(* LS Electric XG5000 project: 1군지사 유류제어(V1.0.3) *)
(* PLC LSPLC *)
(* module base 0 slot 0: FEnet:XGL-EFMT(B) (Fast Ethernet 통신 모듈, 전기 Master) *)
(* module base 1 slot 0: 입력 모듈:XGI-D28A/B (DC 24V 입력, 64점 (전류소스 싱크공용/ 전류소스 입력)) *)
(* module base 1 slot 1: 입력 모듈:XGI-D28A/B (DC 24V 입력, 64점 (전류소스 싱크공용/ 전류소스 입력)) *)
(* module base 1 slot 2: 출력 모듈:XGQ-TR8A/B (트랜지스터 출력, 64점 (0.1A용, 싱크출력/소스출력)) *)
(* module base 1 slot 3: 출력 모듈:XGQ-TR4A/B (트랜지스터 출력, 32점 (0.1A용, 싱크출력/소스출력)) *)
(* module base 1 slot 4: 출력 모듈:XGQ-TR8A/B (트랜지스터 출력, 64점 (0.1A용, 싱크출력/소스출력)) *)
(* module base 1 slot 5: 입력 모듈:XGI-D24A/B (DC 24V 입력, 32점 (전류소스 싱크공용/ 전류소스 입력)) *)
(* module base 1 slot 6: 출력 모듈:XGQ-TR8A/B (트랜지스터 출력, 64점 (0.1A용, 싱크출력/소스출력)) *)
(* module base 1 slot 7: 출력 모듈:XGQ-TR4A/B (트랜지스터 출력, 32점 (0.1A용, 싱크출력/소스출력)) *)
(* module base 1 slot 8: 아날로그입력 모듈:XGF-AD4S (A/D 절연형 4채널) *)
(* module base 1 slot 9: 아날로그출력 모듈:XGF-DC4S (D/A 절연형 4채널(전류형)) *)
(* module base 1 slot 10: 아날로그출력 모듈:XGF-DC4S (D/A 절연형 4채널(전류형)) *)
(* module base 1 slot 11: 입력 모듈:XGI-D24A/B (DC 24V 입력, 32점 (전류소스 싱크공용/ 전류소스 입력)) *)
(* module base 2 slot 0: 입력 모듈:XGI-D24A/B (DC 24V 입력, 32점 (전류소스 싱크공용/ 전류소스 입력)) *)
(* module base 2 slot 1: 입력 모듈:XGI-D24A/B (DC 24V 입력, 32점 (전류소스 싱크공용/ 전류소스 입력)) *)
(* module base 2 slot 2: 입력 모듈:XGI-D24A/B (DC 24V 입력, 32점 (전류소스 싱크공용/ 전류소스 입력)) *)
(* module base 2 slot 3: 출력 모듈:XGQ-TR4A/B (트랜지스터 출력, 32점 (0.1A용, 싱크출력/소스출력)) *)
(* module base 2 slot 4: 출력 모듈:XGQ-TR4A/B (트랜지스터 출력, 32점 (0.1A용, 싱크출력/소스출력)) *)
(* module base 2 slot 5: 출력 모듈:XGQ-TR4A/B (트랜지스터 출력, 32점 (0.1A용, 싱크출력/소스출력)) *)
(* module base 2 slot 6: 아날로그입력 모듈:XGF-AD4S (A/D 절연형 4채널) *)
(* module base 2 slot 7: 아날로그출력 모듈:XGF-DC4S (D/A 절연형 4채널(전류형)) *)
(* module base 2 slot 9: 입력 모듈:XGI-D24A/B (DC 24V 입력, 32점 (전류소스 싱크공용/ 전류소스 입력)) *)
(* module base 3 slot 0: 입력 모듈:XGI-D24A/B (DC 24V 입력, 32점 (전류소스 싱크공용/ 전류소스 입력)) *)
(* module base 3 slot 1: 입력 모듈:XGI-D24A/B (DC 24V 입력, 32점 (전류소스 싱크공용/ 전류소스 입력)) *)
(* module base 3 slot 2: 입력 모듈:XGI-D24A/B (DC 24V 입력, 32점 (전류소스 싱크공용/ 전류소스 입력)) *)
(* module base 3 slot 3: 출력 모듈:XGQ-TR4A/B (트랜지스터 출력, 32점 (0.1A용, 싱크출력/소스출력)) *)
(* module base 3 slot 4: 출력 모듈:XGQ-TR4A/B (트랜지스터 출력, 32점 (0.1A용, 싱크출력/소스출력)) *)
(* module base 3 slot 5: 출력 모듈:XGQ-TR4A/B (트랜지스터 출력, 32점 (0.1A용, 싱크출력/소스출력)) *)
(* module base 3 slot 6: 출력 모듈:XGQ-TR4A/B (트랜지스터 출력, 32점 (0.1A용, 싱크출력/소스출력)) *)
(* module base 3 slot 7: 아날로그입력 모듈:XGF-AD4S (A/D 절연형 4채널) *)
(* module base 3 slot 8: 아날로그출력 모듈:XGF-DC4S (D/A 절연형 4채널(전류형)) *)
(* module base 4 slot 0: Cnet:XGL-CH2A/B (Cnet 통신 모듈(RS-232C, RS-422/485)) *)
VAR_GLOBAL
    RP01_2차 : TON;
    RP01_3차 : TON;
    _0108_CH0_ACT AT %UX1.8.16 : BOOL; (* 절연형 아날로그입력 모듈: 채널0 운전중 *)
    _0108_CH0_DATA AT %UW1.8.2 : INT; (* 절연형 아날로그입력 모듈: 채널0 변환값 *)
    _0108_CH0_IDD AT %UX1.8.160 : BOOL; (* 절연형 아날로그입력 모듈: 채널0 입력단선검출 *)
    _0108_CH1_ACT AT %UX1.8.17 : BOOL; (* 절연형 아날로그입력 모듈: 채널1 운전중 *)
    _0108_CH1_DATA AT %UW1.8.3 : INT; (* 절연형 아날로그입력 모듈: 채널1 변환값 *)
    _0108_CH1_IDD AT %UX1.8.161 : BOOL; (* 절연형 아날로그입력 모듈: 채널1 입력단선검출 *)
    _0108_CH2_ACT AT %UX1.8.18 : BOOL; (* 절연형 아날로그입력 모듈: 채널2 운전중 *)
    _0108_CH2_DATA AT %UW1.8.4 : INT; (* 절연형 아날로그입력 모듈: 채널2 변환값 *)
    _0108_CH2_IDD AT %UX1.8.162 : BOOL; (* 절연형 아날로그입력 모듈: 채널2 입력단선검출 *)
    _0108_CH3_ACT AT %UX1.8.19 : BOOL; (* 절연형 아날로그입력 모듈: 채널3 운전중 *)
    _0108_CH3_DATA AT %UW1.8.5 : INT; (* 절연형 아날로그입력 모듈: 채널3 변환값 *)
    _0108_CH3_IDD AT %UX1.8.163 : BOOL; (* 절연형 아날로그입력 모듈: 채널3 입력단선검출 *)
    _0109_CH0_ACT AT %UX1.9.16 : BOOL; (* 절연형 아날로그출력 모듈: 채널0 운전중 *)
    _0109_CH0_DATA AT %UW1.9.3 : INT; (* 절연형 아날로그출력 모듈: 채널0 입력값 *)
    _0109_CH0_ERR AT %UX1.9.0 : BOOL; (* 절연형 아날로그출력 모듈: 채널0 에러 *)
    _0109_CH0_OUTEN AT %UX1.9.32 : BOOL; (* 절연형 아날로그출력 모듈: 채널0 출력상태설정 *)
    _0109_CH1_ACT AT %UX1.9.17 : BOOL; (* 절연형 아날로그출력 모듈: 채널1 운전중 *)
    _0109_CH1_DATA AT %UW1.9.4 : INT; (* 절연형 아날로그출력 모듈: 채널1 입력값 *)
    _0109_CH1_ERR AT %UX1.9.1 : BOOL; (* 절연형 아날로그출력 모듈: 채널1 에러 *)
    _0109_CH2_ACT AT %UX1.9.18 : BOOL; (* 절연형 아날로그출력 모듈: 채널2 운전중 *)
    _0109_CH2_DATA AT %UW1.9.5 : INT; (* 절연형 아날로그출력 모듈: 채널2 입력값 *)
    _0109_CH2_ERR AT %UX1.9.2 : BOOL; (* 절연형 아날로그출력 모듈: 채널2 에러 *)
    _0109_CH3_ACT AT %UX1.9.19 : BOOL; (* 절연형 아날로그출력 모듈: 채널3 운전중 *)
    _0109_CH3_DATA AT %UW1.9.6 : INT; (* 절연형 아날로그출력 모듈: 채널3 입력값 *)
    _0109_CH3_ERR AT %UX1.9.3 : BOOL; (* 절연형 아날로그출력 모듈: 채널3 에러 *)
    _0109_OUTEN AT %UW1.9.2 : WORD; (* 절연형 아날로그출력 모듈: 출력상태 설정 *)
    _0110_CH0_ACT AT %UX1.10.16 : BOOL; (* 절연형 아날로그출력 모듈: 채널0 운전중 *)
    _0110_CH0_DATA AT %UW1.10.3 : INT; (* 절연형 아날로그출력 모듈: 채널0 입력값 *)
    _0110_CH0_ERR AT %UX1.10.0 : BOOL; (* 절연형 아날로그출력 모듈: 채널0 에러 *)
    _0110_OUTEN AT %UW1.10.2 : WORD; (* 절연형 아날로그출력 모듈: 출력상태 설정 *)
    _0206_CH0_ACT AT %UX2.6.16 : BOOL; (* 절연형 아날로그입력 모듈: 채널0 운전중 *)
    _0206_CH0_DATA AT %UW2.6.2 : INT; (* 절연형 아날로그입력 모듈: 채널0 변환값 *)
    _0206_CH0_IDD AT %UX2.6.160 : BOOL; (* 절연형 아날로그입력 모듈: 채널0 입력단선검출 *)
    _0206_CH1_ACT AT %UX2.6.17 : BOOL; (* 절연형 아날로그입력 모듈: 채널1 운전중 *)
    _0206_CH1_DATA AT %UW2.6.3 : INT; (* 절연형 아날로그입력 모듈: 채널1 변환값 *)
    _0206_CH1_IDD AT %UX2.6.161 : BOOL; (* 절연형 아날로그입력 모듈: 채널1 입력단선검출 *)
    _0206_CH2_ACT AT %UX2.6.18 : BOOL; (* 절연형 아날로그입력 모듈: 채널2 운전중 *)
    _0206_CH2_DATA AT %UW2.6.4 : INT; (* 절연형 아날로그입력 모듈: 채널2 변환값 *)
    _0206_CH2_IDD AT %UX2.6.162 : BOOL; (* 절연형 아날로그입력 모듈: 채널2 입력단선검출 *)
    _0206_CH3_ACT AT %UX2.6.19 : BOOL; (* 절연형 아날로그입력 모듈: 채널3 운전중 *)
    _0206_CH3_DATA AT %UW2.6.5 : INT; (* 절연형 아날로그입력 모듈: 채널3 변환값 *)
    _0206_CH3_IDD AT %UX2.6.163 : BOOL; (* 절연형 아날로그입력 모듈: 채널3 입력단선검출 *)
    _0207_CH0_ACT AT %UX2.7.16 : BOOL; (* 절연형 아날로그출력 모듈: 채널0 운전중 *)
    _0207_CH0_DATA AT %UW2.7.3 : INT; (* 절연형 아날로그출력 모듈: 채널0 입력값 *)
    _0207_CH0_ERR AT %UX2.7.0 : BOOL; (* 절연형 아날로그출력 모듈: 채널0 에러 *)
    _0207_CH1_ACT AT %UX2.7.17 : BOOL; (* 절연형 아날로그출력 모듈: 채널1 운전중 *)
    _0207_CH1_DATA AT %UW2.7.4 : INT; (* 절연형 아날로그출력 모듈: 채널1 입력값 *)
    _0207_CH2_ACT AT %UX2.7.18 : BOOL; (* 절연형 아날로그출력 모듈: 채널2 운전중 *)
    _0207_CH2_DATA AT %UW2.7.5 : INT; (* 절연형 아날로그출력 모듈: 채널2 입력값 *)
    _0207_CH2_ERR AT %UX2.7.2 : BOOL; (* 절연형 아날로그출력 모듈: 채널2 에러 *)
    _0207_CH3_DATA AT %UW2.7.6 : INT; (* 절연형 아날로그출력 모듈: 채널3 입력값 *)
    _0207_OUTEN AT %UW2.7.2 : WORD; (* 절연형 아날로그출력 모듈: 출력상태 설정 *)
    _0307_CH0_ACT AT %UX3.7.16 : BOOL; (* 절연형 아날로그입력 모듈: 채널0 운전중 *)
    _0307_CH0_DATA AT %UW3.7.2 : INT; (* 절연형 아날로그입력 모듈: 채널0 변환값 *)
    _0307_CH0_IDD AT %UX3.7.160 : BOOL; (* 절연형 아날로그입력 모듈: 채널0 입력단선검출 *)
    _0307_CH1_ACT AT %UX3.7.17 : BOOL; (* 절연형 아날로그입력 모듈: 채널1 운전중 *)
    _0307_CH1_DATA AT %UW3.7.3 : INT; (* 절연형 아날로그입력 모듈: 채널1 변환값 *)
    _0307_CH1_IDD AT %UX3.7.161 : BOOL; (* 절연형 아날로그입력 모듈: 채널1 입력단선검출 *)
    _0307_CH2_ACT AT %UX3.7.18 : BOOL; (* 절연형 아날로그입력 모듈: 채널2 운전중 *)
    _0307_CH2_DATA AT %UW3.7.4 : INT; (* 절연형 아날로그입력 모듈: 채널2 변환값 *)
    _0307_CH2_IDD AT %UX3.7.162 : BOOL; (* 절연형 아날로그입력 모듈: 채널2 입력단선검출 *)
    _0307_CH3_DATA AT %UW3.7.5 : INT; (* 절연형 아날로그입력 모듈: 채널3 변환값 *)
    _0307_CH3_IDD AT %UX3.7.163 : BOOL; (* 절연형 아날로그입력 모듈: 채널3 입력단선검출 *)
    _0308_CH0_ACT AT %UX3.8.16 : BOOL; (* 절연형 아날로그출력 모듈: 채널0 운전중 *)
    _0308_CH0_DATA AT %UW3.8.3 : INT; (* 절연형 아날로그출력 모듈: 채널0 입력값 *)
    _0308_CH1_ACT AT %UX3.8.17 : BOOL; (* 절연형 아날로그출력 모듈: 채널1 운전중 *)
    _0308_CH1_DATA AT %UW3.8.4 : INT; (* 절연형 아날로그출력 모듈: 채널1 입력값 *)
    _0308_CH2_ACT AT %UX3.8.18 : BOOL; (* 절연형 아날로그출력 모듈: 채널2 운전중 *)
    _0308_CH2_DATA AT %UW3.8.5 : INT; (* 절연형 아날로그출력 모듈: 채널2 입력값 *)
    _0308_CH2_ERR AT %UX3.8.2 : BOOL; (* 절연형 아날로그출력 모듈: 채널2 에러 *)
    _0308_CH3_ACT AT %UX3.8.19 : BOOL; (* 절연형 아날로그출력 모듈: 채널3 운전중 *)
    _0308_CH3_DATA AT %UW3.8.6 : INT; (* 절연형 아날로그출력 모듈: 채널3 입력값 *)
    _0308_CH3_ERR AT %UX3.8.3 : BOOL; (* 절연형 아날로그출력 모듈: 채널3 에러 *)
    _0308_OUTEN AT %UW3.8.2 : WORD; (* 절연형 아날로그출력 모듈: 출력상태 설정 *)
END_VAR
VAR_GLOBAL CONSTANT
    _F0308_CH0_DEC_RATE : UINT := 30; (* 절연형 아날로그출력 모듈: 채널0 변화율 감소값 *)
    _F0308_CH0_STAT : UINT := 03; (* 절연형 아날로그출력 모듈: 채널0 이상 상태 출력 설정값 *)
    _F0308_LIMIT_EN : UINT := 19; (* 절연형 아날로그출력 모듈: 출력제한 채널 설정 *)
END_VAR

(* Comments on direct variables
%QX1.2.0	UPS ON LAMP
%QX1.2.1	UPS TROUBLE LAMP
%QX1.2.2	MCC ON LAMP
%QX1.2.3	AUTO LAMP
%QX1.2.4	MANUAL LAMP
%QX1.2.5	HORN STOP LAMP
%QX1.2.6	RESET LAMP
%QX1.2.7	LAMP TEST LAMP
%QX1.2.8	SYSTEM PRESSURE MIN
LAMP
%QX1.2.9	PUMP RESTART 6TIME/H
LAMP
%QX1.2.10	EV-1 LAMP
%QX1.2.11	EV-2 LAMP
%QX1.2.12	BPCV LAMP
%QX1.2.13	SPARE LAMP
%QX1.2.14	SPARE LAMP
%QX1.2.15	CONTROL PANEL EM S/W
LAMP
%QX1.2.16	DF-1A TANK EM S/W
LAMP
%QX1.2.17	DF-1B TANK EM S/W
LAMP
%QX1.2.18	DRAIN TANK EM S/W
LAMP
%QX1.2.19	FILTER ROOM EM S/W
LAMP
%QX1.2.20	대량 주유대 1 EM S/W
LAMP
%QX1.2.21	대량 주유대 2 EM S/W
LAMP
%QX1.2.22	대량 주유대 3 EM S/W
LAMP
%QX1.2.23	대량 주유대 4 EM S/W
LAMP
%QX1.2.24	포장 주유대 EM S/W
LAMP
%QX1.2.25	PIT-1 TROUBLE LAMP
%QX1.2.26	PIT-2 TROUBLE LAMP
%QX1.2.27	FIT-1 TROUBLE LAMP
%QX1.2.28	FIT-2 TROUBLE LAMP
%QX1.2.29	PLC 1 RUN LAMP
%QX1.2.30	PLC 1 STANDBY LAMP
%QX1.2.31	PLC 1 TROUBLE LAMP
%QX1.2.32	PLC 2 RUN LAMP

%QX1.2.33	PLC 2 STANDBY LAMP

%QX1.2.34	PLC 2 TROUBLE LAMP

%QX1.2.35	DF-1 DRAIN PUMP 1 TROUBLE LAMP

%QX1.2.36	DF-1 DRAIN PUMP 1 LOCAL LAMP

%QX1.2.37	DP-01 STOP LAMP

%QX1.2.38	DF-1 DRAIN PUMP RUN LAMP

%QX1.2.39	DTK-1 HLVD LAMP
%QX1.2.40	DTK-1 LEVEL HH LAMP

%QX1.2.41	DTK-1 LEVEL H LAMP

%QX1.2.42	DTK-1 LEVEL L LAMP

%QX1.2.43	DTK-1 LEVEL LL LAMP

%QX1.2.44	DTK-1 LEVEL TROUBLE LAMP

%QX1.2.45	SPARE LAMP

%QX1.2.46	SPARE LAMP
%QX1.2.47	SPARE LAMP
%QX1.3.0	경광등
%QX1.3.1	RP11 LEVEL TROUBLE RELAY
%QX1.3.3	RP-1 START RELAY
%QX1.3.4	RP01LEVEL HH RELAY
%QX1.3.5	RP01 INVERTER RESET RELAY
%QX1.3.7	RP-2 START RELAY
%QX1.3.8	RP02 LEVEL HH RELAY
%QX1.3.9	RP02 INVERTER RESET
RELAY
%QX1.3.11	RP03 START RELAY
%QX1.3.12	DF-1B RP3 LEVEL HH RELAY
%QX1.3.13	RP03 INVERTER RESET RELAY
%QX1.3.14	RP1, RP2 LEVEL TROUBLE RELAY
%QX1.3.16	RP04 START RELAY
%QX1.3.17	RP9 LEVEL TROUBLE RELAY
%QX1.3.18	RP10 LEVEL TROUBLE RELAY
%QX1.3.20	RP-9 START RELAY
%QX1.3.21	RP9 LEVEL LL RELAY

%QX1.3.22	RP3, RP4 LEVEL TROUBLE RELAY
%QX1.3.24	RP-10 START RELAY
%QX1.3.25	RP10 LEVEL HH RELAY
%QX1.3.26	RP10 INVERTER RESET RELAY
%QX1.3.28	RP11 START RELAY
%QX1.3.29	RP11 LEVEL HH RELAY
%QX1.3.30	RP11 INVERTER RESET RELAY
%QX1.4.0	RP12 START RELAY
%QX1.4.1	RP12 LEVEL TROUBLE RELAY
%QX1.4.2	RP12 INVERTER RESET RELAY
%QX1.4.4	SP-1 START RELAY

%QX1.4.5	DF-1A SUMP PUMP DMPI RESET RELAY

%QX1.4.7	SP-2 START RELAY
%QX1.4.8	DF-1B SUMP PUMP DMPI RESET RELAY

%QX1.4.10	DF-1B FAN START RELAY
%QX1.4.11	DF-1A FAN START RELAY
%QX1.4.13	DF-1 DRAIN PUMP START RELAY

%QX1.4.14	DP1 LEVEL TROUBLE RELAY
%QX1.4.16	EV-1 SOLVALVE RELAY
%QX1.4.17	EV-2 SOLVALVE RELAY
%QX1.4.18	EV-3 SOLVALVE RELAY
%QX1.4.19	EV-4 SOLVALVE RELAY
%QX1.4.20	EV-5 SOLVALVE RELAY
%QX1.4.21	EV-6 SOLVALVE RELAY
%QX1.4.22	DF-1/BPCV SOLVALVE RELAY
%QX1.4.23	DF-M/BPCV SOLVALVE RELAY
%QX1.4.24	MOGAS/BPCV SOLVALVE RELAY
%QX1.4.25	DF-1B HLV SOLVALVE RELAY

%QX1.4.26	DF-1A HLV SOLVALVE RELAY
%QX1.4.32	SP1 LEVEL TROUBLE RELAY
%QX1.4.33	SP2 LEVEL TROUBLE RELAY
%QX1.4.34	DMPI RESET
%QX1.4.35	DMPI RESET
%QX1.4.36	RP04 DMPI RESET RELAY
%QX1.4.48	RP-1 TIME WATCH RELAY
%QX1.4.49	RP-2 TIME WATCH RELAY
%QX1.4.50	RP-3 TIME WATCH RELAY

%QX1.4.51	RP-4 TIME WATCH RELAY

%QX1.4.52	RP9 TIME WATCH RELAY

%QX1.4.53	RP-10 TIME WATCH RELAY

%QX1.4.54	RP-11 TIME WATCH RELAY

%QX1.4.55	RP-12 TIME WATCH RELAY

%QX1.6.0	DF-1B FAN RUN LAMP
%QX1.6.1	DF-1B HLV LAMP

%QX1.6.2	RP-1 TROUBLE LAMP
%QX1.6.3	RP-1 LOCAL LAMP
%QX1.6.4	RP-1 STOP LAMP
%QX1.6.5	RP-1 RUN LAMP
%QX1.6.6	SUMP-1 TROUBLE LAMP
%QX1.6.7	SUMP-1 LOCAL LAMP
%QX1.6.8	SUMP-1 STOP LAMP
%QX1.6.9	SUMP-1 RUN LAMP
%QX1.6.10	RP-2 TROUBLE LAMP

%QX1.6.11	RP-2 LOCAL LAMP

%QX1.6.12	RP-2 STOP LAMP

%QX1.6.13	RP-2 RUN LAMP

%QX1.6.14	DF-1B LEVEL HH LAMP

%QX1.6.15	DF-1B LEVEL H LAMP

%QX1.6.16	DF-1B LEVEL L LAMP

%QX1.6.17	DF-1B LEVEL LL LAMP

%QX1.6.18	DF-1A LEVEL TROUBLE LAMP

%QX1.6.19	DF-1B 소화피트-1 누수 LAMP

%QX1.6.20	DF-1B 소화피트-1 누유 LAMP

%QX1.6.21	DF-1B 소화피트-2 누수 LAMP

%QX1.6.22	DF-1B 소화피트-2 누유 LAMP

%QX1.6.23	DF-1B 소화피트-3 누수 LAMP

%QX1.6.24	DF-1B 소화피트-3 누유 LAMP

%QX1.6.25	DF-1B 소화피트-4 누수 LAMP

%QX1.6.26	DF-1B 소화피트-4 누유 LAMP

%QX1.6.27	PUMP 선택 RP-1 1ST SET LAMP

%QX1.6.28	PUMP 선택 RP-2 1ST SET LAMP
%QX1.6.29	PUMP 선택 RP-3 1ST SET LAMP
%QX1.6.30	PUMP 선택 RP-4 1ST SET LAMP
%QX1.6.31	PUMP 선택 RP-1 2ST SET LAMP
%QX1.6.32	PUMP 선택 RP-2 2ST SET LAMP
%QX1.6.33	PUMP 선택 RP-3 2ST SET LAMP
%QX1.6.34	PUMP 선택 RP-4 2ST SET LAMP
%QX1.6.35	DF-1A FAN RUN LAMP
%QX1.6.36	DF-1A HLV LAMP

%QX1.6.37	RP-3 TROUBLE LAMP

%QX1.6.38	RP-3 LOCAL LAMP

%QX1.6.39	RP-3 STOP LAMP

%QX1.6.40	RP-3 RUN LAMP

%QX1.6.41	SUMP-2 TROUBLE LAMP

%QX1.6.42	SUMP-2 LOCAL LAMP

%QX1.6.43	SUMP-2 STOP LAMP

%QX1.6.44	SUMP-2 RUN LAMP

%QX1.6.45	RP-4 TROUBLE LAMP

%QX1.6.46	RP-4 LOCAL LAMP

%QX1.6.47	RP-4 STOP LAMP

%QX1.6.48	RP-4 RUN LAMP

%QX1.6.49	DF-1A LEVEL HH LAMP

%QX1.6.50	DF-1A LEVEL H LAMP

%QX1.6.51	DF-1A LEVEL L LAMP

%QX1.6.52	DF-1A LEVEL LL LAMP

%QX1.6.53	DF-1B LEVEL TROUBLE LAMP

%QX1.6.54	DF-1A 소화피트-1 누수 LAMP

%QX1.6.55	DF-1A 소화피트-1 누유 LAMP

%QX1.6.56	DF-1A 소화피트-2 누수 LAMP

%QX1.6.57	DF-1A 소화피트-2 누유 LAMP

%QX1.6.58	DF-1A 소화피트-3 누수 LAMP

%QX1.6.59	DF-1A 소화피트-3 누유 LAMP

%QX1.6.60	DF-1A 소화피트-4 누수 LAM

%QX1.6.61	DF-1A 소화피트-4 누유 LAMP

%QX1.6.62	RP-9 TROUBLE LAMP
%QX1.6.63	RP-9 LOCAL LAMP

%QX1.7.0	RP-9 STOP LAMP

%QX1.7.1	RP-9 RUN LAMP
 
%QX1.7.2	RP-10 TROUBLE LAMP
%QX1.7.3	RP-10 LOCAL LAMP
%QX1.7.4	RP-10 STOP LAMP
%QX1.7.5	RP-10 RUN LAMP
%QX1.7.6	RP-11 TROUBLE LAMP

%QX1.7.7	RP-11 LOCAL LAMP

%QX1.7.8	RP-11 STOP LAMP

%QX1.7.9	RP-11 RUN LAMP

%QX1.7.10	RP-12 TROUBLE LAMP
%QX1.7.11	RP-12 LOCAL LAMP
%QX1.7.12	RP-12 STOP LAMP
%QX1.7.13	RP-12 RUN LAMP
%QX2.3.0	RP-7 START RELAY [TO MCC]
%QX2.3.1	DF-M PUMP RP7 DMPI RESET RELAY

%QX2.3.2	DF-M PUMP RP7 INVERTER RESET
 RELAY
%QX2.3.4	RP-8 START RELAY
%QX2.3.5	DF-M PUMP RP8 DMPI RESET RELAY

%QX2.3.6	DF-M PUMP RP8 INVERTER RESET RELAY

%QX2.3.8	DF-M PUMP RP13 START RELAY

%QX2.3.9	RP13 LEVEL TROUBLE RELAY
%QX2.3.10	DF-M PUMP RP13 INVERTER RESET RELAY

%QX2.3.12	PUMP RP14 START RELAY

%QX2.3.13	RP14 LEVEL TROUBLE RELAY
%QX2.3.14	PUMP RP14 INVERTER RESET RELAY

%QX2.3.16	SP-4 START RELAY

%QX2.3.17	DF-M SUMP PUMP DMPI RESET RELAY

%QX2.3.19	DF-M FAN START RELAY
%QX2.3.21	RP7. RP8 LEVEL TROUBLE RELAY
%QX2.3.22	SP4 LEVEL TROUBLE RELAY
%QX2.3.24	RP-7 TIME WATCH RELAY

%QX2.3.25	RP-8 TIME WATCH RELAY
%QX2.3.26	RP-13 TIME WATCH RELAY
%QX2.3.27	RP-14 TIME WATCH RELAY
%QX2.4.0	DF-M EV-3 LAMP

%QX2.4.1	DF-M EV-4 LAMP

%QX2.4.3	DF-M BPCV LAMP

%QX2.4.6	FILTER ROOM EM-STOP LAMP

%QX2.4.7	DF-M TANK EM-STOP LAMP

%QX2.4.8	DF-M 대량 주유대 EM-STOP LAMP

%QX2.4.9	DF-M 포장주유대 EM-STOP DRUM LAMP

%QX2.4.12	RP-7 SET LAMP

%QX2.4.13	RP-8 SET LAMP

%QX2.4.14	DF-M PIT-3 TROUBLE LAMP

%QX2.4.15	DF-M PIT-4 TROUBLE LAMP

%QX2.4.16	DF-M FIT-3 TROUBLE LAMP

%QX2.4.17	DF-M FIT-4 TROUBLE LAMP

%QX2.4.18	RP-13 TROUBLE LAMP

%QX2.4.19	RP-13 LOCAL LAMP

%QX2.4.20	RP-13 STOP LAMP

%QX2.4.21	RP-13 RUN LAMP

%QX2.4.22	RP-14 TROUBLE LAMP

%QX2.4.23	RP-14 LOCAL LAMP

%QX2.4.24	RP-14 STOP LAMP

%QX2.4.25	RP-14 RUN LAMP

%QX2.4.26	DF-M FAN LAMP

%QX2.4.27	RP-7 TROUBLE LAMP [PANEL]
%QX2.4.28	RP-7 LOCAL LAMP [PANEL]
%QX2.4.29	RP-7 STOP LAMP [PANEL]
%QX2.4.30	RP-7 RUN LAMP [PANEL]
%QX2.4.31	SP-4 TROUBLE LAMP

%QX2.5.0	SUMP-4 LOCAL LAMP

%QX2.5.1	SUMP-4 STOP LAMP

%QX2.5.2	SUMP-4 RUN LAMP

%QX2.5.3	RP-8 TROUBLE LAMP

%QX2.5.4	RP-8 LOCAL LAMP

%QX2.5.5	RP-8 STOP LAMP

%QX2.5.6	RP-8 RUN LAMP

%QX2.5.7	DF-M LEVEL HH LAMP

%QX2.5.8	DF-M LEVEL H LAMP

%QX2.5.9	DF-M LEVEL L LAMP

%QX2.5.10	DF-M LEVEL LL LAMP
%QX2.5.11	DF-M LEVEL TROUBLE LAMP

%QX2.5.12	DF-M 소화피트-1 누수 LAMP

%QX2.5.13	DF-M 소화피트-1 누유 LAMP

%QX2.5.14	DF-M 소화피트-2 누수 LAMP

%QX2.5.15	DF-M 소화피트-2 누유 LAMP

%QX2.5.16	DF-M 소화피트-3 누수 LAMP

%QX2.5.17	DF-M 소화피트-3 누유 LAMP

%QX2.5.18	DF-M 소화피트-4 누수 LAMP

%QX2.5.19	DF-M 소화피트-4 누유 LAMP

%QX3.2.21	RP5, RP6 LEVEL TROUBLE RELAY
%QX3.3.0	PUMP RP5 START RELAY
%QX3.3.1	RP15 LEVEL TROUBLE RELAY

%QX3.3.2	RP16 LEVEL TROUBLE RELAY
%QX3.3.4	PUMP RP6 START RELAY
%QX3.3.5	PUMP RP6 DMPI RESET RELAY

%QX3.3.6	PUMP RP6 INVERTER RESET RELAY

%QX3.3.8	PUMP RP15 START RELAY
%QX3.3.9	PUMP RP15 DMPI RESET RELAY
%QX3.3.10	PUMP RP15 INVERTER RESET RELAY
%QX3.3.12	PUMP RP16 START RELAY

%QX3.3.13	PUMP RP16 DMPI RESET RELAY
%QX3.3.14	PUMP RP16 INVERTER RESET RELAY

%QX3.3.16	SP-3 START RELAY
%QX3.3.17	DP2 LEVEL TROUBLE RELAY
%QX3.3.19	FAN START RELAY

%QX3.3.21	RP5, RP6 LEVEL TROUBLE RELAY
%QX3.3.22	SP3 LEVEL TROUBLE RELAY
%QX3.3.24	RP-5 TIME WATCH RELAY

%QX3.3.25	RP-6 TIME WATCH RELAY
%QX3.3.26	RP-15 TIME WATCH RELAY
%QX3.3.27	RP-16 TIME WATCH RELAY
%QX3.3.28	DRAIN TANK TIME WATCH RELAY
%QX3.4.0	DRAIN PUMP START RELAY

%QX3.4.1	DRAIN PUMP DMPI RESET RELAY

%QX3.4.3	BUZZER 1 RELAY

%QX3.4.4	BUZZER 2 RELAY
%QX3.4.5	BUZZER 3 RELAY
%QX3.4.6	BUZZER 4 RELAY
%QX3.4.7	BUZZER 5 RELAY
%QX3.5.0	MOGAS EV-5 LAMP

%QX3.5.1	MOGAS EV-6 LAMP
%QX3.5.3	MOGAS BPCV LAMP
%QX3.5.6	MOGAS FILTER ROOM EM S/W LAMP
%QX3.5.7	MOGAS TANK EM S/W LAMP
%QX3.5.8	MOGAS 대량 주유대 EM S/W LAMP
%QX3.5.9	MOGAS 포장주유대 EM STOP LAMP
%QX3.5.10	MOGAS DRAIN TANK-2 EM S/W LAMP
%QX3.5.12	MOGAS RP-5 SET LAMP
%QX3.5.13	MOGAS RP-6 SET LAMP
%QX3.5.14	MOGAS PIT-5 TROUBLE LAMP
%QX3.5.15	MOGAS PIT-6 TROUBLE LAMP
%QX3.5.16	MOGAS FIT-5 TROUBLE LAMP
%QX3.5.17	MOGAS FIT-6 TROUBLE LAMP
%QX3.5.18	RP-15 TROUBLE LAMP
%QX3.5.19	RP-15 LOCAL LAMP
%QX3.5.20	RP-15 STOP LAMP
%QX3.5.21	RP-15 RUN LAMP
%QX3.5.22	RP-16 TROUBLE LAMP
%QX3.5.23	RP-16 LOCAL LAMP
%QX3.5.24	RP-16 STOP LAMP
%QX3.5.25	RP-16 RUN LAMP
%QX3.5.26	MOGAS FAN LAMP
%QX3.5.27	RP-5 TROUBLE LAMP
%QX3.5.28	RP-5 LOCAL LAMP
%QX3.5.29	RP-5 STOP LAMP
%QX3.5.30	RP-5 RUN LAMP
%QX3.5.31	SP-3 TROUBLE LAMP
%QX3.6.0	SUMP-3 LOCAL LAMP

%QX3.6.1	SUMP-3 STOP LAMP

%QX3.6.2	SUMP-3 RUN LAMP

%QX3.6.3	RP-6 TROUBLE LAMP
%QX3.6.4	RP-6 LOCAL LAMP
%QX3.6.5	RP-6 STOP LAMP
%QX3.6.6	RP-6 RUN LAMP
%QX3.6.7	MOGAS LEVEL HH LAMP
%QX3.6.8	MOGAS LEVEL H LAMP
%QX3.6.9	MOGAS LEVEL L LAMP
%QX3.6.10	MOGAS LEVEL LL LAMP
%QX3.6.11	MOGAS LEVEL TROUBLE LAMP
%QX3.6.12	MOGAS 소화피트-1 누수 LAMP
%QX3.6.13	MOGAS 소화피트-1 누유 LAMP
%QX3.6.14	MOGAS 소화피트-2 누수 LAMP
%QX3.6.15	MOGAS 소화피트-2 누유 LAMP
%QX3.6.16	MOGAS 소화피트-3 누수 LAMP
%QX3.6.17	MOGAS 소화피트-3 누유 LAMP
%QX3.6.18	MOGAS 소화피트-4 누수 LAMP
%QX3.6.19	MOGAS 소화피트-4 누유 LAMP
%QX3.6.20	DP-02 TROUBLE LAMP

%QX3.6.21	DP-02 LOCAL LAMP
%QX3.6.22	DP-02 STOP LAMP
%QX3.6.23	DP-02 RUN LAMP
%QX3.6.24	DTK-2 HLVD LAMP
%QX3.6.25	DTK-2 LEVEL HH LAMP
%QX3.6.26	DTK-2 LEVEL H LAMP
%QX3.6.27	DTK-2 LEVEL L LAMP
%QX3.6.28	DTK-2 LEVEL LL LAMP
%QX3.6.29	DTK-2 LEVEL TROUBLE LAMP
%IX1.0.0	UPS ON
%IX1.0.1	UPS TROUBLE 
%IX1.0.3	MCCB POWER ON CHECK
%IX1.0.4	MCCB 2 POWER ON CHECK
%IX1.0.8	RP-1 REMOTE 선택 (MCC)
%IX1.0.9	RP-1 RUN (MCC)
%IX1.0.10	RP-1 DMPI(INV) ALARM (MCC)
%IX1.0.11	RP-1 FLOW S/W (MCC)
%IX1.0.12	RP-1 MCCB ON (MCC)
%IX1.0.13	RP-1 PUMP 과열 (MCC)
%IX1.0.16	RP-2 REMOTE 선택 (MCC)
%IX1.0.17	RP-2 RUN (MCC)
%IX1.0.18	RP-2 DMPI(INV) ALARM (MCC)
%IX1.0.19	FLOW S/W (MCC)
%IX1.0.20	RP-2 MCCB ON (MCC)
%IX1.0.21	RP-2 PUMP 과열 (MCC)
%IX1.0.24	RP-3 REMOTE 선택 (MCC)
%IX1.0.25	RP-3 RUN (MCC)
%IX1.0.26	RP-3 DMPI(INV) ALARM (MCC)
%IX1.0.27	FLOW S/W (MCC)
%IX1.0.28	RP-3 MCCB ON (MCC)
%IX1.0.29	RP-3 PUMP 과열 (MCC)
%IX1.0.32	RP -4 REMOTE 선택 (MCC)
%IX1.0.33	RP-4 RUN (MCC)
%IX1.0.34	RP-4 DMPI(INV) ALARM (MCC)
%IX1.0.35	FLOW S/W (MCC)
%IX1.0.36	RP-4 MCCB ON (MCC)
%IX1.0.37	RP-4 PUMP 과열 (MCC)
%IX1.0.40	RP-9 REMOTE 선택 (MCC)
%IX1.0.41	RP-9 RUN (MCC)
%IX1.0.42	RP-9 DMPI ALARM (MCC)
%IX1.0.43	RP-9 FLOW S/W (MCC)
%IX1.0.44	RP-9 MCCB ON (MCC)
%IX1.0.45	RP-9 PUMP 과열 (MCC)
%IX1.0.48	RP-10 REMOTE 선택 (MCC)
%IX1.0.49	RP-10 PUMP RUN (MCC)
%IX1.0.50	RP-10 DMPI ALARM (MCC)
%IX1.0.51	RP-10 FLOW S/W (MCC)
%IX1.0.52	RP-10 MCCB ON (MCC)
%IX1.0.53	RP-10 PUMP 과열 (MCC)
%IX1.0.56	RP-11 REMOTE 선택 (MCC)
%IX1.0.57	RP-11 PUMP RUN (MCC)
%IX1.0.58	RP-11 DMPI ALARM (MCC)
%IX1.0.59	RP-11 FLOW S/W (MCC)
%IX1.0.60	RP-11 MCCB ON (MCC)
%IX1.0.61	RP-11 PUMP 과열 (MCC)
%IX1.1.0	(단자불량)
%IX1.1.1	SP-1 DMPI ALARM (MCC)
%IX1.1.2	SP-1 REMOTE 선택 (MCC)
%IX1.1.3	FLOW S/W (MCC)
%IX1.1.4	SP-1 MCCB ON (MCC)
%IX1.1.5	SP-1 PUMP 과열 (MCC)
%IX1.1.7	SP-1 RUN (MCC)
%IX1.1.8	SP-2 RUN (MCC)
%IX1.1.9	SP-2 DMPI ALARM (MCC)
%IX1.1.10	SP-2 REMOTE 선택 (MCC)
%IX1.1.11	FLOW S/W (MCC)
%IX1.1.12	SP-2 MCCB ON (MCC)
%IX1.1.13	SP-2 PUMP 과열 (MCC)
%IX1.1.15	DRAIN TANK 1 HLVD (LIMIT)
%IX1.1.16	RP-12 REMOTE 선택 (MCC)
%IX1.1.17	RP-12 PUMP RUN (MCC)
%IX1.1.18	RP-12 DMPI ALARM (MCC)
%IX1.1.19	RP-12 FLOW S/W (MCC)
%IX1.1.20	RP-12 MCCB ON (MCC)
%IX1.1.21	RP-12 PUMP 과열 (MCC)
%IX1.1.24	DRAIN PUMP RUN (MCC)
%IX1.1.25	DRAIN PUMP 1 DMPI ALARM (MCC)
%IX1.1.26	DP-01 REMOTE 선택 (MCC)
%IX1.1.27	FLOW S/W (MCC)
%IX1.1.28	DRAIN PUMP 1 MCCB ON (MCC)
%IX1.1.29	DRAIN PUMP 1 PUMP 과열 (MCC)
%IX1.1.31	SOL VALVE 전원 이상
%IX1.1.32	SYSTEM AUTO S/W (PANEL)
%IX1.1.33	SYSTEM MANUAL S/W (PANEL)
%IX1.1.34	HORN STOP
%IX1.1.35	RESET S/W (PANEL)
%IX1.1.36	LAMP TEST S/W (PANEL)
%IX1.1.37	PIT 1 선택
%IX1.1.38	PIT 2 선택
%IX1.1.39	FIT 1 선택
%IX1.1.40	FIT 2 선택
%IX1.1.41	OPERTION SELECT SCADA
%IX1.1.42	OPERTION SELECT PANEL
%IX1.1.43	DRAIN PUMP STOP S/W (PANEL)
%IX1.1.44	DP-01 RUN S/W (PANEL)
%IX1.1.45	DP-1 MANUAL (PANEL)
%IX1.1.46	DP-1 AUTO (PANEL)
%IX1.1.47	제어실 EM-STOP (PANEL)
%IX1.5.0	DF1B HLV S/W (PANEL)
%IX1.5.1	DF-1B 개별 탱크 정지 KEY S/S (PANEL)
%IX1.5.2	RP-1 STOP S/W (PANEL)
%IX1.5.3	RP-1 RUN S/W (PANEL)
%IX1.5.4	SP-1 STOP S/W (PANEL)
%IX1.5.5	SP-1 RUN S/W (PANEL)
%IX1.5.6	RP-2 STOP S/W (PANEL)
%IX1.5.7	RP-2 PUMP RUN S/W (PANEL)
%IX1.5.8	출하 PUMP 1차선택 S/W RP-1
%IX1.5.9	출하 PUMP 1차선택 S/W RP-2
%IX1.5.10	출하 PUMP 1차선택 S/W RP-3
%IX1.5.11	출하 PUMP 1차선택 S/W RP-4
%IX1.5.12	출하 PUMP 2차선택 S/W RP-1
%IX1.5.13	출하 PUMP 2차선택 S/W RP-2
%IX1.5.14	출하 PUMP 2차선택 S/W RP-3
%IX1.5.15	출하 PUMP 2차선택 S/W RP-4
%IX1.5.16	DF1A HLV S/W (PANEL)
%IX1.5.17	DF-1A 개별 탱크 정지 KEY S/S (PANEL)
%IX1.5.18	RP-3 PUMP STOP S/W (PANEL)
%IX1.5.19	RP-3 PUMP RUN S/W (PANEL)
%IX1.5.20	SP-2 STOP S/W (PANEL)
%IX1.5.21	SP-2 RUN S/W (PANEL)
%IX1.5.22	RP-4 PUMP STOP S/W (PANEL)
%IX1.5.23	RP-4 PUMP RUN S/W (PANEL)
%IX1.5.24	RP-9 STOP S/W (PANEL)
%IX1.5.25	RP-9 RUN S/W (PANEL)
%IX1.5.26	RP-10 STOP S/W (PANEL)
%IX1.5.27	RP-10 RUN S/W (PANEL)
%IX1.5.28	RP-11 STOP S/W (PANEL)
%IX1.5.29	RP-11 RUN S/W (PANEL)
%IX1.5.30	RP-12 STOP S/W (PANEL)
%IX1.5.31	RP-12 RUN S/W (PANEL)
%IX1.11.0	RP-1 전시 비상 S/W
%IX1.11.1	SUMP PUMP1 전시 비상 S/W
%IX1.11.2	RP-2 전시 비상 S/W
%IX1.11.3	RP-3 전시 비상 S/W
%IX1.11.4	SP-2 전시 비상 S/W
%IX1.11.5	RP-4 전시 비상 S/W
%IX1.11.6	DP-01 전시 비상 S/W
%IX1.11.7	RP-9 전시 비상 S/W
%IX1.11.8	RP-10 전시 비상 S/W
%IX1.11.9	RP-11 전시 비상 S/W
%IX1.11.10	RP-12 전시 비상 S/W
%IX1.11.11	DF-1A FAN ON/OFF S/W (PLC)
%IX1.11.12	DF-1A FAN OFF S/W (TankRoom)
%IX1.11.13	DF-1A FAN ON S/W (TankRoom)
%IX1.11.14	DF-1A FAN DOOR S/W (TankRoom)
%IX1.11.16	DF-1A FAN RUN (MCC)
%IX1.11.17	DF-1B FAN ALARM (MCC)
%IX1.11.18	DF-1B FAN REMOTE (MCC)
%IX1.11.22	DF-1B FAN PLC RUN (MCC)
%IX1.11.23	DF-1A FAN ALARM (MCC)
%IX1.11.24	DF-1A FAN REMOTE (MCC)
%IX1.11.25	DF-1B FAN MCCB ON (MCC)
%IX1.11.27	DF-1B FAN ON/OFF S/W (PLC)
%IX1.11.28	DF-1B FAN OFF S/W (TankRoom)
%IX1.11.29	DF-1B FAN ON S/W (TankRoom)
%IX1.11.30	DF-1B FAN DOOR S/W (TankRoom)
%IX2.0.0	RP-7 REMOTE 선택 (MCC)
%IX2.0.1	RP-7 PUMP RUN (MCC)
%IX2.0.2	RP-7 DMPI ALARM (MCC)
%IX2.0.3	FLOW S/W (MCC)
%IX2.0.4	RP-7 MCCB ON (MCC)
%IX2.0.5	RP-7 PUMP 과열 (MCC)
%IX2.0.8	RP-8 REMOTE 선택 (MCC)
%IX2.0.9	RP-8 PUMP RUN (MCC)
%IX2.0.10	RP-8 DMPI ALARM (MCC)
%IX2.0.11	FLOW S/W (MCC)
%IX2.0.12	 RP-8 MCCB ON (MCC)
%IX2.0.13	RP-8 PUMP 과열 (MCC)
%IX2.0.16	RP-13 REMOTE 선택 (MCC)
%IX2.0.17	RP-13 PUMP RUN (MCC)
%IX2.0.18	RP-13 DMPI ALARM (MCC)
%IX2.0.19	RP-13 FLOW S/W (MCC)
%IX2.0.20	RP-13 MCCB ON (MCC)
%IX2.0.21	RP-13 PUMP 과열 (MCC)
%IX2.0.24	RP-14 REMOTE 선택 (MCC)
%IX2.0.25	RP-14 PUMP RUN (MCC)
%IX2.0.26	RP-14 DMPI ALARM (MCC)
%IX2.0.27	RP-14 FLOW S/W (MCC)
%IX2.0.28	RP-14 MCCB ON (MCC)
%IX2.0.29	RP-14 PUMP 과열 (MCC)
%IX2.1.0	SUMP PUMP-4 RUN (MCC)
%IX2.1.1	SUMP PUMP-4 DMPI ALARM (MCC)
%IX2.1.2	SP-4 REMOTE 선택 (MCC)
%IX2.1.3	FLOW S/W (MCC)
%IX2.1.4	SUMP PUMP-4 MCCB ON (MCC)
%IX2.1.5	SUMP PUMP-4 PUMP 과열 (MCC)
%IX2.1.8	DF-1 대량주유대 1 LOCAL/REMOTE(LDCAL)
%IX2.1.9	DF-1 대량주유대 1 RUN(LOCAL)
%IX2.1.10	DF-1 대량주유대 1 STOP (LOCAL)
%IX2.1.11	DF-1 대량주유대 1 EM STOP (LOCAL)
%IX2.1.12	DF-1 대량주유대 2 LOCAL/REMOTE(LDCAL)
%IX2.1.13	DF-1 대량주유대 2 RUN(LOCAL)
%IX2.1.14	DF-1 대량주유대 2 STOP (LOCAL)
%IX2.1.15	DF-1 대량주유대 2 EM STOP (LDCAL)
%IX2.1.16	RP-7 전시 비상 S/W
%IX2.1.17	RP-8 전시 비상 S/W
%IX2.1.18	SUMP PUMP-4 전시 비상 S/W
%IX2.1.19	RP-13 전시 비상 S/W
%IX2.1.20	RP-14 전시 비상 S/W
%IX2.1.21	DF-M FAN RUN (MCC)
%IX2.1.22	DF-M FAN ALARM (MCC)
%IX2.1.23	DF-M FAN REMOTE (MCC)
%IX2.1.24	DF-1 대량주유대 3 LOCAL/REMOTE(LDCAL)
%IX2.1.25	DF-1 대량주유대 3 RUN (LOCAL)
%IX2.1.26	DF-1 대량주유대 3 STOP (LOCAL)
%IX2.1.27	DF-1 대량주유대 3 EM STOP (LOCAL)
%IX2.1.28	DF-1 대량주유대 4 LOCAL/REMOTE(LDCAL)
%IX2.1.29	DF-1 대량주유대 4 RUN(LOCAL)
%IX2.1.30	DF-1 대량주유대 4 STOP (LOCAL)
%IX2.1.31	DF-1 대량주유대 4 EM STOP (LOCAL)
%IX2.2.0	출하 PUMP RP-07 선택 S/W
%IX2.2.1	출하 PUMP RP-08 선택 S/W
%IX2.2.2	PIT 1 선택
%IX2.2.3	PIT 2 선택
%IX2.2.4	FIT 1 선택
%IX2.2.5	FIT 2 선택
%IX2.2.6	RP-13 STOP S/W (PANEL)
%IX2.2.7	RP-13 RUN S/W (PANEL)
%IX2.2.8	RP-14 STOP S/W (PANEL)
%IX2.2.9	RP-14 RUN S/W (PANEL)
%IX2.2.10	개별 TANK PUMP STOP (PANEL)
%IX2.2.11	RP-7 STOP S/W (PANEL)
%IX2.2.12	RP-7 PUMP RUN S/W (PANEL)
%IX2.2.13	SP-4 STOP S/W (PANEL)
%IX2.2.14	SUMP PUMP-4 RUN S/W (PANEL)
%IX2.2.16	RP-8 STOP S/W (PANEL)
%IX2.2.17	RP-8 RUN S/W (PANEL)
%IX2.2.28	DF-M FAN ON S/W (TankRoom)
%IX2.2.29	DF-M FAN OFF S/W (TankRoom)
%IX2.2.30	DF-M FAN DOOR S/W (TankRoom)
%IX2.9.0	DF-1 포장주유대 LOCAL/REMOTE(LDCAL)
%IX2.9.1	DF-1 포장주유대 RUN (LOCAL)
%IX2.9.2	DF-1 포장주유대 STOP (LOCAL)
%IX2.9.3	DF-1 포장주유대 EM STOP (LOCAL)
%IX2.9.4	DF-M 대량주유대 LOCAL/REMOTE(LDCAL)
%IX2.9.5	DF-M 대량주유대 RUN (LOCAL)
%IX2.9.6	DF-M 대량주유대 STOP (LOCAL)
%IX2.9.7	DF-M 대량주유대 5 EM STOP (LOCAL)
%IX2.9.8	DF-M 포장주유대 LOCAL/REMOTE(LDCAL)
%IX2.9.9	DF-M 포장주유대 RUN (LOCAL)
%IX2.9.10	DF-M 포장주유대 STOP (LOCAL)
%IX2.9.11	DF-M 포장주유대 EM STOP (LOCAL)
%IX2.9.12	MOGAS 대량주유대 LOCAL/REMOTE(LDCAL)
%IX2.9.13	MOGAS 대량주유대 RUN (LOCAL)
%IX2.9.14	MOGAS 대량주유대 STOP (LOCAL)
%IX2.9.15	MOGAS 대량주유대 EM STOP (LOCAL)
%IX2.9.16	MOGAS 포장주유대 LOCAL/REMOTE(LDCAL)
%IX2.9.17	MOGAS 포장주유대 RUN (LOCAL)
%IX2.9.18	MOGAS 포장주유대 STOP (LOCAL)
%IX2.9.19	MOGAS 포장주유대 EM STOP (LOCAL)
%IX2.9.20	DF-1B TankRoom EM-STOP
%IX2.9.21	DF-1A TankRoom EM-STOP
%IX2.9.22	MOGAS TankRoom EM-STOP
%IX2.9.23	DF-M TankRoom EM-STOP
%IX2.9.24	 DF-1 FILTER ROOM EM-STOP
%IX2.9.25	 DF-M FILTER ROOM EM-STOP
%IX2.9.26	 MOGAS FILTER ROOM EM-STOP
%IX2.9.27	DRAIN TANK1 EM STOP (LOCAL)
%IX2.9.28	DRAIN TANK2 EM STOP (LOCAL)
%IX2.9.29	DF-M FAN S/L S/W
%IX2.9.30	DF-M FAN DOOR S/W
%IX2.9.31	DF-M FAN S/W (PANEL)
%IX3.0.0	RP-5 REMOTE 선택 (MCC)
%IX3.0.1	RP-5 PUMP RUN (MCC)
%IX3.0.2	RP-5 DMPI ALARM (MCC)
%IX3.0.3	FLOW S/W (MCC)
%IX3.0.4	RP-5 MCCB ON (MCC)
%IX3.0.5	RP-5 PUMP 과열 (MCC)
%IX3.0.8	RP-6 REMOTE 선택 (MCC)
%IX3.0.9	RP-6 PUMP RUN (MCC)
%IX3.0.10	RP-6 DMPI ALARM (MCC)
%IX3.0.11	FLOW S/W (MCC)
%IX3.0.12	RP-6 MCCB ON (MCC)
%IX3.0.13	RP-6 PUMP 과열 (MCC)
%IX3.0.16	RP-15 REMOTE 선택 (MCC)
%IX3.0.17	RP-15 PUMP RUN (MCC)
%IX3.0.18	RP-15 DMPI ALARM (MCC)
%IX3.0.19	RP-15 FLOW S/W (MCC)
%IX3.0.20	RP-15 MCCB ON (MCC)
%IX3.0.21	RP-15 PUMP 과열 (MCC)
%IX3.0.24	RP-16 REMOTE 선택 (MCC)
%IX3.0.25	RP-16 PUMP RUN (MCC)
%IX3.0.26	RP-16 DMPI ALARM (MCC)
%IX3.0.27	RP-16 FLOW S/W (MCC)
%IX3.0.28	RP-16 MCCB ON (MCC)
%IX3.0.29	RP-16 PUMP 과열 (MCC)
%IX3.1.0	SUMP PUMP-3 RUN (MCC)
%IX3.1.1	SUMP PUMP-3 DMPI ALARM (MCC)
%IX3.1.2	SUMP PUMP-3 REMOTE 선택 (MCC)
%IX3.1.3	FLOW S/W (MCC)
%IX3.1.4	SUMP PUMP-3 MCCB ON (MCC)
%IX3.1.5	SUMP PUMP-3 PUMP 과열 (MCC)
%IX3.1.8	DRAIN PUMP RUN (MCC)
%IX3.1.9	DP-02 DMPI ALARM (MCC)
%IX3.1.10	DP-02 REMOTE 선택 (MCC)
%IX3.1.11	FLOW S/W (MCC)
%IX3.1.12	DP-02 MCCB ON (MCC)
%IX3.1.13	DP-02 PUMP 과열 (MCC)
%IX3.1.15	DRAIN TANK 2 HLVD (LIMIT)
%IX3.1.16	RP-5 전시 비상 S/W
%IX3.1.17	SUMP PUMP-3 전시 비상 S/W
%IX3.1.18	RP-6 전시 비상 S/W
%IX3.1.19	DRAIN PUMP-2 전시 비상 S/W
%IX3.1.20	RP-15 전시 비상 S/W
%IX3.1.21	RP-16 전시 비상 S/W
%IX3.1.24	MOGAS FAN RUN (MCC)
%IX3.1.25	MOGAS FAN RUN (MCC)
%IX3.1.26	MOGAS FAN ALARM (MCC)
%IX3.1.27	MOGAS FAN REMOTE (MCC)
%IX3.1.28	DF-1B 누유
%IX3.1.29	DF-1A 누유
%IX3.1.30	MOGAS 누유
%IX3.1.31	DF-M 누유
%IX3.2.0	출하 PUMP RP-05 선택 S/W
%IX3.2.1	출하 PUMP RP-06 선택 S/W
%IX3.2.2	PIT 5 선택
%IX3.2.3	PIT 6 선택
%IX3.2.4	FIT 5 선택
%IX3.2.5	FIT 6 선택
%IX3.2.6	RP-15 STOP S/W (PANEL)
%IX3.2.7	RP-15 RUN S/W (PANEL)
%IX3.2.8	RP-16 STOP S/W (PANEL)
%IX3.2.9	RP-16 RUN S/W (PANEL)
%IX3.2.10	개별 TANK PUMP STOP (PANEL)
%IX3.2.11	RP-5 STOP S/W (PANEL)
%IX3.2.12	RP-5 RUN S/W (PANEL)
%IX3.2.13	SUMP PUMP-3 STOP S/W (PANEL)
%IX3.2.14	SUMP PUMP-3 RUN S/W (PANEL)
%IX3.2.15	RP-6 STOP S/W (PANEL)
%IX3.2.16	RP-6 RUN S/W (PANEL)
%IX3.2.17	DRAIN PUMP STOP S/W (PANEL)
%IX3.2.18	DP-02 RUN S/W (PANEL)
%IX3.2.19	DRAIN PUMP 2 MANUAL
%IX3.2.28	MOGAS FAN ON S/W (TankRoom)
%IX3.2.29	MOGAS FAN OFF S/W (TankRoom)
%IX3.2.30	MOGAS FAN DOOR S/W (TankRoom)
%MX0	P2P 쓰기 PULS
%MX1	P2P 읽기 PULS
%MX64	AUTO SET
%MX65	MANUAL SET
%MX6400	OPERTION SELECT (SCADA)
%MX12800	OPERTION SELECT (PANEL)
%MX12864	출하 PUMP RP-1,2,3,4 STOP
%MX12928	RP-01 2차 선택
%MX12929	RP-02 2차 선택
%MX12930	RP-03 2차 선택
%MX12931	RP-04 2차 선택
%MX12934	RP-01 1차 선택
%MX12935	RP-02 1차 선택
%MX12936	RP-03 1차 선택
%MX12937	RP-04 1차 선택
%MX12992	출하 PUMP RP-7,8 STOP
%MX13056	출하 PUMP RP-5,6 STOP
%MX13120	HORN STOP 1
%MX13121	HORN STOP 2
%MX13122	HORN STOP 3
%MX13440	DRAIN PUMP 1 RUN 
%MX13441	DRAIN PUMP 1 FLOW ALARM
%MX13442	DP-1 READY
%MX13445	DRAIN TK-113 Run SIG
%MX16000	RP-1 RUN (SCADA) (PANEL)
%MX16001	RP-1 FLOW ALARM
%MX16002	RP-1 RUN READY
%MX16004	RP-2 RUN (SCADA) (PANEL)
%MX16005	RP-2 FLOW ALARM
%MX16006	RP-2 RUN READY
%MX16008	SP-1 RUN 
%MX16009	SP-1 FLOW ALARM
%MX16010	SP-1 RUN READY
%MX16012	RP-3 RUN 
%MX16013	RP-03 FLOW ALARM
%MX16014	RP-3 RUN READY
%MX16016	RP-4 RUN 
%MX16017	RP-04 FLOW ALARM
%MX16018	RP-4 RUN READY
%MX16020	SP-2 RUN 
%MX16021	SP-2 FLOW ALARM
%MX16022	SP-2 RUN READY
%MX16024	RP-9 PUMP RUN 
%MX16025	RP-9 FLOW ALARM
%MX16026	RP-9 PUMP RUN READY
%MX16028	RP-10 RUN 
%MX16029	RP-10 FLOW ALARM
%MX16030	RP-10 RUN READY
%MX16032	RP-11 PUMP RUN 
%MX16033	RP-11 FLOW ALARM
%MX16034	RP-11 PUMP RUN READY
%MX16036	RP-12 PUMP RUN 
%MX16037	RP-12 FLOW ALARM
%MX16038	RP-12 PUMP RUN READY
%MX16640	DF-1 대량주유대 1 RUN
%MX16643	DF-1 대량주유대 2 RUN
%MX16646	DF-1 대량주유대 3 RUN
%MX16649	DF-1 대량주유대 4 RUN
%MX16652	DF-1 포장주유대 RUN
%MX16704	DF1 대량,포장 1개 이상 운전명령
%MX16705	DF1 대량,포장 ANY PUMP RUN SIG
%MX16768	RP-1 AUTO RUN 
%MX16769	RP-2 AUTO RUN 
%MX16770	RP-3 AUTO RUN 
%MX16771	RP-4 AUTO RUN 
%MX16832	1차 기동중
%MX16833	 2차 기동
%MX17280	DF-1A FAN RUN
%MX17281	DF-1A FAN RUN (TankRoom)
%MX17283	DF-1A FAN SIG (ARES)
%MX17284	DF-1A FAN RUN (ARES)
%MX17287	DF-1B FAN RUN
%MX17288	DF-1B FAN RUN [LOCAL]
%MX17290	DF-1B FAN PLC RUN SIG
%MX17291	DF-1B FAN PLC RUN
%MX17344	DF-1A HLV OPEN PULS
%MX17345	DF-1A HLV OPEN
%MX17408	DF-1B HLV OPEN PULS
%MX17409	DF-1B HLV OPEN
%MX19200	SYSTEM AUTO (PANEL)
%MX19201	SYSTEM MANU (PANEL)
%MX19264	DP-1 MANUAL
%MX19265	DP-1 AUTO
%MX19274	MOGAS DRAIN PUMP 2 MANUAL
%MX19275	DRAIN PUMP 2 AUTO
%MX19840	RP-7 PUMP RUN 
%MX19841	RP-7 FLOW ALARM
%MX19842	RP-7 PUMP RUN READY
%MX19844	RP-8 PUMP RUN 
%MX19845	RP-8 FLOW ALARM
%MX19846	RP-8 PUMP RUN READY
%MX19848	RP-13 PUMP RUN 
%MX19849	RP-13 FLOW ALARM
%MX19850	RP-13 PUMP RUN READY
%MX19852	RP-14 PUMP RUN 
%MX19853	RP-14 FLOW ALARM
%MX19854	RP-14 PUMP RUN READY
%MX19856	SP-4 RUN 
%MX19857	SUMP PUMP-4 FLOW ALARM
%MX19858	SP-4 RUN READY
%MX20480	DF-M 대량주유대 RUN
%MX20483	DF-M 포장주유대 RUN
%MX20544	RP-7 PUMP RUN 
%MX20545	RP-8 PUMP RUN 
%MX21120	DF-M FAN RUN
%MX21121	DF-M FAN RUN (TankRoom)
%MX21123	DF-M FAN PLC RUN SIG
%MX21124	DF-M FAN S/W (PLC OR SCADA)
%MX22400	RP-5 PUMP RUN 
%MX22401	RP-5 FLOW ALARM
%MX22402	RP-5 PUMP RUN READY
%MX22404	RP-6 PUMP RUN 
%MX22405	RP-6 FLOW ALARM
%MX22406	RP-6 PUMP RUN READY
%MX22408	RP-15 PUMP RUN 
%MX22409	RP-15 FLOW ALARM
%MX22410	RP-15 PUMP RUN READY
%MX22412	RP-16 PUMP RUN 
%MX22413	RP-16 FLOW ALARM
%MX22414	RP-16 PUMP RUN READY
%MX22416	SP-3 RUN 
%MX22417	SUMP PUMP-3 FLOW ALARM
%MX22418	SUMP PUMP-3 RUN READY
%MX22420	DRAIN PUMP RUN 
%MX22421	DP-02 FLOW ALARM
%MX22422	DRAIN PUMP RUN READY
%MX23040	MOGAS 대량주유대 RUN
%MX23043	MOGAS 포장주유대 RUN
%MX23104	RP-5 PUMP RUN 
%MX23105	RP-6 PUMP RUN 
%MX23680	MOGAS FAN RUN
%MX23681	MOGAS FAN RUN (TankRoom)
%MX23683	MOGAS FAN PLC RUN SIG
%MX23684	MOGAS FAN PLC RUN
%MX128000	LAMP TEST
%MX160000	ALL E-M STOP
%MX160001	RESET
%MX160002	ALL E-M STOP
%MX160010	ALL ALARM
%MX160011	ALL ALARM
%MX160020	ALL 누유 ALARM
%MX160064	제어실 EM-STOP (PANEL)
%MX160065	DF-1 대량주유대 1 EM STOP (LOCAL)
%MX160066	DF-1 대량주유대 2 EM STOP (LDCAL)
%MX160067	DF-1 대량주유대 3 EM STOP (LOCAL)
%MX160068	DF-1 대량주유대 4 EM STOP (LOCAL)
%MX160069	DF-M 대량주유대 5 EM STOP (LOCAL)
%MX160070	MOGAS 대량주유대 EM STOP (LOCAL)
%MX160071	DF-1 포장주유대 EM STOP (LOCAL)
%MX160072	DF-M 포장주유대 EM STOP (LOCAL)
%MX160073	MOGAS 포장주유대 EM STOP (LOCAL)
%MX160074	DF-1B TankRoom EM-STOP
%MX160075	DF-1A TankRoom EM-STOP
%MX160076	MOGAS TankRoom EM-STOP
%MX160077	DF-M TankRoom EM-STOP
%MX160078	DF-1 FILTER ROOM EM-STOP
%MX160079	DF-M FILTER ROOM EM-STOP
%MX160080	MOGAS FILTER ROOM EM-STOP
%MX160081	DRAIN TANK1 EM STOP (LOCAL)
%MX160082	DRAIN TANK2 EM STOP (LOCAL)
%MX160129	DRAIN PIMP 1 ALARM
%MX160130	RP-1 ALARM
%MX160131	RP-2 ALARM
%MX160132	SP-1 ALARM
%MX160133	RP-3 ALARM
%MX160134	RP-4 ALARM
%MX160135	SP-2 ALARM
%MX160136	RP-9 ALARM
%MX160137	RP-10 ALARM
%MX160138	RP-11 ALARM
%MX160139	RP-12 ALARM
%MX160140	RP-7 ALARM
%MX160141	RP-8 ALARM
%MX160142	SUMP PUMP 4 ALARM
%MX160143	RP-13 ALARM
%MX160144	RP-14 ALARM
%MX160145	RP-5 ALARM
%MX160146	RP-6 ALARM
%MX160147	SUMP PUMP 3 ALARM
%MX160148	RP-15 ALARM
%MX160149	RP-16 ALARM
%MX160150	DRAIN PUMP 2 ALARM
%MX166400	CH0,1 단선검출 ERROR
%MX166401	CH2,3 단선검출 ERROR
%MX166464	CH0,1 단선검출 ERROR
%MX166465	CH2,3 단선검출 ERROR
%MX166528	CH0,1 단선검출 ERROR
%MX166529	CH2,3 단선검출 ERROR
%MX192000	NC
%MX192001	NC
%MX192002	NC
%MX192003	NC
%MX192004	NC
%MX192005	NC
%MX192006	NC
%MX192007	AUTO TOUCH S/W
%MX192008	MANUAL TOUCH S/W
%MX192009	HORN STOP TOUCH S/W
%MX192010	RESET S/W (SCADA)
%MX192011	LAMP TEST TOUCH S/W
%MX192012	NC
%MX192013	NC
%MX192014	NC
%MX192015	NC
%MX192016	NC
%MX192017	NC
%MX192018	NC
%MX192019	NC
%MX192020	NC
%MX192021	NC
%MX192022	NC
%MX192023	NC
%MX192024	NC
%MX192025	NC
%MX192026	NC
%MX192027	NC
%MX192028	NC
%MX192029	NC
%MX192030	NC
%MX192031	출하 압력 PIT-1 선택 TOUCH S/W
%MX192032	출하 압력 PIT-2 선택 TOUCH S/W
%MX192033	출하 유량 FIT-1 선택 TOUCH S/W
%MX192034	출하 유량 FIT-2 선택 TOUCH S/W
%MX192035	NC
%MX192036	NC
%MX192037	NC
%MX192038	NC
%MX192039	NC
%MX192040	NC
%MX192041	NC
%MX192042	NC
%MX192043	NC
%MX192044	NC
%MX192045	NC
%MX192046	NC
%MX192047	NC
%MX192048	NC
%MX192049	NC
%MX192050	NC
%MX192051	NC
%MX192052	NC
%MX192053	NC
%MX192054	NC
%MX192055	NC
%MX192056	NC
%MX192057	NC
%MX192058	NC
%MX192059	NC
%MX192060	NC
%MX192061	NC
%MX192062	NC
%MX192063	NC
%MX192064	NC
%MX192065	NC
%MX192066	NC
%MX192067	NC
%MX192068	NC
%MX192069	NC
%MX192070	NC
%MX192071	NC
%MX192072	NC
%MX192073	NC
%MX192074	NC
%MX192075	NC
%MX192076	NC
%MX192077	NC
%MX192640	NC
%MX192641	NC
%MX192642	NC
%MX192643	NC
%MX192644	NC
%MX192645	NC
%MX192646	NC
%MX192647	NC
%MX192648	NC
%MX192649	DP-01 RUN S/W (SCADA)
%MX192650	DF-1 DRAIN PUMP STOP S/W (SCADA)
%MX192651	DF-1 DRAIN TANK AUTO TOUCH S/W
%MX192652	DF-1 DRAIN TANK MANU TOUCH S/W
%MX192653	NC
%MX192654	NC
%MX192655	DF-1A FAN ON S/W (SCADA)
%MX192656	DF-1A FAN OFF TOUCH S/W
%MX192657	DF-1A HLVD ON S/W (SCADA)
%MX192658	DF-1A HLVD OFF TOUCH S/W
%MX192659	NC
%MX192660	NC
%MX192661	NC
%MX192662	RP-1 RUN S/W (SCADA)
%MX192663	RP-1 STOP S/W (SCADA)
%MX192664	NC
%MX192665	NC
%MX192666	NC
%MX192667	DF-1B RP-2 RUN S/W (SCADA)
%MX192668	RP-2 STOP S/W (SCADA)
%MX192669	NC
%MX192670	NC
%MX192671	NC
%MX192672	SP-1 RUN S/W (SCADA)
%MX192673	SP-1 STOP S/W (SCADA)
%MX192674	NC
%MX192675	NC
%MX192676	NC
%MX192677	NC
%MX192678	NC
%MX192679	NC
%MX192680	NC
%MX192681	NC
%MX192682	NC
%MX192683	NC
%MX192684	NC
%MX192685	NC
%MX192686	NC
%MX192687	NC
%MX192688	NC
%MX192689	NC
%MX192690	DF-1 PUMP 선택 1차 RP-01 TOOUCH S/W
%MX192691	DF-1 PUMP 선택 1차 RP-02 TOOUCH S/W
%MX192692	DF-1 PUMP 선택 1차 RP-03 TOOUCH S/W
%MX192693	DF-1 PUMP 선택 1차 RP-04 TOOUCH S/W
%MX192694	DF-1 PUMP 선택 2차 RP-01 TOOUCH S/W
%MX192695	DF-1 PUMP 선택 2차 RP-02 TOOUCH S/W
%MX192696	DF-1 PUMP 선택 2차 RP-03 TOOUCH S/W
%MX192697	DF-1 PUMP 선택 2차 RP-04 TOOUCH S/W
%MX192698	NC
%MX193280	DF-1B FAN ON S/W (TO SCADA)
%MX193281	DF-1B FAN OFF TOUCH S/W
%MX193282	DF-1B HLVD ON S/W (SCADA)
%MX193283	DF-1B HLVD OFF TOUCH S/W
%MX193284	NC
%MX193285	NC
%MX193286	NC
%MX193287	DF-1A RP-3 RUN S/W (SCADA)
%MX193288	DF-1A RP-3 STOP S/W (SCADA)
%MX193289	NC
%MX193290	NC
%MX193291	NC
%MX193292	DF-1A RP-4 RUN S/W (SCADA)
%MX193293	RP-4 STOP S/W (SCADA)
%MX193294	NC
%MX193295	NC
%MX193296	NC
%MX193297	DF-1A SP-2 RUN S/W (SCADA)
%MX193298	SP-2 STOP S/W (SCADA)
%MX193299	NC
%MX193304	NC
%MX193305	NC
%MX193306	NC
%MX193307	NC
%MX193308	NC
%MX193309	NC
%MX193310	NC
%MX193311	NC
%MX193312	NC
%MX193313	NC
%MX193314	NC
%MX193315	NC
%MX193316	NC
%MX193317	RP-9 RUN S/W (SCADA)
%MX193318	RP-9 STOP S/W (SCADA)
%MX193319	NC
%MX193320	NC
%MX193321	NC
%MX193322	RP-10 RUN S/W (SCADA)
%MX193323	RP-10 STOP S/W (SCADA)
%MX193324	NC
%MX193325	NC
%MX193326	NC
%MX193327	RP-11 RUN S/W (SCADA)
%MX193328	RP-11 STOP S/W (SCADA)
%MX193329	NC
%MX193330	NC
%MX193331	NC
%MX193332	DF-1 UNLOADING PUMP RP-12 RUN S/W (SCADA)
%MX193333	RP-12 STOP S/W (SCADA)
%MX193334	NC
%MX193920	DF-M 출하 압력 PIT-3 선택 TOUCH S/W
%MX193921	DF-M 출하 압력 PIT-4 선택 TOUCH S/W
%MX193922	DF-M 출하 유량 FIT-3 선택 TOUCH S/W
%MX193923	DF-M 출하 유량 FIT-4 선택 TOUCH S/W
%MX193924	NC
%MX193925	NC
%MX193926	NC
%MX193927	NC
%MX193928	NC
%MX193929	NC
%MX193930	NC
%MX193931	NC
%MX193932	NC
%MX193933	NC
%MX193934	NC
%MX193935	NC
%MX193936	NC
%MX193937	NC
%MX193938	DF-M PUMP 선택 RP-07 TOOUCH S/W (SCADA)
%MX193939	DF-M PUMP 선택 RP-08 TOOUCH S/W (SCADA)
%MX193940	NC
%MX193941	NC
%MX193942	NC
%MX193943	NC
%MX193944	NC
%MX193945	DF-M UNLOADING PUMP RP-13 RUN S/W (SCADA)
%MX193946	DF-M UNLOADING PUMP RP-13 STOP S/W (SCADA)
%MX193947	NC
%MX193948	NC
%MX193949	NC
%MX193950	DF-M UNLOADING PUMP RP-14 RUN S/W (SCADA)
%MX193951	DF-M UNLOADING PUMP RP-14 STOP S/W (SCADA)
%MX193952	NC
%MX193953	DF-M FAN S/W (SCADA)
%MX193954	DF-M FAN OFF TOUCH S/W
%MX193955	NC
%MX193956	NC
%MX193957	NC
%MX193958	NC
%MX193959	DF-M RP-7 RUN S/W (SCADA)
%MX193960	DF-M RP-7 STOP S/W (SCADA)
%MX193961	NC
%MX193962	NC
%MX193963	NC
%MX193964	DF-M RP-8 RUN S/W (SCADA)
%MX193965	DF-M RP-8 STOP S/W (SCADA)
%MX193966	NC
%MX193967	NC
%MX193968	NC
%MX193969	DF-M SUMP PUMP-4 RUN S/W (SCADA)
%MX193970	SP-4 STOP S/W (SCADA)
%MX193971	NC
%MX193975	NC
%MX193976	NC
%MX193977	NC
%MX193978	NC
%MX193979	NC
%MX193980	NC
%MX193981	NC
%MX193982	NC
%MX193983	NC
%MX193984	NC
%MX193985	NC
%MX193986	NC
%MX193987	NC
%MX194560	MOGAS 출하 압력 PIT-5 선택 TOUCH S/W
%MX194561	MOGAS 출하 압력 PIT-6 선택 TOUCH S/W
%MX194562	MOGAS 출하 유량 FIT-5 선택 TOUCH S/W
%MX194563	MOGAS 출하 유량 FIT-6 선택 TOUCH S/W
%MX194564	NC
%MX194565	NC
%MX194566	NC
%MX194567	NC
%MX194568	NC
%MX194569	NC
%MX194570	NC
%MX194571	NC
%MX194572	NC
%MX194573	NC
%MX194574	NC
%MX194575	NC
%MX194576	NC
%MX194577	NC
%MX194578	NC
%MX194579	MOGAS 출하펌프 선택 RP-05 TOOUCH S/W
%MX194580	MOGAS 출하펌프 선택 RP-06 TOOUCH S/W
%MX194581	NC
%MX194582	NC
%MX194583	NC
%MX194584	NC
%MX194585	NC
%MX194586	MOGAS UNLOADING PUMP RP-15 RUN S/W (SCADA)
%MX194587	MOGAS UNLOADING PUMP RP-15 STOP S/W (SCADA)
%MX194588	NC
%MX194589	NC
%MX194590	NC
%MX194591	MOGAS UNLOADING PUMP RP-16 RUN S/W (SCADA)
%MX194592	MOGAS UNLOADING PUMP RP-16 STOP S/W (SCADA)
%MX194593	NC
%MX194594	MOGAS FAN ON S/W (SCADA)
%MX194595	MOGAS FAN OFF TOUCH S/W
%MX194596	NC
%MX194597	NC
%MX194598	NC
%MX194599	NC
%MX194600	MOGAS RP-5 RUN S/W (SCADA)
%MX194601	MOGAS RP-5 STOP S/W (SCADA)
%MX194602	NC
%MX194603	NC
%MX194604	NC
%MX194605	MOGAS RP-6 RUN S/W (SCADA)
%MX194606	MOGAS RP-6 STOP S/W (SCADA)
%MX194607	NC
%MX194608	NC
%MX194609	NC
%MX194610	MOGAS SUMP PUMP-3 RUN S/W (SCADA)
%MX194611	MOGAS SUMP PUMP-3 STOP S/W (SCADA)
%MX194612	NC
%MX194617	NC
%MX194618	NC
%MX194619	NC
%MX194620	NC
%MX194621	NC
%MX194622	NC
%MX194623	NC
%MX194624	NC
%MX194625	NC
%MX194626	NC
%MX194627	NC
%MX194628	NC
%MX194629	NC
%MX194630	NC
%MX194631	NC
%MX194632	NC
%MX194633	NC
%MX194634	NC
%MX194635	NC
%MX194636	NC
%MX194637	MOGAS DRAIN PUMP RUN TOUCH S/W
%MX194638	DP-02 RUN S/W (SCADA)
%MX194639	MOGAS DRAIN TANK STOP S/W (SCADA)
%MX194640	MOGAS DRAIN TANK MANU TOUCH S/W
%MX196481	DTK1 LEVEL HH(TO SCADA)
%MX196482	DTK1 LEVEL H(TO SCADA)
%MX196483	DTK1 LEVEL LL(TO SCADA)
%MX196484	DTK1 LEVEL L(TO SCADA)
%MX196491	DF-1A LEVEL HH(TO SCADA)
%MX196492	DF-1A LEVEL H(TO SCADA)
%MX196493	DF-1A LEVEL LL(TO SCADA)
%MX196494	DF-1A LEVEL L(TO SCADA)
%MX196501	DF-1B LEVEL HH(TO SCADA)
%MX196502	DF-1B LEVEL H(TO SCADA)
%MX196503	DF-1B LEVEL LL(TO SCADA)
%MX196504	DF-1B LEVEL L(TO SCADA)
%MX196511	DF-M LEVEL HH(TO SCADA)
%MX196512	DF-M LEVEL H(TO SCADA)
%MX196513	DF-M LEVEL LL(TO SCADA)
%MX196514	DF-M LEVEL L(TO SCADA)
%MX196521	MOGAS LEVEL HH(TO SCADA)
%MX196522	MOGAS LEVEL H(TO SCADA)
%MX196523	MOGAS LEVEL LL(TO SCADA)
%MX196524	MOGAS LEVEL L(TO SCADA)
%MX196531	DTK2 LEVEL HH(TO SCADA)
%MX196532	DTK2 LEVEL H(TO SCADA)
%MX196533	DTK2 LEVEL LL(TO SCADA)
%MX196534	DTK2 LEVEL L(TO SCADA)
%MX198400	ALARM RESET
%MX198401	NC
%MX198402	NC
%MX198403	NC
%MX198404	NC
%MX198405	NC
%MX198406	NC
%MX198407	NC
%MX198408	NC
%MX198409	NC
%MX198410	RP01 FLOW S/W
%MX198411	RP02 FLOW S/W
%MX198412	RP03 FLOW S/W
%MX198413	RP04 FLOW S/W
%MX198414	RP05 FLOW S/W
%MX198415	RP06 FLOW S/W
%MX198416	RP07 FLOW S/W
%MX198417	RP08 FLOW S/W
%MX198418	RP09 FLOW S/W
%MX198419	RP10 FLOW S/W
%MX198420	RP11 FLOW S/W
%MX198421	RP12 FLOW S/W
%MX198422	RP13 FLOW S/W
%MX198423	RP14 FLOW S/W
%MX198424	RP15 FLOW S/W
%MX198425	RP16 FLOW S/W
%MX198426	SP01 FLOW S/W
%MX198427	SP02 FLOW S/W
%MX198428	SP03 FLOW S/W
%MX198429	SP04 FLOW S/W
%MX198430	DP01 FLOW S/W
%MX198431	DP02 FLOW S/W
%MX198432	NC
%MX198433	NC
%MX198434	NC
%MX198435	NC
%MX198436	NC
%MX198437	NC
%MX198438	NC
%MX198439	NC
%MX198440	NC
%MX198441	NC
%MX198442	NC
%MX198443	NC
%MX198444	NC
%MX198445	NC
%MX198446	NC
%MX198447	NC
%MX198448	NC
%MX198449	NC
%MX198450	NC
%MX198451	NC
%MX198452	NC
%MX198453	NC
%MX198454	NC
%MX198455	NC
%MX198456	NC
%MX198457	NC
%MX198458	NC
%MX198459	NC
%MX198460	NC
%MX198461	NC
%MX198462	NC
%MX198463	NC
%MX199040	NC
%MX199041	NC
%MX199042	NC
%MX199043	NC
%MX199044	NC
%MX199045	NC
%MX199046	NC
%MX199047	NC
%MX199048	NC
%MX199049	NC
%MX199050	NC
%MX199051	NC
%MX199052	NC
%MX199053	NC
%MX199054	NC
%MX199055	NC
%MX199056	NC
%MX199057	NC
%MX199058	NC
%MX199059	NC
%MX199060	NC
%MX199061	NC
%MX199062	NC
%MX199063	NC
%MX199064	NC
%MX199065	NC
%MX199066	NC
%MX199067	NC
%MX199068	NC
%MX199069	NC
%MX199070	NC
%MX199071	NC
%MX199072	NC
%MX199073	NC
%MX199074	NC
%MX199075	NC
%MX199076	NC
%MX199077	NC
%MX199078	NC
%MX199079	NC
%MX199080	NC
%MX199081	NC
%MX199082	NC
%MX199083	NC
%MX199084	NC
%MX199085	NC
%MX199086	NC
%MX199087	NC
%MX199088	NC
%MX199089	NC
%MX199090	NC
%MX199091	NC
%MX199092	NC
%MX199093	NC
%MX199094	NC
%MX199095	NC
%MX199096	NC
%MX199097	NC
%MX199098	NC
%MX199099	NC
%MX199100	NC
%MX199101	NC
%MX199102	NC
%MX199103	NC
%MX199680	NC
%MX199681	NC
%MX199682	NC
%MX199683	NC
%MX199684	NC
%MX199685	NC
%MX224000	LOCAL(MCC)선택 TOUCH LAMP
%MX224001	REMOTE(PLC)선택 TOUCH LAMP
%MX224002	SCADA 선택 TOUCH LAMP
%MX224003	PANEL 선택 TOUCH LAMP
%MX224004	UPS ON LAMP
%MX224005	UPS TROUBLE TOUCH LAMP
%MX224006	MCC ON LAMP
%MX224007	AUTO TOUCH LAMP
%MX224008	MANUAL TOUCH LAMP
%MX224009	HORN STOP TOUCH LAMP
%MX224010	RESET TOUCH LAMP
%MX224011	LAMP TEST TOUCH LAMP
%MX224012	NC
%MX224013	NC
%MX224014	NC
%MX224015	NC
%MX224016	EV-1 TOUCH LAMP
%MX224017	EV-2 TOUCH LAMP
%MX224018	BPCV TOUCH LAMP
%MX224019	NC
%MX224020	CONTROL EM-STOP TOUCH LAMP
%MX224021	DF-1A TANK EM-STOP TOUCH LAMP
%MX224022	DF-1B TANK EM-STOP TOUCH LAMP
%MX224023	DRAIN TANK EM-STOP TOUCH LAMP
%MX224024	FILTER ROOM EM-STOP TOUCH LAMP
%MX224025	대량 주유대 1 EM-STOP TOUCH LAMP
%MX224026	대량 주유대 2 EM-STOP TOUCH LAMP
%MX224027	대량 주유대 3 EM-STOP TOUCH LAMP
%MX224028	대량 주유대 4 EM-STOP TOUCH LAMP
%MX224029	포장 주유대 EM-STOP TOUCH LAMP
%MX224030	NC
%MX224031	출하 압력 PIT-1 선택 TOUCH LAMP
%MX224032	출하 압력 PIT-2 선택 TOUCH LAMP
%MX224033	출하 유량 FIT-1 선택 TOUCH LAMP
%MX224034	출하 유량 FIT-2 선택 TOUCH LAMP
%MX224035	출하 압력 PIT-1 TROUBLE TOUCH LAMP
%MX224036	출하 압력 PIT-2 TROUBLE TOUCH LAMP
%MX224037	출하 유량 FIT-1 TROUBLE TOUCH LAMP
%MX224038	출하 유량 FIT-2 TROUBLE TOUCH LAMP
%MX224039	NC
%MX224040	PLC1 RUN LAMP
%MX224041	PLC1 STANDBY LAMP
%MX224042	PLC1 TROUBLE LAMP
%MX224043	PLC2 RUN LAMP
%MX224044	PLC2 STANDBY LAMP
%MX224045	PLC2 TROUBLE LAMP
%MX224046	NC
%MX224047	DF-1B RP-1 전시 비상스위치 ON
%MX224048	DF-1B SP-1 전시 비상스위치 ON
%MX224049	DF-1B RP-2 전시 비상스위치 ON
%MX224050	DF-1A RP-3 전시 비상스위치 ON
%MX224051	DF-1A SP-2 전시 비상스위치 ON
%MX224052	DF-1A RP-4 전시 비상스위치 ON
%MX224053	DF-1 DP-01 전시 비상스위치 ON
%MX224054	DF-1 UNLODING PUMP RP-9 전시 비상스위치 ON
%MX224055	DF-1 UNLODING PUMP RP-10 전시 비상스위치 ON
%MX224056	DF-1 UNLODING PUMP RP-11 전시 비상스위치 ON
%MX224057	DF-1 UNLODING PUMP RP-12 전시 비상스위치 ON
%MX224058	DF-M RP-7 전시 비상스위치 ON
%MX224059	DF-M SP-4 전시 비상스위치 ON
%MX224060	DF-M RP-8 전시 비상스위치 ON
%MX224061	DF-M UNLODING PUMP RP-13 전시 비상스위치 ON
%MX224062	DF-M UNLODING PUMP RP-14 전시 비상스위치 ON
%MX224063	MOGAS RP-5 전시 비상스위치 ON
%MX224064	MOGAS SP-3 전시 비상스위치 ON
%MX224065	MOGAS RP-6 전시 비상스위치 ON
%MX224066	MOGAS DP-02 전시 비상스위치 ON
%MX224067	MOGAS UNLODING PUMP RP-15 전시 비상스위치 ON
%MX224068	MOGAS UNLODING PUMP RP-16 전시 비상스위치 ON
%MX224069	포장 주유대 DF-1 스위치-ON 신호
%MX224070	대량 주유대 DF1-1 스위치-ON 신호
%MX224071	대량 주유대 DF1-2 스위치-ON 신호
%MX224072	대량 주유대 DF1-3 스위치-ON 신호
%MX224073	대량 주유대 DF1-4 스위치-ON 신호
%MX224640	DF-1 DRAIN PUMP HLVD CLOSE TOUCH LAMP
%MX224641	NC
%MX224642	NC
%MX224643	NC
%MX224644	NC
%MX224645	DF-1 DRAIN TANK LEVEL TROUBLE TOUCH LAMP
%MX224646	NC
%MX224647	DF-1 DRAIN PUMP TROUBLE TOUCH LAMP
%MX224648	DF-1 DRAIN PUMP LOCAL TOUCH LAMP
%MX224649	DF-1 DRAIN PUMP RUN TOUCH LAMP
%MX224650	DF-1 DRAIN PUMP STOP TOUCH LAMP
%MX224651	DF-1 DRAIN TANK AUTO TOUCH LAMP
%MX224652	DF-1 DRAIN TANK MANU TOUCH LAMP
%MX224653	NC
%MX224654	NC
%MX224655	DF-1A FAN ON LAMP (TO SCADA)
%MX224656	DF-1A FAN OFF TOUCH LAMP
%MX224657	DF-1A HLV ON LAMP
%MX224658	DF-1A HLVD OFF TOUCH LAMP
%MX224659	DF-1A 개별TANK STOP TOUCH LAMP
%MX224660	DF-1B RP-1 TROUBLE TOUCH LAMP
%MX224661	DF-1B RP-1 LOCAL TOUCH LAMP
%MX224662	DF-1B RP-1 RUN TOUCH LAMP
%MX224663	DF-1B RP-1 STOP TOUCH LAMP
%MX224664	NC
%MX224665	DF-1B RP-2 TROUBLE TOUCH LAMP
%MX224666	DF-1B RP-2 LOCAL TOUCH LAMP
%MX224667	DF-1B RP-2 RUN TOUCH LAMP
%MX224668	DF-1B RP-2 STOP TOUCH LAMP
%MX224669	NC
%MX224670	DF-1B SP-1 TROUBLE TOUCH LAMP
%MX224671	DF-1B SP-1 LOCAL TOUCH LAMP
%MX224672	DF-1B SP-1 RUN TOUCH LAMP
%MX224673	DF-1B SP-1 STOP TOUCH LAMP
%MX224674	NC
%MX224679	DF-1A TANK LEVEL TROUBLE TOUCH LAMP
%MX224680	NC
%MX224681	DF-1A 누유 TOUCH LAMP
%MX224682	DF-1A 소화피트 1 누유 TOUCH LAMP
%MX224683	DF-1A 소화피트 2 누수 TOUCH LAMP
%MX224684	DF-1A 소화피트 2 누유 TOUCH LAMP
%MX224685	DF-1A 소화피트 3 누수 TOUCH LAMP
%MX224686	DF-1A 소화피트 3 누유 TOUCH LAMP
%MX224687	DF-1A 소화피트 4 누수 TOUCH LAMP
%MX224688	DF-1A 소화피트 4 누유 TOUCH LAMP
%MX224689	NC
%MX224690	DF-1 PUMP 선택 1차 RP-01 TOOUCH LAMP
%MX224691	DF-1 PUMP 선택 1차 RP-02 TOOUCH LAMP
%MX224692	DF-1 PUMP 선택 1차 RP-03 TOOUCH LAMP
%MX224693	DF-1 PUMP 선택 1차 RP-04 TOOUCH LAMP
%MX224694	DF-1 PUMP 선택 2차 RP-01 TOOUCH LAMP
%MX224695	DF-1 PUMP 선택 2차 RP-02 TOOUCH LAMP
%MX224696	DF-1 PUMP 선택 2차 RP-03 TOOUCH LAMP
%MX224697	DF-1 PUMP 선택 2차 RP-04 TOOUCH LAMP
%MX224698	NC
%MX225280	DF-1B FAN ON LAMP (TO SCADA)
%MX225281	DF-1B FAN OFF TOUCH LAMP
%MX225282	DF-1B HLVD ON LAMP
%MX225283	DF-1B HLVD OFF TOUCH LAMP
%MX225284	DF-1B 개별TANK STOP TOUCH LAMP
%MX225285	DF-1A RP-3 TROUBLE TOUCH LAMP
%MX225286	DF-1A RP-3 LOCAL TOUCH LAMP
%MX225287	DF-1A RP-3 RUN TOUCH LAMP
%MX225288	DF-1A RP-3 STOP TOUCH LAMP
%MX225289	NC
%MX225290	DF-1A RP-4 TROUBLE TOUCH LAMP
%MX225291	DF-1A RP-4 LOCAL TOUCH LAMP
%MX225292	DF-1A RP-4 RUN TOUCH LAMP
%MX225293	DF-1A RP-4 STOP TOUCH LAMP
%MX225294	NC
%MX225295	DF-1A SP-2 TROUBLE TOUCH LAMP
%MX225296	DF-1A SP-2 LOCAL TOUCH LAMP
%MX225297	DF-1A SP-2 RUN TOUCH LAMP
%MX225298	DF-1A SP-2 STOP TOUCH LAMP
%MX225299	NC
%MX225304	DF-1B TANK LEVEL TROUBLE TOUCH LAMP
%MX225305	NC
%MX225306	DF-1B 누유 TOUCH LAMP
%MX225307	DF-1B 소화피트 1 누유 TOUCH LAMP
%MX225308	DF-1B 소화피트 2 누수 TOUCH LAMP
%MX225309	DF-1B 소화피트 2 누유 TOUCH LAMP
%MX225310	DF-1B 소화피트 3 누수 TOUCH LAMP
%MX225311	DF-1B 소화피트 3 누유 TOUCH LAMP
%MX225312	DF-1B 소화피트 4 누수 TOUCH LAMP
%MX225313	DF-1B 소화피트 4 누유 TOUCH LAMP
%MX225314	NC
%MX225315	DF-1 UNLOADING PUMP RP-9 TROUBLE TOUCH LAMP
%MX225316	DF-1 UNLOADING PUMP RP-9 LOCAL TOUCH LAMP
%MX225317	DF-1 UNLOADING PUMP RP-9 RUN TOUCH LAMP
%MX225318	DF-1 UNLOADING PUMP RP-9 STOP TOUCH LAMP
%MX225319	NC
%MX225320	DF-1 UNLOADING PUMP RP-10 TROUBLE TOUCH LAMP
%MX225321	DF-1 UNLOADING PUMP RP-10 LOCAL TOUCH LAMP
%MX225322	DF-1 UNLOADING PUMP RP-10 RUN TOUCH LAMP
%MX225323	DF-1 UNLOADING PUMP RP-10 STOP TOUCH LAMP
%MX225324	NC
%MX225325	DF-1 UNLOADING PUMP RP-11 TROUBLE TOUCH LAMP
%MX225326	DF-1 UNLOADING PUMP RP-11 LOCAL TOUCH LAMP
%MX225327	DF-1 UNLOADING PUMP RP-11 RUN TOUCH LAMP
%MX225328	DF-1 UNLOADING PUMP RP-11 STOP TOUCH LAMP
%MX225329	NC
%MX225330	DF-1 UNLOADING PUMP RP-12 TROUBLE TOUCH LAMP
%MX225331	DF-1 UNLOADING PUMP RP-12 LOCAL TOUCH LAMP
%MX225332	DF-1 UNLOADING PUMP RP-12 RUN TOUCH LAMP
%MX225333	DF-1 UNLOADING PUMP RP-12 STOP TOUCH LAMP
%MX225334	NC
%MX225920	DF-M 출하 압력 PIT-3 선택 TOUCH LAMP
%MX225921	DF-M 출하 압력 PIT-4 선택 TOUCH LAMP
%MX225922	DF-M 출하 유량 FIT-3 선택 TOUCH LAMP
%MX225923	DF-M 출하 유량 FIT-4 선택 TOUCH LAMP
%MX225924	DF-M 출하 압력 PIT-3 TROUBLE TOUCH LAMP
%MX225925	DF-M 출하 압력 PIT-4 TROUBLE TOUCH LAMP
%MX225926	DF-M 출하 유량 FIT-3 TROUBLE TOUCH LAMP
%MX225927	DF-M 출하 유량 FIT-4 TROUBLE TOUCH LAMP
%MX225928	NC
%MX225929	DF-M EV-3 TOUCH LAMP
%MX225930	DF-M EV-4 TOUCH LAMP
%MX225931	DF-M BPCV TOUCH LAMP
%MX225932	NC
%MX225933	DF-M FILTER ROOM EM-STOP TOUCH LAMP
%MX225934	DF-M TANK EM-STOP TOUCH LAMP
%MX225935	DF-M 대량 주유대 EM-STOP TOUCH LAMP
%MX225936	DF-M 포장주유대 EM-STOP TOUCH LAMP
%MX225937	NC
%MX225938	DF-M 출하펌프 선택 RP-07 TOUCH LAMP
%MX225939	DF-M 출하펌프 선택 RP-08 TOUCH LAMP
%MX225940	NC
%MX225941	NC
%MX225942	NC
%MX225943	DF-M UNLOADING PUMP RP-13 TROUBLE TOUCH LAMP
%MX225944	DF-M UNLOADING PUMP RP-13 LOCAL TOUCH LAMP
%MX225945	DF-M UNLOADING PUMP RP-13 RUN TOUCH LAMP
%MX225946	DF-M UNLOADING PUMP RP-13 STOP TOUCH LAMP
%MX225947	NC
%MX225948	DF-M UNLOADING PUMP RP-14 TROUBLE TOUCH LAMP
%MX225949	DF-M UNLOADING PUMP RP-14 LOCAL TOUCH LAMP
%MX225950	DF-M UNLOADING PUMP RP-14 RUN TOUCH LAMP
%MX225951	DF-M UNLOADING PUMP RP-14 STOP TOUCH LAMP
%MX225952	NC
%MX225953	DF-M FAN ON LAMP(TO SCADA)
%MX225954	DF-M FAN OFF TOUCH LAMP
%MX225955	NC
%MX225956	DF-M 개별TANK STOP TOUCH LAMP
%MX225957	RP-7 TROUBLE LAMP [SCADA]
%MX225958	DF-M RP-7 LOCAL TOUCH LAMP
%MX225959	DF-M RP-7 RUN TOUCH LAMP
%MX225960	DF-M RP-7 STOP TOUCH LAMP
%MX225961	NC
%MX225962	DF-M RP-8 TROUBLE TOUCH LAMP
%MX225963	DF-M RP-8 LOCAL TOUCH LAMP
%MX225964	DF-M RP-8 RUN TOUCH LAMP
%MX225965	DF-M RP-8 STOP TOUCH LAMP
%MX225966	NC
%MX225967	DF-M SUMP PUMP-4 TROUBLE TOUCH LAMP
%MX225968	DF-M SUMP PUMP-4 LOCAL TOUCH LAMP
%MX225969	DF-M SUMP PUMP-4 RUN TOUCH LAMP
%MX225970	DF-M SUMP PUMP-4 STOP TOUCH LAMP
%MX225971	NC
%MX225975	NC
%MX225976	DF-M TANK LEVEL TROUBLE TOUCH LAMP
%MX225977	NC
%MX225978	DF-M 누유 TOUCH LAMP
%MX225979	DF-M 소화피트 1 누유 TOUCH LAMP
%MX225980	DF-M 소화피트 2 누수 TOUCH LAMP
%MX225981	DF-M 소화피트 2 누유 TOUCH LAMP
%MX225982	DF-M 소화피트 3 누수 TOUCH LAMP
%MX225983	DF-M 소화피트 3 누유 TOUCH LAMP
%MX225984	DF-M 소화피트 4 누수 TOUCH LAMP
%MX225985	DF-M 소화피트 4 누유 TOUCH LAMP
%MX225986	포장 주유대 DF-M LOCAL S/W ON
%MX225987	대량 주유대 DF-M LOCAL S/W ON
%MX226560	MOGAS 출하 압력 PIT-5 선택 TOUCH LAMP
%MX226561	MOGAS 출하 압력 PIT-6 선택 TOUCH LAMP
%MX226562	MOGAS 출하 유량 FIT-5 선택 TOUCH LAMP
%MX226563	MOGAS 출하 유량 FIT-6 선택 TOUCH LAMP
%MX226564	MOGAS 출하 압력 PIT-5 TROUBLE TOUCH LAMP
%MX226565	MOGAS 출하 압력 PIT-6 TROUBLE TOUCH LAMP
%MX226566	MOGAS 출하 유량 FIT-5 TROUBLE TOUCH LAMP
%MX226567	MOGAS 출하 유량 FIT-6 TROUBLE TOUCH LAMP
%MX226568	NC
%MX226569	MOGAS EV-5 TOUCH LAMP
%MX226570	MOGAS EV-6 TOUCH LAMP
%MX226571	MOGAS BPCV TOUCH LAMP
%MX226572	NC
%MX226573	MOGAS FILTER ROOM EM-STOP TOUCH LAMP
%MX226574	MOGAS TANK EM-STOP TOUCH LAMP
%MX226575	MOGAS 대량 주유대 EM-STOP TOUCH LAMP
%MX226576	MOGAS 포장주유대 EM-STOP TOUCH LAMP
%MX226577	MOGAS DRAIN TANK EM-STOP TOUCH LAMP
%MX226578	NC
%MX226579	MOGAS 출하펌프 선택 RP-05 TOUCH LAMP
%MX226580	MOGAS 출하펌프 선택 RP-06 TOUCH LAMP
%MX226581	NC
%MX226582	NC
%MX226583	NC
%MX226584	MOGAS UNLOADING PUMP RP-15 TROUBLE TOUCH LAMP
%MX226585	MOGAS UNLOADING PUMP RP-15 LOCAL TOUCH LAMP
%MX226586	MOGAS UNLOADING PUMP RP-15 RUN TOUCH LAMP
%MX226587	MOGAS UNLOADING PUMP RP-15 STOP TOUCH LAMP
%MX226588	NC
%MX226589	MOGAS UNLOADING PUMP RP-16 TROUBLE TOUCH LAMP
%MX226590	MOGAS UNLOADING PUMP RP-16 LOCAL TOUCH LAMP
%MX226591	MOGAS UNLOADING PUMP RP-16 RUN TOUCH LAMP
%MX226592	MOGAS UNLOADING PUMP RP-16 STOP TOUCH LAMP
%MX226593	NC
%MX226594	MOGAS FAN ON LAMP(TO SCADA)
%MX226595	MOGAS FAN OFF TOUCH LAMP
%MX226596	NC
%MX226597	MOGAS 개별TANK STOP TOUCH LAMP
%MX226598	MOGAS RP-5 TROUBLE TOUCH LAMP
%MX226599	MOGAS RP-5 LOCAL TOUCH LAMP
%MX226600	MOGAS RP-5 RUN TOUCH LAMP
%MX226601	MOGAS RP-5 STOP TOUCH LAMP
%MX226602	NC
%MX226603	MOGAS RP-6 TROUBLE TOUCH LAMP
%MX226604	MOGAS RP-6 LOCAL TOUCH LAMP
%MX226605	MOGAS RP-6 RUN TOUCH LAMP
%MX226606	MOGAS RP-6 STOP TOUCH LAMP
%MX226607	NC
%MX226608	MOGAS SUMP PUMP-3 TROUBLE TOUCH LAMP
%MX226609	MOGAS SUMP PUMP-3 LOCAL TOUCH LAMP
%MX226610	MOGAS SUMP PUMP-3 RUN TOUCH LAMP
%MX226611	SMOGAS UM PUMP-3 STOP TOUCH LAMP
%MX226612	NC
%MX226617	MOGAS TANK LEVEL TROUBLE TOUCH LAMP
%MX226618	NC
%MX226619	MOGAS 누유 TOUCH LAMP
%MX226620	MOGAS 소화피트 1 누유 TOUCH LAMP
%MX226621	MOGAS 소화피트 2 누수 TOUCH LAMP
%MX226622	MOGAS 소화피트 2 누유 TOUCH LAMP
%MX226623	MOGAS 소화피트 3 누수 TOUCH LAMP
%MX226624	MOGAS 소화피트 3 누유 TOUCH LAMP
%MX226625	MOGAS 소화피트 4 누수 TOUCH LAMP
%MX226626	MOGAS 소화피트 4 누유 TOUCH LAMP
%MX226627	대량 주유대 MOGAS 스위치-ON 신호
%MX226628	MOGAS DRAIN PUMP HLVD CLOSE TOUCH LAMP
%MX226629	NC
%MX226630	NC
%MX226631	NC
%MX226632	NC
%MX226633	MOGAS DRAIN TANK LEVEL TROUBLE TOUCH LAMP
%MX226634	MOGAS DRAIN TANK LEVEL TROUBLE
%MX226635	MOGAS DRAIN PUMP TROUBLE TOUCH LAMP
%MX226636	MOGAS DRAIN PUMP TROUBLE TOUCH LAMP
%MX226637	MOGAS DRAIN PUMP LOCAL TOUCH LAMP
%MX226638	MOGAS DRAIN PUMP RUN TOUCH LAMP
%MX226639	MOGAS DRAIN TANK AUTO TOUCH LAMP
%MX226640	MOGAS DRAIN TANK AUTO TOUCH LAMP
%MX226641	MOGAS DRAIN TANK MANU TOUCH LAMP
%MX226643	MOGAS 포장주유대 LOCAL S/W ON
%MX228481	DF-1 DRAIN TANK LEVEL HH TOUCH LAMP
%MX228482	DF-1 DRAIN TANK LEVEL H TOUCH LAMP
%MX228483	DF-1 DRAIN TANK LEVEL LL TOUCH LAMP
%MX228484	DF-1 DRAIN TANK LEVEL L TOUCH LAMP
%MX228491	DF-1A TANK LEVEL HH TOUCH LAMP
%MX228492	DF-1A TANK LEVEL H TOUCH LAMP
%MX228493	DF-1A TANK LEVEL LL TOUCH LAMP
%MX228494	DF-1A TANK LEVEL L TOUCH LAMP
%MX228501	DF-1B TANK LEVEL HH TOUCH LAMP
%MX228502	DF-1B TANK LEVEL H TOUCH LAMP
%MX228503	DF-1B TANK LEVEL LL TOUCH LAMP
%MX228504	DF-1B TANK LEVEL L TOUCH LAMP
%MX228511	DF-M TANK LEVEL HH TOUCH LAMP
%MX228512	DF-M TANK LEVEL H TOUCH LAMP
%MX228513	DF-M TANK LEVEL LL TOUCH LAMP
%MX228514	DF-M TANK LEVEL L TOUCH LAMP
%MX228521	MOGAS TANK LEVEL HH TOUCH LAMP
%MX228522	MOGAS TANK LEVEL H TOUCH LAMP
%MX228523	MOGAS TANK LEVEL LL TOUCH LAMP
%MX228524	MOGAS TANK LEVEL L TOUCH LAMP
%MX228531	MOGAS DRAIN TANK LEVEL HH TOUCH LAMP
%MX228532	MOGAS DRAIN TANK LEVEL H TOUCH LAMP
%MX228533	MOGAS DRAIN TANK LEVEL LL TOUCH LAMP
%MX228534	MOGAS DRAIN TANK LEVEL L TOUCH LAMP
%MX230400	ALL EM-STOP (TO SCADA)
%MX230401	ALL ALARM
%MX230402	NC
%MX230403	NC
%MX230404	NC
%MX230405	NC
%MX230406	NC
%MX230407	NC
%MX230408	NC
%MX230409	NC
%MX230410	HLV VALVE(TANK) 선택이 안되어 있습니다.
%MX230411	DF-1 출하 PUMP 선택이 안되어 있습니다.
%MX230412	DF-M 출하 PUMP 선택이 안되어 있습니다.
%MX230413	MOGAS 출하 PUMP 선택이 안되어 있습니다.
%MX230414	RP-1 PUMP가 MCC에서 수동 상태입니다.
%MX230415	RP-2 PUMP가 MCC에서 수동 상태입니다.
%MX230416	RP-3 PUMP가 MCC에서 수동 상태입니다.
%MX230417	RP-4 PUMP가 MCC에서 수동 상태입니다.
%MX230418	RP-5 PUMP가 MCC에서 수동 상태입니다.
%MX230419	RP-6 PUMP가 MCC에서 수동 상태입니다.
%MX230420	RP-7 PUMP가 MCC에서 수동 상태입니다.
%MX230421	RP-8 PUMP가 MCC에서 수동 상태입니다.
%MX230422	RP-9 PUMP가 MCC에서 수동 상태입니다.
%MX230423	RP-10 PUMP가 MCC에서 수동 상태입니다.
%MX230424	RP-11 PUMP가 MCC에서 수동 상태입니다.
%MX230425	RP-12 PUMP가 MCC에서 수동 상태입니다.
%MX230426	RP-13 PUMP가 MCC에서 수동 상태입니다.
%MX230427	RP-14 PUMP가 MCC에서 수동 상태입니다.
%MX230428	RP-15 PUMP가 MCC에서 수동 상태입니다.
%MX230429	RP-16 PUMP가 MCC에서 수동 상태입니다.
%MX230430	DF- 1 DRAIN PUMP가 MCC에서 수동 상태입니다. 
%MX230431	MOGAS DRAIN PUMP가 MCC에서 수동 상태입니다.
%MX230432	DF-1A SUMP PUMP 02 가 MCC에서 수동 상태입니다.
%MX230433	DF-1B SUMP PUMP 01 가 MCC에서 수동 상태입니다.
%MX230434	대량 주유대 DF-1-1 번의 스위치 박스 KEY 위치가 OFF 상태입니다
%MX230435	대량 주유대 DF-1-2 번의 스위치 박스 KEY 위치가 OFF 상태입니다
%MX230436	대량 주유대 DF-1-3 번의 스위치 박스 KEY 위치가 OFF 상태입니다
%MX230437	대량 주유대 DF-1-4 번의 스위치 박스 KEY 위치가 OFF 상태입니다
%MX230438	대량 주유대 DF-M 스위치 박스 KEY 위치가 OFF 상태입니다
%MX230439	대량 주유대 MOGAS 스위치 박스 KEY 위치가 OFF 상태입니다
%MX230440	포장 주유대 DF-1 스위치 박스 KEY 위치가 OFF 상태입니다
%MX230441	포장 주유대 DF-M 스위치 박스 KEY 위치가 OFF 상태입니다
%MX230442	포장 주유대 MOGAS 스위치 박스 KEY 위치가 OFF 상태입니다
%MX230443	MOGAS SUMP PUMP 03 가 MCC에서 수동 상태입니다.
%MX230444	DF-M SUMP PUMP 04 가 MCC에서 수동 상태입니다.
%MX230445	NC
%MX230446	NC
%MX230447	NC
%MX230448	NC
%MX230449	NC
%MX230450	NC
%MX230451	NC
%MX230452	NC
%MX230453	NC
%MX230454	NC
%MX230455	NC
%MX230456	NC
%MX230457	NC
%MX230458	NC
%MX230459	NC
%MX230460	NC
%MX230461	NC
%MX230462	NC
%MX230463	NC
%MX230464	UPS ALARM (TO SCADA)
%MX230465	DP-01 INVER&DMPI ALARM
%MX230466	DP-01 MCCB ALARM
%MX230467	DP-01 PUMP 과열 ALARM
%MX230468	DP-01 FLOW ALARM
%MX230469	RP-1 INVER&DMPI ALARM
%MX230470	RP-1 MCCB ALARM
%MX230471	RP-1 PUMP 과열 ALARM
%MX230472	RP-1 FLOW ALARM
%MX230473	RP-2 INVER&DMPI ALARM
%MX230474	RP-2 MCCB ALARM
%MX230475	RP-2 PUMP 과열 ALARM
%MX230476	RP-2 FLOW ALARM
%MX230477	SUMP PUMP 1 INVER&DMPI ALARM
%MX230478	SUMP PUMP 1 MCCB ALARM
%MX230479	SUMP PUMP 1 PUMP 과열 ALARM
%MX230480	SUMP PUMP 1 FLOW ALARM
%MX230481	RP-3 INVER&DMPI ALARM
%MX230482	RP-3 MCCB ALARM
%MX230483	RP-3 PUMP 과열 ALARM
%MX230484	RP-3 FLOW ALARM
%MX230485	RP-4 INVER&DMPI ALARM
%MX230486	RP-4 MCCB ALARM
%MX230487	RP-4 PUMP 과열 ALARM
%MX230488	RP-4 FLOW ALARM
%MX230489	SP-2 INVER&DMPI ALARM
%MX230490	SP-2 MCCB ALARM
%MX230491	SP-2 PUMP 과열 ALARM
%MX230492	SP-2 FLOW ALARM
%MX230493	RP-9 INVER&DMPI ALARM
%MX230494	RP-9 MCCB ALARM
%MX230495	RP-9 PUMP 과열 ALARM
%MX230496	RP-9 FLOW ALARM
%MX230497	RP-10 INVER&DMPI ALARM
%MX230498	RP-10 MCCB ALARM
%MX230499	RP-10 PUMP 과열 ALARM
%MX230500	RP-10 FLOW ALARM
%MX230501	RP-11 INVER&DMPI ALARM
%MX230502	RP-11 MCCB ALARM
%MX230503	RP-11 PUMP 과열 ALARM
%MX230504	RP-11 FLOW ALARM
%MX230505	RP-12 INVER&DMPI ALARM
%MX230506	RP-12 MCCB ALARM
%MX230507	RP-12 PUMP 과열 ALARM
%MX230508	RP-12 FLOW ALARM
%MX230509	RP-7 INVER&DMPI ALARM
%MX230510	RP-7 MCCB ALARM
%MX230511	RP-7 PUMP 과열 ALARM
%MX230512	RP-7 FLOW ALARM
%MX230513	RP-8 INVER&DMPI ALARM
%MX230514	RP-8 MCCB ALARM
%MX230515	RP-8 PUMP 과열 ALARM
%MX230516	RP-8 FLOW ALARM
%MX230517	SUMP PUMP 4 INVER&DMPI ALARM
%MX230518	SUMP PUMP 4 MCCB ALARM
%MX230519	SUMP PUMP 4 PUMP 과열 ALARM
%MX230520	SUMP PUMP 4 FLOW ALARM
%MX230521	RP-13 INVER&DMPI ALARM
%MX230522	RP-13 MCCB ALARM
%MX230523	RP-13 PUMP 과열 ALARM
%MX230524	RP-13 FLOW ALARM
%MX230528	RP-14 INVER&DMPI ALARM
%MX230529	RP-14 MCCB ALARM
%MX230530	RP-14 PUMP 과열 ALARM
%MX230531	RP-14 FLOW ALARM
%MX230532	RP-5 INVER&DMPI ALARM
%MX230533	RP-5 MCCB ALARM
%MX230534	RP-5 PUMP 과열 ALARM
%MX230535	RP-5 FLOW ALARM
%MX230536	RP-6 INVER&DMPI ALARM
%MX230537	RP-6 MCCB ALARM
%MX230538	RP-6 PUMP 과열 ALARM
%MX230539	RP-6 FLOW ALARM
%MX230540	SUMP PUMP 3 INVER&DMPI ALARM
%MX230541	SUMP PUMP 3 MCCB ALARM
%MX230542	SUMP PUMP 3 PUMP 과열 ALARM
%MX230543	SUMP PUMP 3 FLOW ALARM
%MX230544	RP-15 INVER&DMPI ALARM
%MX230545	RP-15 MCCB ALARM
%MX230546	RP-15 PUMP 과열 ALARM
%MX230547	RP-15 FLOW ALARM
%MX230548	RP-16 INVER&DMPI ALARM
%MX230549	RP-16 MCCB ALARM
%MX230550	RP-16 PUMP 과열 ALARM
%MX230551	RP-16 FLOW ALARM
%MX230552	DP-02 INVER&DMPI ALARM
%MX230553	DP-02 MCCB ALARM
%MX230554	DP-02 PUMP 과열 ALARM
%MX230555	DP-02 FLOW ALARM
%MX230592	SOL VALVE 전원이상
%MX230593	DF-1B 누유
%MX230594	DF-1A 누유
%MX230595	MOGAS 누유
%MX230596	DF-M 누유
%MX230597	누유 ALARM
%MX230598	DF-1B FAN ALARM
%MX230599	DF-1A FAN ALARM
%MX230600	DF-M FAN ALARM
%MX230601	MOGAS FAN ALARM
%MX231040	NC
%MX231041	NC
%MX231042	NC
%MX231043	NC
%MX231044	NC
%MX231045	NC
%MX231046	NC
%MX231047	NC
%MX231048	NC
%MX231049	NC
%MX231050	NC
%MX231051	NC
%MX231052	NC
%MX231053	NC
%MX231054	NC
%MX231055	NC
%MX231056	NC
%MX231057	NC
%MX231058	NC
%MX231059	NC
%MX231060	NC
%MX231061	NC
%MX231062	NC
%MX231063	NC
%MX231064	NC
%MX231065	NC
%MX231066	NC
%MX231067	NC
%MX231068	NC
%MX231069	NC
%MX231070	NC
%MX231071	NC
%MX231072	NC
%MX231073	NC
%MX231074	NC
%MX231075	NC
%MX231076	NC
%MX231077	NC
%MX231078	NC
%MX231079	NC
%MX231080	NC
%MX231081	NC
%MX231082	NC
%MX231083	NC
%MX231084	NC
%MX231085	NC
%MX231086	NC
%MX231087	NC
%MX231088	NC
%MX231089	NC
%MX231090	NC
%MX231091	NC
%MX231092	NC
%MX231093	NC
%MX231094	NC
%MX231095	NC
%MX231096	NC
%MX231097	NC
%MX231098	NC
%MX231099	NC
%MX231100	NC
%MX231101	NC
%MX231102	NC
%MX231103	NC
%MX231680	NC
%MX231681	NC
%MX231682	NC
%MX231683	NC
%MX231684	NC
%MX231685	NC
%WW182	DRAIN TK113 Run SET
%WW200	DF-1 출하 PUMP 1차 선택
%WW201	DF-1 출하 PUMP 2차 선택
%WW210	DF-M SET 1=RP7, 2=RP8
%WW220	MOGAS SET 1=RP5, 2=RP6
%WW410	PT101 회수압력
%WW412	PT101 회수압력계 레인지 연산값
%WW520	DF-1 출하유량 (FIT1)
%WW530	DF-1 출하유량 (FIT2)
%WW550	DF-1 출하압력 OUT (PIT1)
%WW700	DF-1A TANK LEVEL
%WW704	DA-1A TEMP [PLC TO SCADA]
%WW708	DA-1A VOLUME [PLC TO SCADA]
%WW710	DF-1B TANK LEVEL
%WW714	DF-1B TEMP [PLC TO SCADA]
%WW718	DF-1B VOLUME [PLC TO SCADA]
%WW720	DF-M TANK LEVEL(%)TO SCADA
%WW724	DF-M TEMP [PLC TO SCADA]
%WW728	DF-M VOLUME [PLC TO SCADA]
%WW730	MOGAS TANK LEVEL (TO SCADA)
%WW734	MOGAS TEMP [PLC TO SCADA]
%WW738	MOGAS VOLUME [PLC TO SCADA]
%WW740	DF-1 DRAIN TANK LEVEL
%WW748	DF-1 DRAIN VOLUME [PLC TO SCADA]
%WW750	MOGAS DRAIN TANK LEVEL (TO SCADA)
%WW758	MOGAS DRAIN VOLUME [PLC TO SCADA]
%WW1000	불출압력 (DF-1A/B) – PT12
%WW1002	불출압력 (DF-M) – PT34
%WW1004	불출압력 (MOGAS) – PT56
%WW1006	불출유량 (DF-1A/B) – FT12
%WW1008	불출유량 (DF-M) – FT34
%WW1010	불출유량 (MOGAS) – FT5,6 (PLC->SCADA)
%WD412	PT101 회수압력계 레인지 연산값 2WORD 변환
*)

PROGRAM MAIN (* task: 스캔 프로그램 *)
VAR
    D200 : BOOL;
    D201 : BOOL;
    DW200 : BOOL;
    DWW : BOOL;
    INST : TON;
    RP01 : TON;
    RP02 : TON;
    SET1 : TON;
    SET10 : TON;
    SET10_1 : TON;
    SET10_2 : TON;
    SET11 : TON;
    SET11_1 : TON;
    SET12 : TON;
    SET12_1 : TON;
    SET13 : TON;
    SET14 : TON;
    SET15 : TON;
    SET16 : TON;
    SET1_1 : TON;
    SET1_2 : TON;
    SET1_3 : TON;
    SET1_4 : TON;
    SET2 : TON;
    SET2_1 : TON;
    SET2_2 : TON;
    SET2_3 : TON;
    SET2_4 : TON;
    SET3 : TON;
    SET3_1 : TON;
    SET3_2 : TON;
    SET4 : TON;
    SET4_1 : TON;
    SET4_2 : TON;
    SET5 : TON;
    SET5_1 : TON;
    SET6 : TON;
    SET6_1 : TON;
    SET7 : TON;
    SET7_1 : TON;
    SET8 : TON;
    SET8_1 : TON;
    SET9 : TON;
    SET9_1 : TON;
    SET9_2 : TON;
    ㅢ202 : BYTE;
END_VAR
VAR
    _t1 : BOOL;
    _t2 : BOOL;
    _t3 : BOOL;
    _t4 : BOOL;
    _t5 : BOOL;
    _t6 : BOOL;
    _t7 : BOOL;
    _t8 : BOOL;
END_VAR

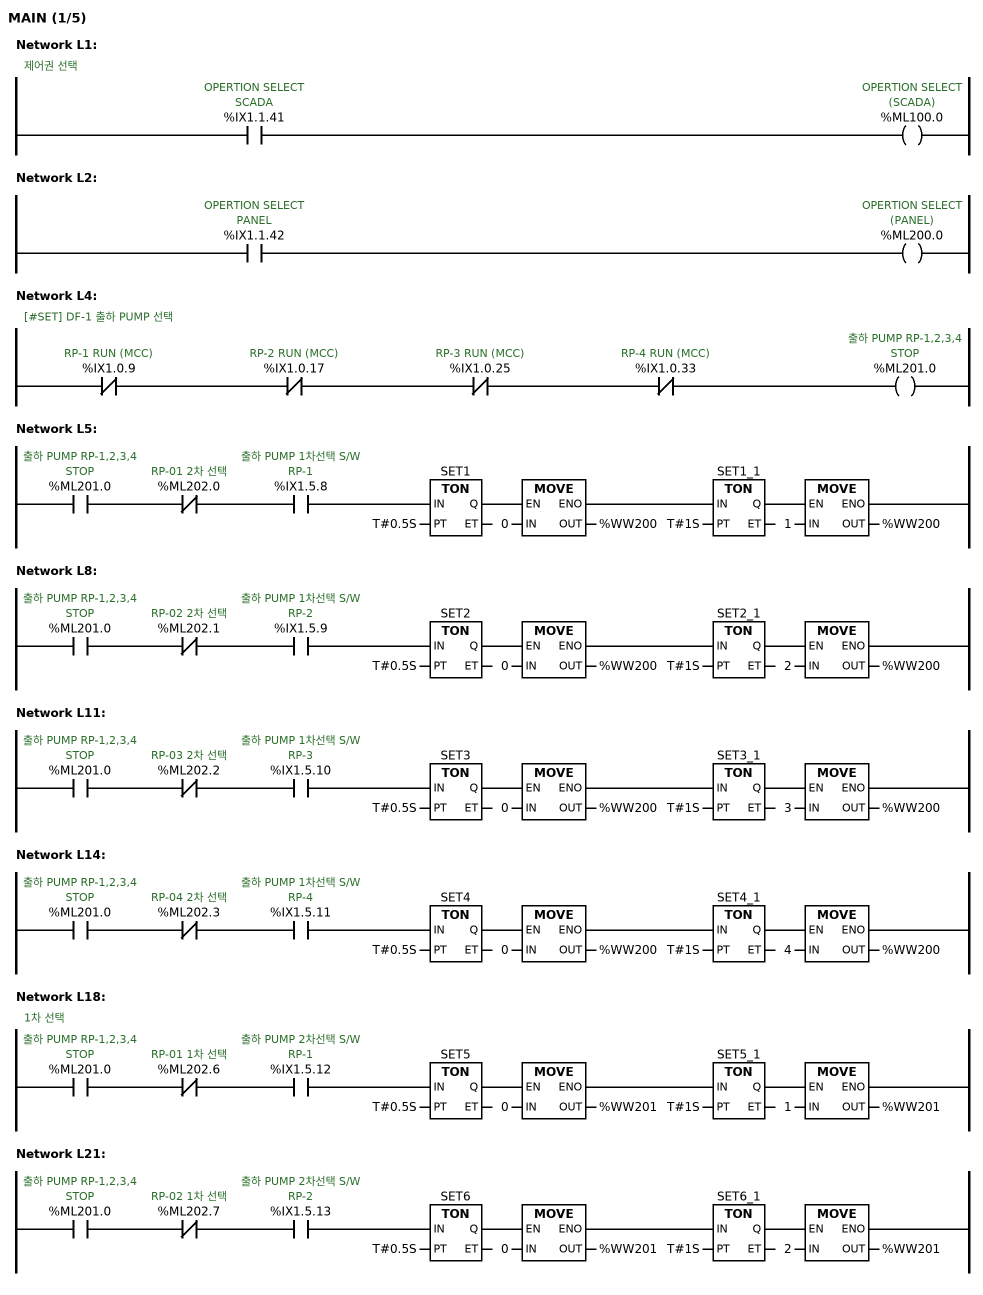
(* 제어권 선택 *)
(* Rung L1 *)
%ML100.0 := %IX1.1.41;
(* Rung L2 *)
%ML200.0 := %IX1.1.42;
(* [#SET] DF-1 출하 PUMP 선택 *)
(* Rung L4 *)
%ML201.0 := NOT %IX1.0.9 AND NOT %IX1.0.17 AND NOT %IX1.0.25 AND NOT %IX1.0.33;
(* Rung L5 *)
SET1(IN := %ML201.0 AND NOT %ML202.0 AND %IX1.5.8, PT := T#0.5S);
IF SET1.Q THEN %WW200 := 0; END_IF;
SET1_1(IN := SET1.Q, PT := T#1S);
IF SET1_1.Q THEN %WW200 := 1; END_IF;
(* Rung L8 *)
SET2(IN := %ML201.0 AND NOT %ML202.1 AND %IX1.5.9, PT := T#0.5S);
IF SET2.Q THEN %WW200 := 0; END_IF;
SET2_1(IN := SET2.Q, PT := T#1S);
IF SET2_1.Q THEN %WW200 := 2; END_IF;
(* Rung L11 *)
SET3(IN := %ML201.0 AND NOT %ML202.2 AND %IX1.5.10, PT := T#0.5S);
IF SET3.Q THEN %WW200 := 0; END_IF;
SET3_1(IN := SET3.Q, PT := T#1S);
IF SET3_1.Q THEN %WW200 := 3; END_IF;
(* Rung L14 *)
SET4(IN := %ML201.0 AND NOT %ML202.3 AND %IX1.5.11, PT := T#0.5S);
IF SET4.Q THEN %WW200 := 0; END_IF;
SET4_1(IN := SET4.Q, PT := T#1S);
IF SET4_1.Q THEN %WW200 := 4; END_IF;
(* 1차 선택 *)
(* Rung L18 *)
SET5(IN := %ML201.0 AND NOT %ML202.6 AND %IX1.5.12, PT := T#0.5S);
IF SET5.Q THEN %WW201 := 0; END_IF;
SET5_1(IN := SET5.Q, PT := T#1S);
IF SET5_1.Q THEN %WW201 := 1; END_IF;
(* Rung L21 *)
SET6(IN := %ML201.0 AND NOT %ML202.7 AND %IX1.5.13, PT := T#0.5S);
IF SET6.Q THEN %WW201 := 0; END_IF;
SET6_1(IN := SET6.Q, PT := T#1S);
IF SET6_1.Q THEN %WW201 := 2; END_IF;

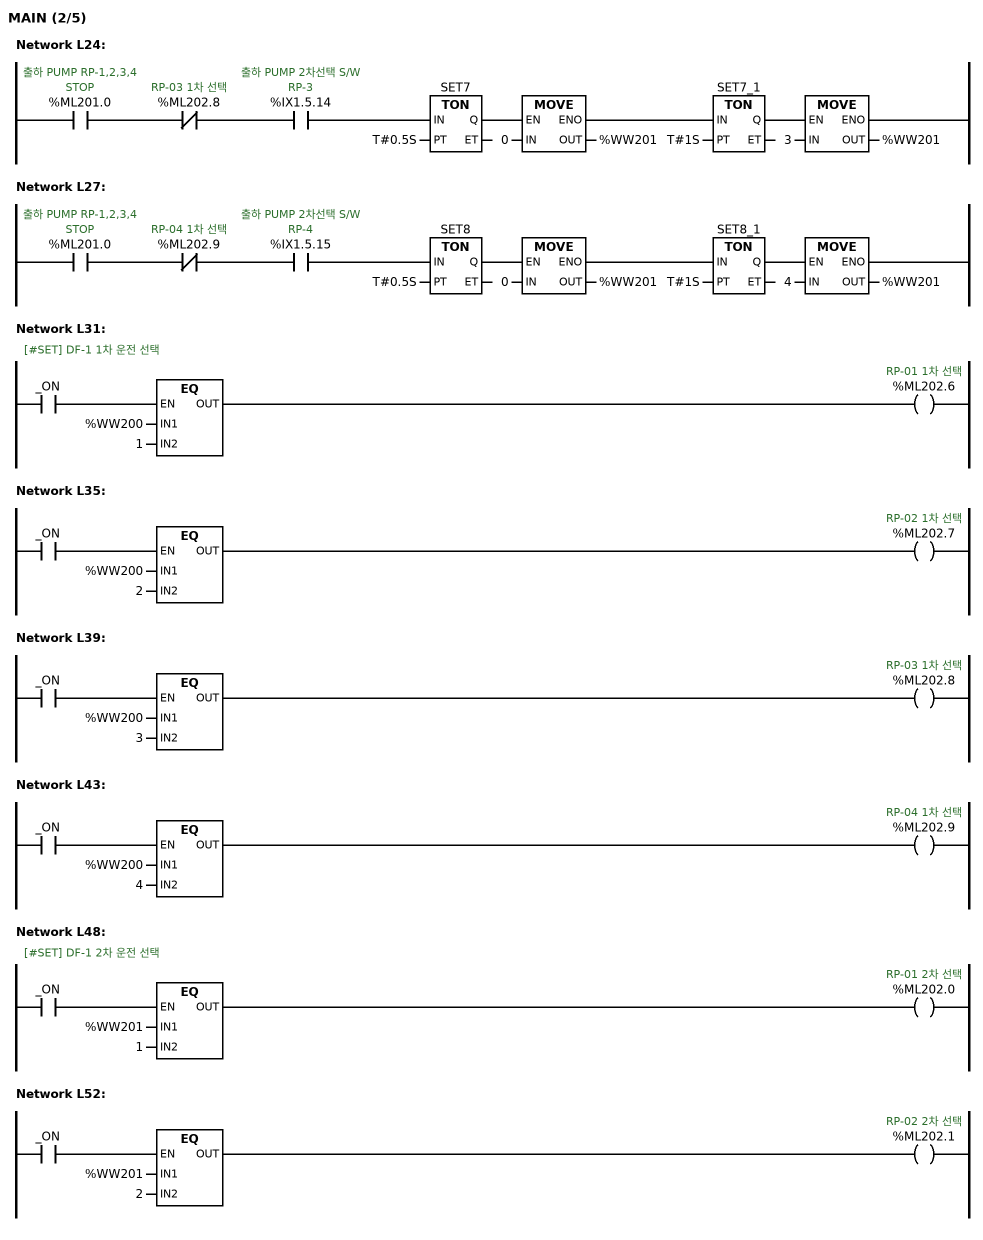
(* Rung L24 *)
SET7(IN := %ML201.0 AND NOT %ML202.8 AND %IX1.5.14, PT := T#0.5S);
IF SET7.Q THEN %WW201 := 0; END_IF;
SET7_1(IN := SET7.Q, PT := T#1S);
IF SET7_1.Q THEN %WW201 := 3; END_IF;
(* Rung L27 *)
SET8(IN := %ML201.0 AND NOT %ML202.9 AND %IX1.5.15, PT := T#0.5S);
IF SET8.Q THEN %WW201 := 0; END_IF;
SET8_1(IN := SET8.Q, PT := T#1S);
IF SET8_1.Q THEN %WW201 := 4; END_IF;
(* [#SET] DF-1 1차 운전 선택 *)
(* Rung L31 *)
IF _ON THEN _t1 := %WW200 = 1; END_IF;
%ML202.6 := _t1;
(* Rung L35 *)
IF _ON THEN _t2 := %WW200 = 2; END_IF;
%ML202.7 := _t2;
(* Rung L39 *)
IF _ON THEN _t3 := %WW200 = 3; END_IF;
%ML202.8 := _t3;
(* Rung L43 *)
IF _ON THEN _t4 := %WW200 = 4; END_IF;
%ML202.9 := _t4;
(* [#SET] DF-1 2차 운전 선택 *)
(* Rung L48 *)
IF _ON THEN _t5 := %WW201 = 1; END_IF;
%ML202.0 := _t5;
(* Rung L52 *)
IF _ON THEN _t6 := %WW201 = 2; END_IF;
%ML202.1 := _t6;

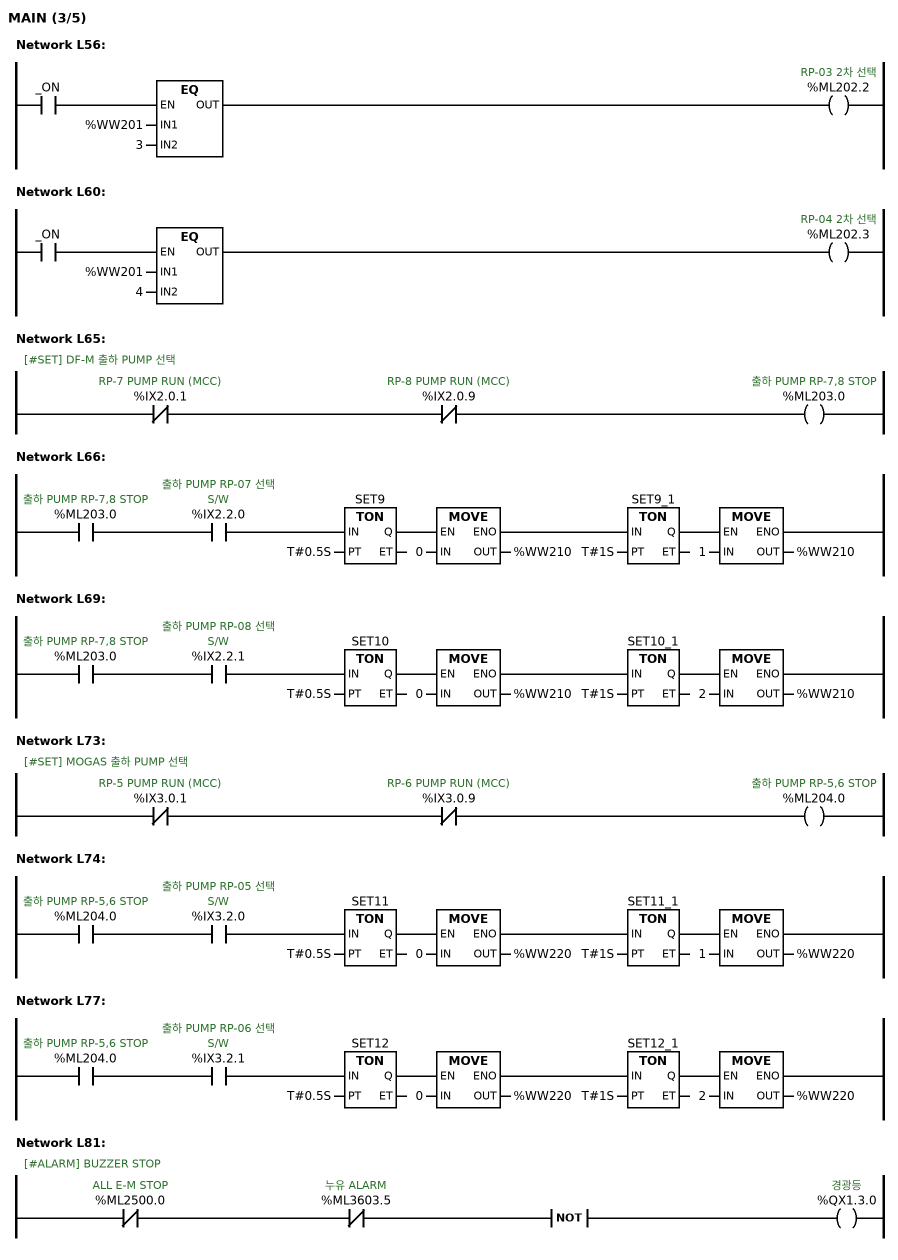
(* Rung L56 *)
IF _ON THEN _t7 := %WW201 = 3; END_IF;
%ML202.2 := _t7;
(* Rung L60 *)
IF _ON THEN _t8 := %WW201 = 4; END_IF;
%ML202.3 := _t8;
(* [#SET] DF-M 출하 PUMP 선택 *)
(* Rung L65 *)
%ML203.0 := NOT %IX2.0.1 AND NOT %IX2.0.9;
(* Rung L66 *)
SET9(IN := %ML203.0 AND %IX2.2.0, PT := T#0.5S);
IF SET9.Q THEN %WW210 := 0; END_IF;
SET9_1(IN := SET9.Q, PT := T#1S);
IF SET9_1.Q THEN %WW210 := 1; END_IF;
(* Rung L69 *)
SET10(IN := %ML203.0 AND %IX2.2.1, PT := T#0.5S);
IF SET10.Q THEN %WW210 := 0; END_IF;
SET10_1(IN := SET10.Q, PT := T#1S);
IF SET10_1.Q THEN %WW210 := 2; END_IF;
(* [#SET] MOGAS 출하 PUMP 선택 *)
(* Rung L73 *)
%ML204.0 := NOT %IX3.0.1 AND NOT %IX3.0.9;
(* Rung L74 *)
SET11(IN := %ML204.0 AND %IX3.2.0, PT := T#0.5S);
IF SET11.Q THEN %WW220 := 0; END_IF;
SET11_1(IN := SET11.Q, PT := T#1S);
IF SET11_1.Q THEN %WW220 := 1; END_IF;
(* Rung L77 *)
SET12(IN := %ML204.0 AND %IX3.2.1, PT := T#0.5S);
IF SET12.Q THEN %WW220 := 0; END_IF;
SET12_1(IN := SET12.Q, PT := T#1S);
IF SET12_1.Q THEN %WW220 := 2; END_IF;
(* [#ALARM] BUZZER STOP *)
(* Rung L81 *)
%QX1.3.0 := NOT (NOT %ML2500.0 AND NOT %ML3603.5);
(*  *)

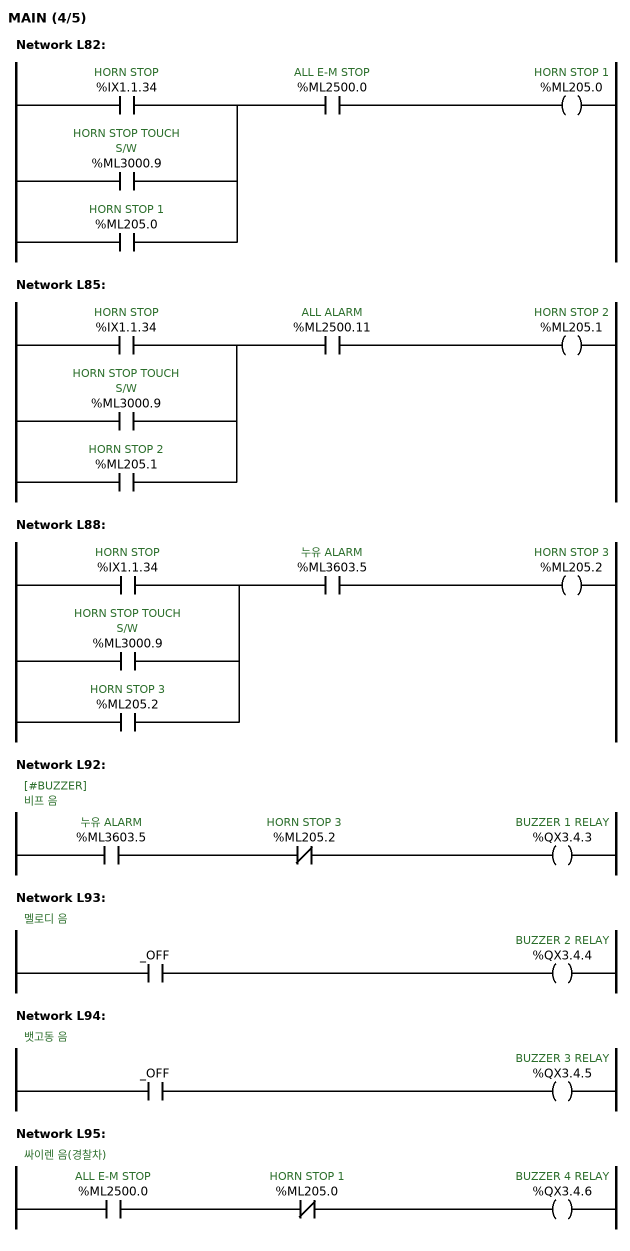
(* Rung L82 *)
%ML205.0 := (%IX1.1.34 OR %ML3000.9 OR %ML205.0) AND %ML2500.0;
(* Rung L85 *)
%ML205.1 := (%IX1.1.34 OR %ML3000.9 OR %ML205.1) AND %ML2500.11;
(* Rung L88 *)
%ML205.2 := (%IX1.1.34 OR %ML3000.9 OR %ML205.2) AND %ML3603.5;
(* [#BUZZER] *)
(* Rung L92 *)
%QX3.4.3 := %ML3603.5 AND NOT %ML205.2;
(* 비프 음 *)
(* Rung L93 *)
%QX3.4.4 := _OFF;
(* 멜로디 음 *)
(* Rung L94 *)
%QX3.4.5 := _OFF;
(* 뱃고동 음 *)
(* Rung L95 *)
%QX3.4.6 := %ML2500.0 AND NOT %ML205.0;
(* 싸이렌 음(경찰차) *)

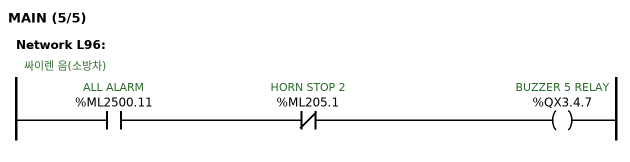
(* Rung L96 *)
%QX3.4.7 := %ML2500.11 AND NOT %ML205.1;
(* 싸이렌 음(소방차) *)
END_PROGRAM

PROGRAM AUTO (* task: 스캔 프로그램 *)
VAR
    PUMP_RUN_EA : INT;
END_VAR
VAR_EXTERNAL
    RP01_2차 : TON;
    _0108_CH2_DATA : INT; (* AT %UW1.8.4 *) (* 절연형 아날로그입력 모듈: 채널2 변환값 *)
    _0108_CH3_DATA : INT; (* AT %UW1.8.5 *) (* 절연형 아날로그입력 모듈: 채널3 변환값 *)
END_VAR
VAR
    _t1 : BOOL;
    _t2 : BOOL;
    _p3 : BOOL;
    _t4 : BOOL;
    _t5 : BOOL;
END_VAR

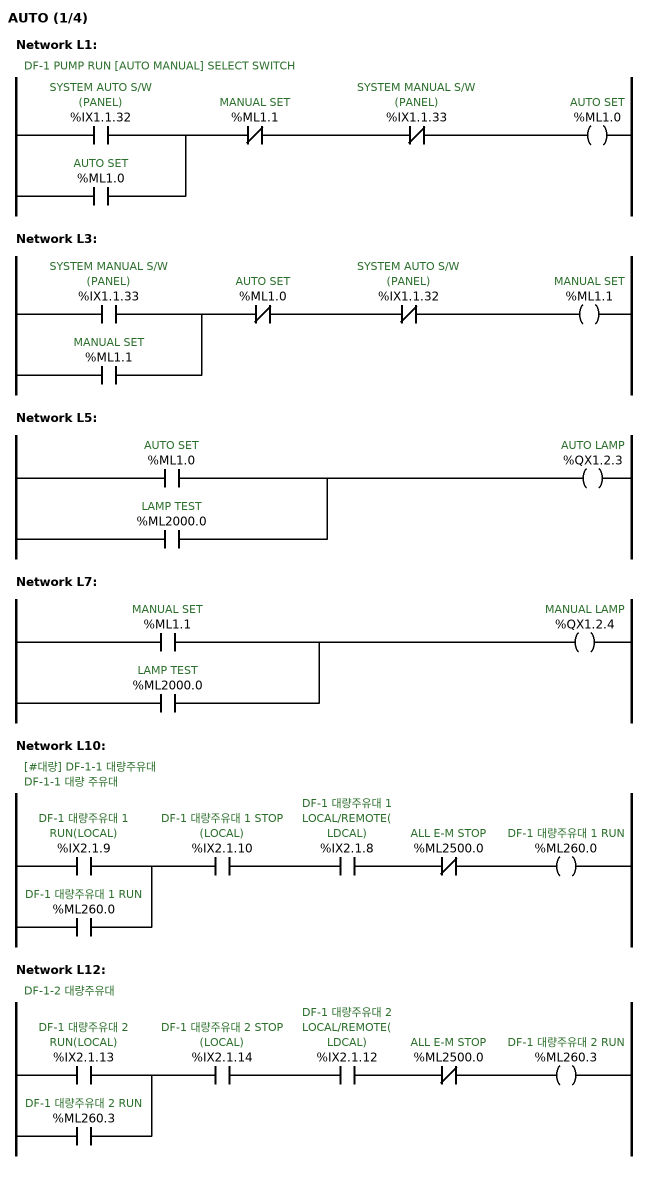
(* DF-1 PUMP RUN [AUTO MANUAL] SELECT SWITCH *)
(* Rung L1 *)
%ML1.0 := (%IX1.1.32 OR %ML1.0) AND NOT %ML1.1 AND NOT %IX1.1.33;
(* Rung L3 *)
%ML1.1 := (%IX1.1.33 OR %ML1.1) AND NOT %ML1.0 AND NOT %IX1.1.32;
(* Rung L5 *)
%QX1.2.3 := %ML1.0 OR %ML2000.0;
(* Rung L7 *)
%QX1.2.4 := %ML1.1 OR %ML2000.0;
(* [#대량] DF-1-1 대량주유대 *)
(* Rung L10 *)
%ML260.0 := (%IX2.1.9 OR %ML260.0) AND %IX2.1.10 AND %IX2.1.8 AND NOT %ML2500.0;
(* DF-1-1 대량 주유대 *)
(* Rung L12 *)
%ML260.3 := (%IX2.1.13 OR %ML260.3) AND %IX2.1.14 AND %IX2.1.12 AND NOT %ML2500.0;
(* DF-1-2 대량주유대 *)

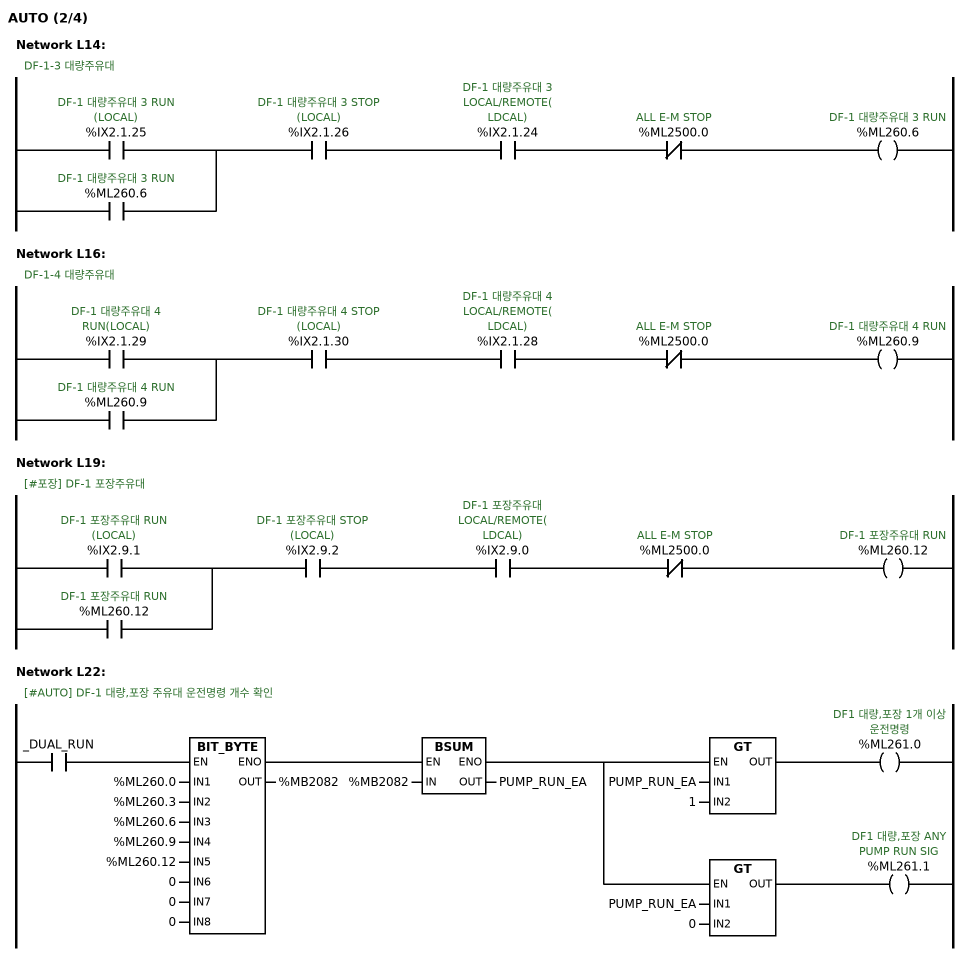
(* Rung L14 *)
%ML260.6 := (%IX2.1.25 OR %ML260.6) AND %IX2.1.26 AND %IX2.1.24 AND NOT %ML2500.0;
(* DF-1-3 대량주유대 *)
(* Rung L16 *)
%ML260.9 := (%IX2.1.29 OR %ML260.9) AND %IX2.1.30 AND %IX2.1.28 AND NOT %ML2500.0;
(* DF-1-4 대량주유대 *)
(* [#포장] DF-1 포장주유대 *)
(* Rung L19 *)
%ML260.12 := (%IX2.9.1 OR %ML260.12) AND %IX2.9.2 AND %IX2.9.0 AND NOT %ML2500.0;
(* [#AUTO] DF-1 대량,포장 주유대 운전명령 개수 확인 *)
(* Rung L22 *)
IF _DUAL_RUN THEN
    %MB2082 := BIT_BYTE(%ML260.0, %ML260.3, %ML260.6, %ML260.9, %ML260.12, 0, 0, 0);
    PUMP_RUN_EA := BSUM(%MB2082);
    _t1 := PUMP_RUN_EA > 1;
END_IF;
%ML261.0 := _t1;
IF _DUAL_RUN THEN _t2 := PUMP_RUN_EA > 0; END_IF;
%ML261.1 := _t2;

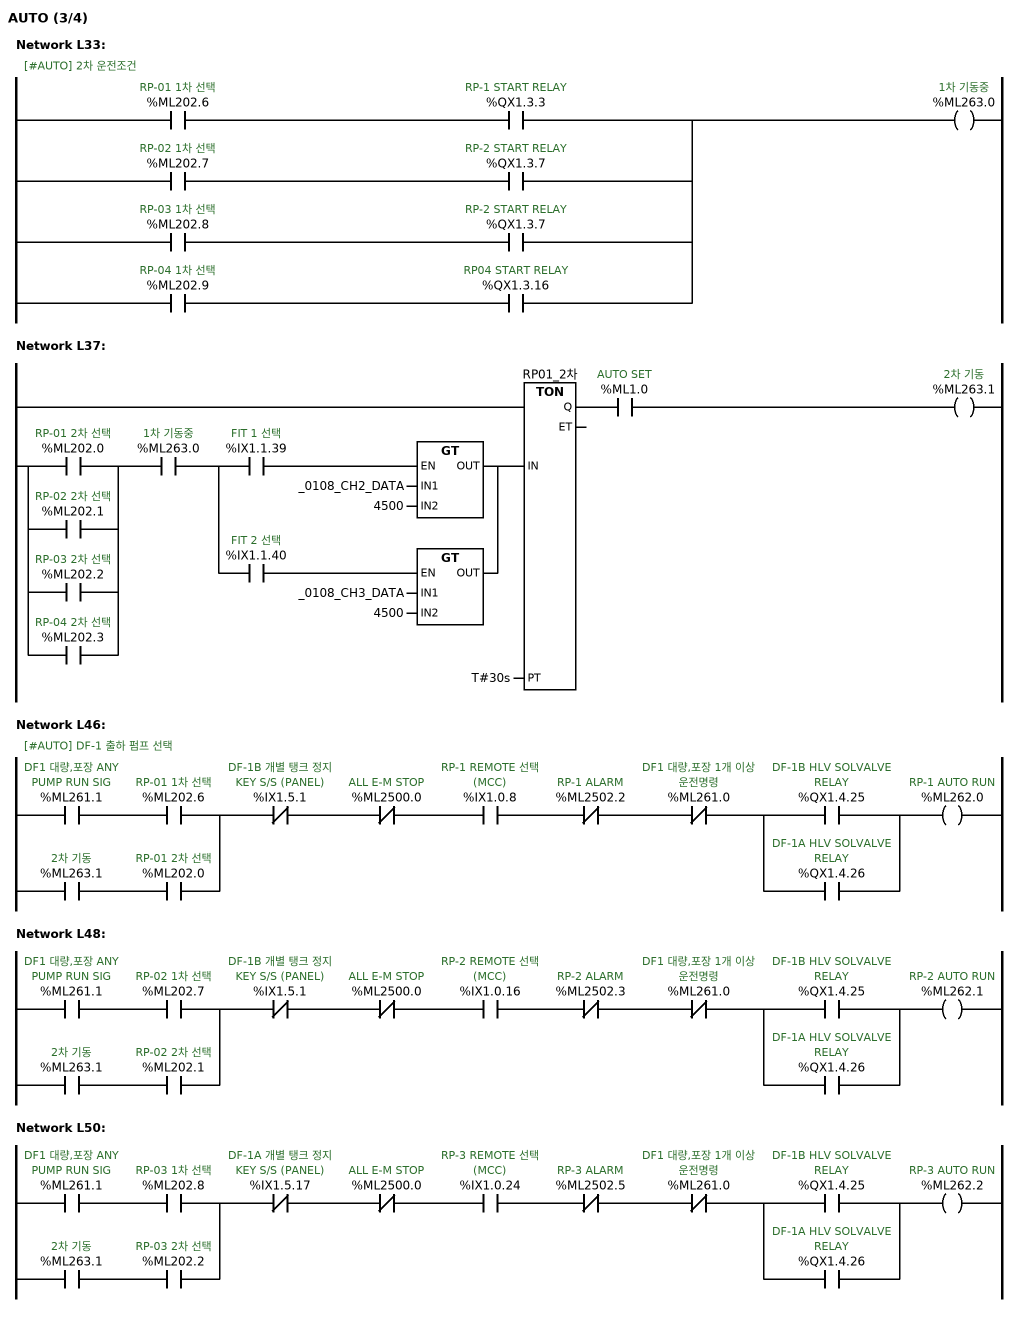
(* [#AUTO] 2차 운전조건 *)
(* Rung L33 *)
%ML263.0 := (%ML202.6 AND %QX1.3.3) OR (%ML202.7 AND %QX1.3.7) OR (%ML202.8 AND %QX1.3.7) OR (%ML202.9 AND %QX1.3.16);
(* Rung L37 *)
_p3 := (%ML202.0 OR %ML202.1 OR %ML202.2 OR %ML202.3) AND %ML263.0;
IF _p3 AND %IX1.1.39 THEN _t4 := _0108_CH2_DATA > 4500; END_IF;
IF _p3 AND %IX1.1.40 THEN _t5 := _0108_CH3_DATA > 4500; END_IF;
RP01_2차(IN := _t4 OR _t5, PT := T#30s);
%ML263.1 := RP01_2차.Q AND %ML1.0;
(* [#AUTO] DF-1 출하 펌프 선택 *)
(* Rung L46 *)
%ML262.0 := ((%ML261.1 AND %ML202.6) OR (%ML263.1 AND %ML202.0)) AND NOT %IX1.5.1 AND NOT %ML2500.0 AND %IX1.0.8 AND NOT %ML2502.2 AND NOT %ML261.0 AND (%QX1.4.25 OR %QX1.4.26);
(* Rung L48 *)
%ML262.1 := ((%ML261.1 AND %ML202.7) OR (%ML263.1 AND %ML202.1)) AND NOT %IX1.5.1 AND NOT %ML2500.0 AND %IX1.0.16 AND NOT %ML2502.3 AND NOT %ML261.0 AND (%QX1.4.25 OR %QX1.4.26);
(* Rung L50 *)
%ML262.2 := ((%ML261.1 AND %ML202.8) OR (%ML263.1 AND %ML202.2)) AND NOT %IX1.5.17 AND NOT %ML2500.0 AND %IX1.0.24 AND NOT %ML2502.5 AND NOT %ML261.0 AND (%QX1.4.25 OR %QX1.4.26);

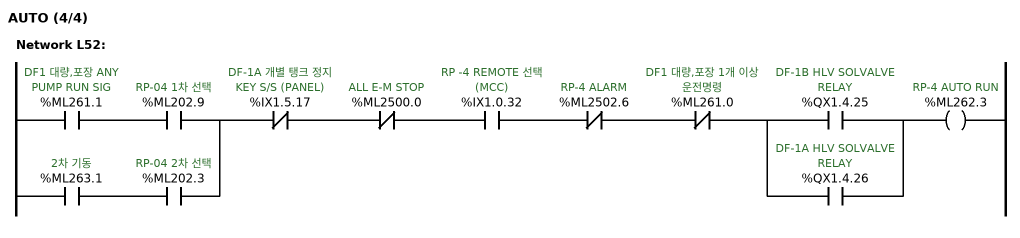
(* Rung L52 *)
%ML262.3 := ((%ML261.1 AND %ML202.9) OR (%ML263.1 AND %ML202.3)) AND NOT %IX1.5.17 AND NOT %ML2500.0 AND %IX1.0.32 AND NOT %ML2502.6 AND NOT %ML261.0 AND (%QX1.4.25 OR %QX1.4.26);
END_PROGRAM

PROGRAM DRAIN (* task: 스캔 프로그램 *)
VAR
    DP01 : TON; (* DRAIN PUMP FLOW SENSOR *)
    DP02 : TON; (* DRAIN PUMP FLOW SENSOR *)
    DP03 : TON; (* DRAIN PUMP FLOW SENSOR *)
    INST : TON;
    T5S : TIME;
END_VAR

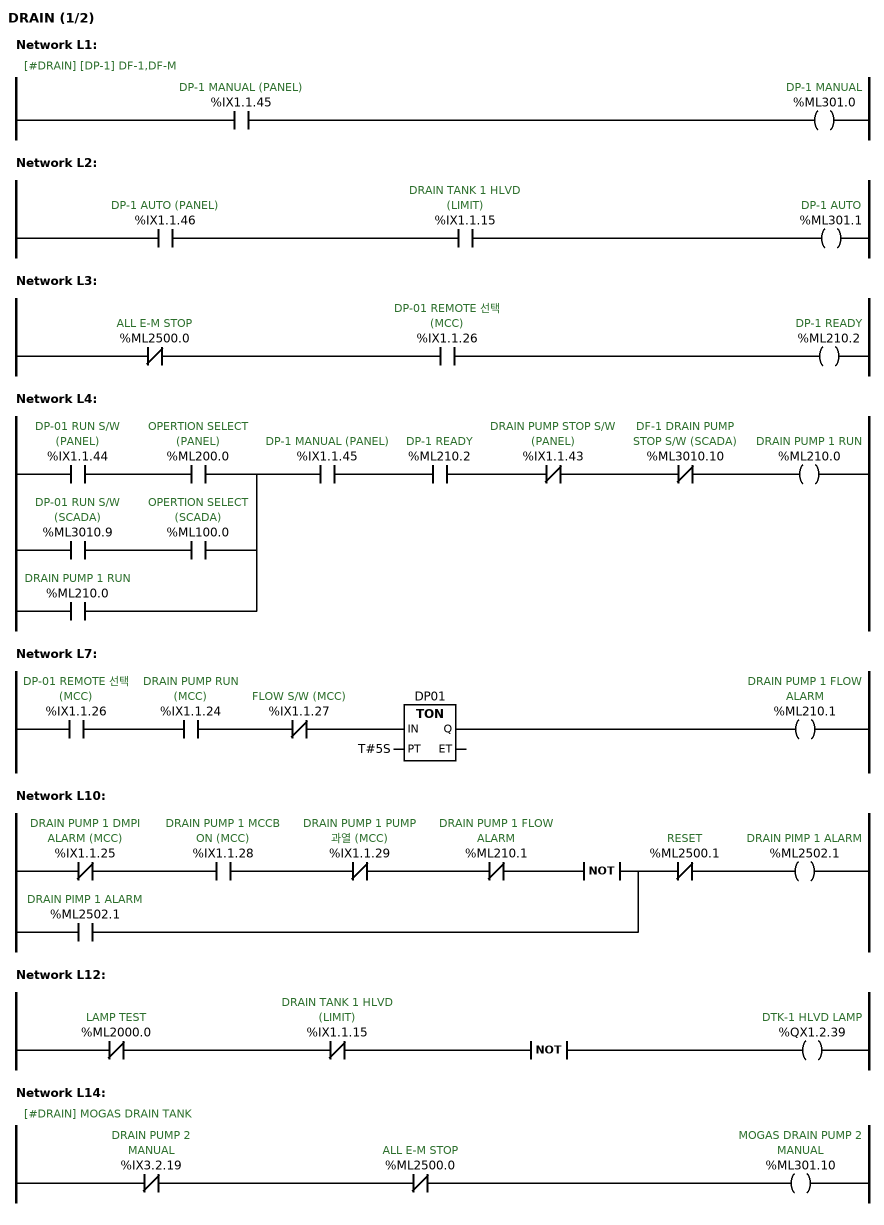
(* [#DRAIN] [DP-1] DF-1,DF-M *)
(* Rung L1 *)
%ML301.0 := %IX1.1.45;
(* Rung L2 *)
%ML301.1 := %IX1.1.46 AND %IX1.1.15;
(* Rung L3 *)
%ML210.2 := NOT %ML2500.0 AND %IX1.1.26;
(* Rung L4 *)
%ML210.0 := ((%IX1.1.44 AND %ML200.0) OR (%ML3010.9 AND %ML100.0) OR %ML210.0) AND %IX1.1.45 AND %ML210.2 AND NOT %IX1.1.43 AND NOT %ML3010.10;
(* Rung L7 *)
DP01(IN := %IX1.1.26 AND %IX1.1.24 AND NOT %IX1.1.27, PT := T#5S);
%ML210.1 := DP01.Q;
(* Rung L10 *)
%ML2502.1 := (NOT (NOT %IX1.1.25 AND %IX1.1.28 AND NOT %IX1.1.29 AND NOT %ML210.1) OR %ML2502.1) AND NOT %ML2500.1;
(* Rung L12 *)
%QX1.2.39 := NOT (NOT %ML2000.0 AND NOT %IX1.1.15);
(* [#DRAIN] MOGAS DRAIN TANK *)
(* Rung L14 *)
%ML301.10 := NOT %IX3.2.19 AND NOT %ML2500.0;

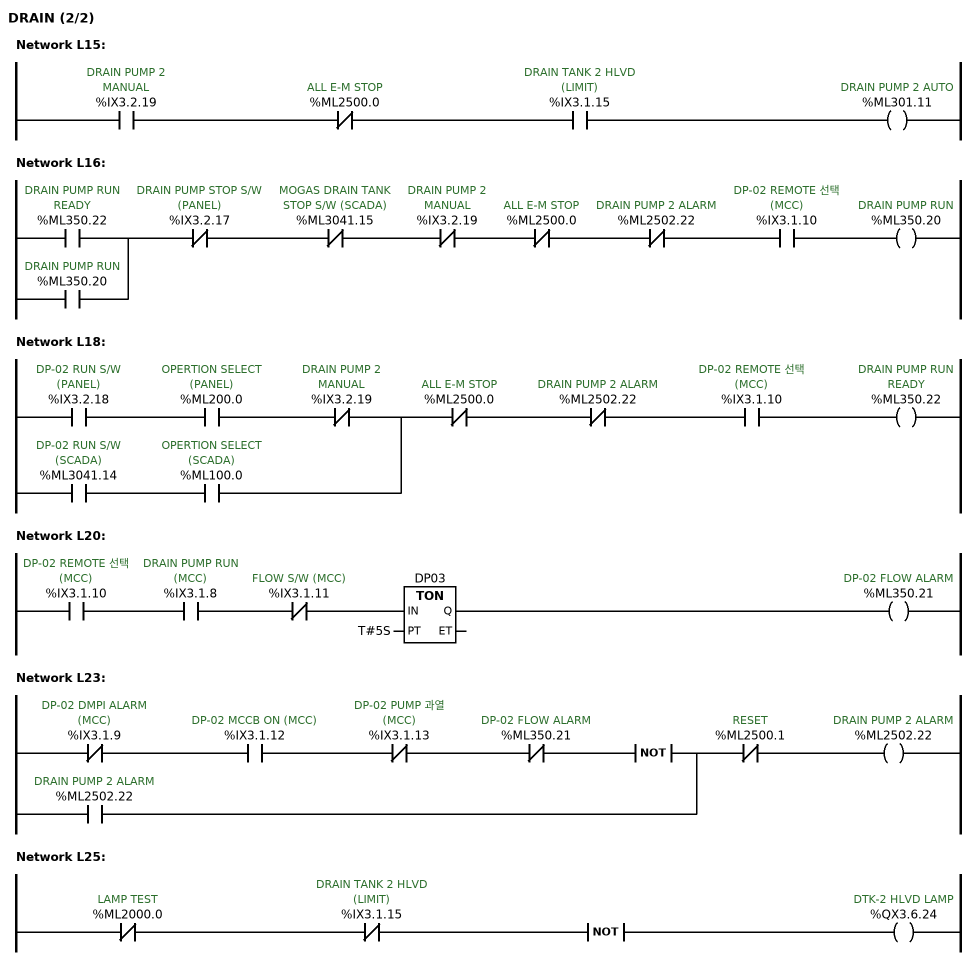
(* Rung L15 *)
%ML301.11 := %IX3.2.19 AND NOT %ML2500.0 AND %IX3.1.15;
(* Rung L16 *)
%ML350.20 := (%ML350.22 OR %ML350.20) AND NOT %IX3.2.17 AND NOT %ML3041.15 AND NOT %IX3.2.19 AND NOT %ML2500.0 AND NOT %ML2502.22 AND %IX3.1.10;
(* Rung L18 *)
%ML350.22 := ((%IX3.2.18 AND %ML200.0 AND NOT %IX3.2.19) OR (%ML3041.14 AND %ML100.0)) AND NOT %ML2500.0 AND NOT %ML2502.22 AND %IX3.1.10;
(* Rung L20 *)
DP03(IN := %IX3.1.10 AND %IX3.1.8 AND NOT %IX3.1.11, PT := T#5S);
%ML350.21 := DP03.Q;
(* Rung L23 *)
%ML2502.22 := (NOT (NOT %IX3.1.9 AND %IX3.1.12 AND NOT %IX3.1.13 AND NOT %ML350.21) OR %ML2502.22) AND NOT %ML2500.1;
(* Rung L25 *)
%QX3.6.24 := NOT (NOT %ML2000.0 AND NOT %IX3.1.15);
END_PROGRAM

PROGRAM DF-1 (* task: 스캔 프로그램 *)
VAR
    DP01 : TON; (* DRAIN PUMP FLOW SENSOR *)
    DP02 : TON; (* DRAIN PUMP FLOW SENSOR *)
    GVAL : DWORD;
    HVAL : DWORD;
    PUMP_RUN_EA : INT;
    RP01 : TON;
    RP02 : TON;
    RP03 : TON;
    RP04 : TON;
    RP05 : TON;
    RP10 : TON;
    RP11 : TON;
    RP12 : TON;
    RP13 : TON;
    RP14 : TON;
    RP15 : TON;
    RP16 : TON;
    RP17 : TON;
    RP18 : TON;
    RP19 : TON;
    RP20 : TON;
    RP21 : TON;
    RP9 : TON;
    SP01 : TON;
    SP02 : TON;
    SUMP01 : TON; (* SUMP PUMP1 *)
    SUMP02 : TON; (* SP-2 *)
    SUMP03 : TON; (* SP-2 *)
END_VAR
VAR_EXTERNAL
    RP01_2차 : TON;
    RP01_3차 : TON;
    _0108_CH1_DATA : INT; (* AT %UW1.8.3 *) (* 절연형 아날로그입력 모듈: 채널1 변환값 *)
    _0108_CH2_DATA : INT; (* AT %UW1.8.4 *) (* 절연형 아날로그입력 모듈: 채널2 변환값 *)
    _0108_CH3_DATA : INT; (* AT %UW1.8.5 *) (* 절연형 아날로그입력 모듈: 채널3 변환값 *)
END_VAR
VAR
    _e1 : R_TRIG;
    _e2 : R_TRIG;
    _e3 : R_TRIG;
    _e4 : R_TRIG;
END_VAR

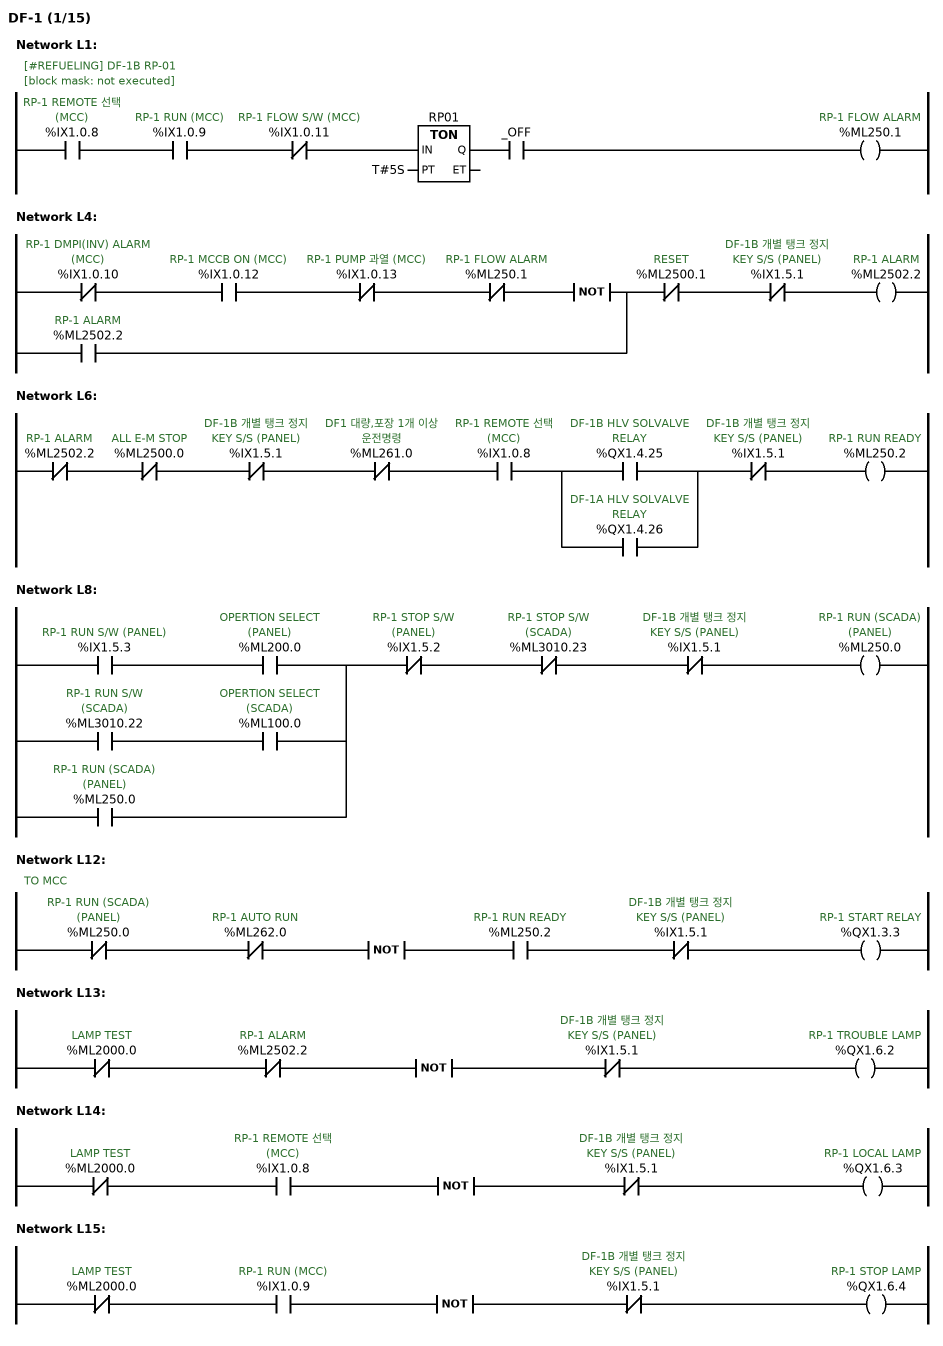
(* [#REFUELING] DF-1B RP-01 *)
(* Rung L1 is block-masked: not executed *)
// RP01(IN := %IX1.0.8 AND %IX1.0.9 AND NOT %IX1.0.11, PT := T#5S);
// %ML250.1 := RP01.Q AND _OFF;
(* Rung L4 *)
%ML2502.2 := (NOT (NOT %IX1.0.10 AND %IX1.0.12 AND NOT %IX1.0.13 AND NOT %ML250.1) OR %ML2502.2) AND NOT %ML2500.1 AND NOT %IX1.5.1;
(* Rung L6 *)
%ML250.2 := NOT %ML2502.2 AND NOT %ML2500.0 AND NOT %IX1.5.1 AND NOT %ML261.0 AND %IX1.0.8 AND (%QX1.4.25 OR %QX1.4.26) AND NOT %IX1.5.1;
(* Rung L8 *)
%ML250.0 := ((%IX1.5.3 AND %ML200.0) OR (%ML3010.22 AND %ML100.0) OR %ML250.0) AND NOT %IX1.5.2 AND NOT %ML3010.23 AND NOT %IX1.5.1;
(* Rung L12 *)
%QX1.3.3 := NOT (NOT %ML250.0 AND NOT %ML262.0) AND %ML250.2 AND NOT %IX1.5.1;
(* TO MCC *)
(* Rung L13 *)
%QX1.6.2 := NOT (NOT %ML2000.0 AND NOT %ML2502.2) AND NOT %IX1.5.1;
(* Rung L14 *)
%QX1.6.3 := NOT (NOT %ML2000.0 AND %IX1.0.8) AND NOT %IX1.5.1;
(* Rung L15 *)
%QX1.6.4 := NOT (NOT %ML2000.0 AND %IX1.0.9) AND NOT %IX1.5.1;

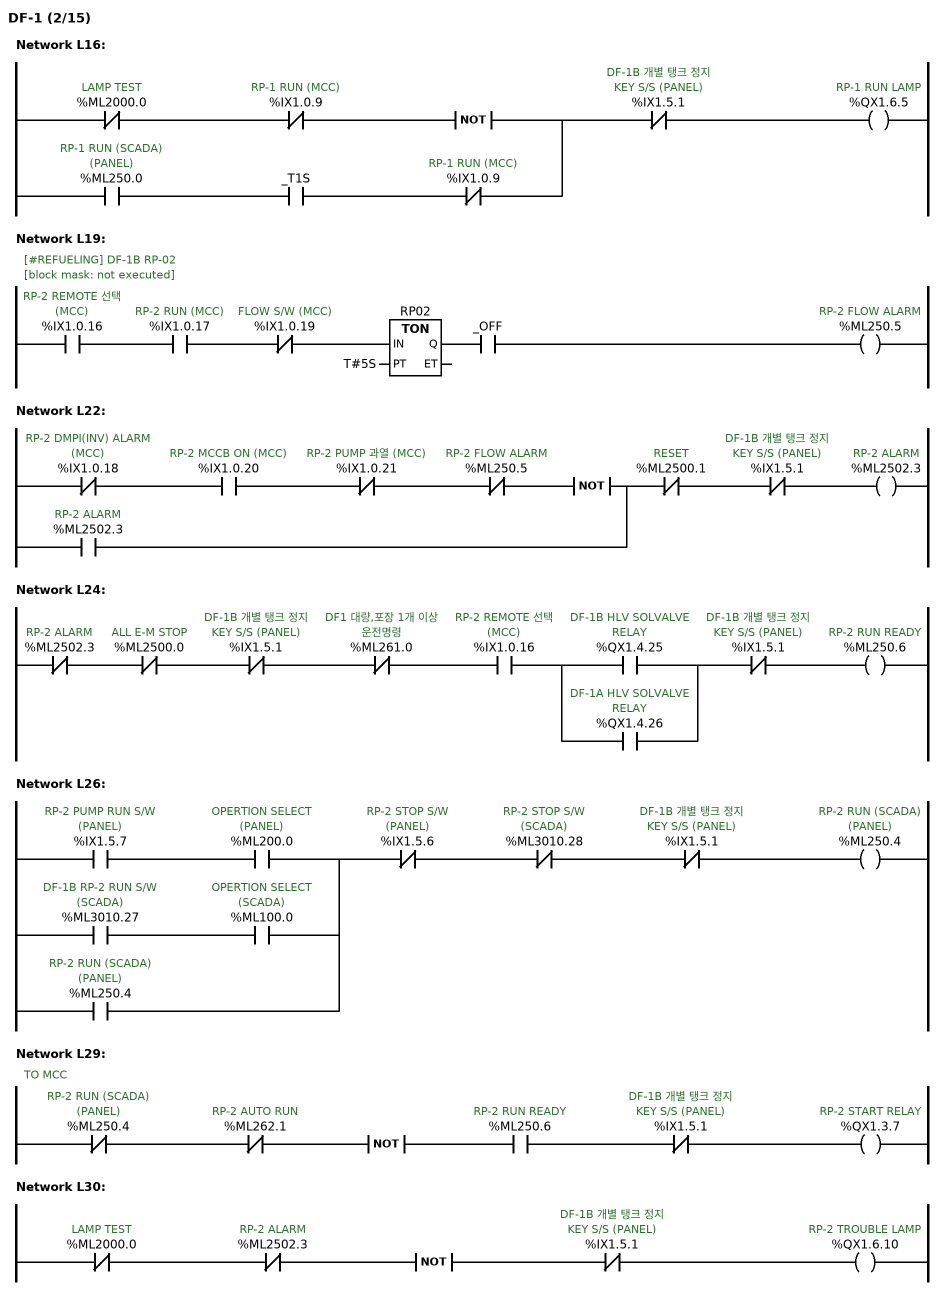
(* Rung L16 *)
%QX1.6.5 := (NOT (NOT %ML2000.0 AND NOT %IX1.0.9) OR (%ML250.0 AND _T1S AND NOT %IX1.0.9)) AND NOT %IX1.5.1;
(* [#REFUELING] DF-1B RP-02 *)
(* Rung L19 is block-masked: not executed *)
// RP02(IN := %IX1.0.16 AND %IX1.0.17 AND NOT %IX1.0.19, PT := T#5S);
// %ML250.5 := RP02.Q AND _OFF;
(* Rung L22 *)
%ML2502.3 := (NOT (NOT %IX1.0.18 AND %IX1.0.20 AND NOT %IX1.0.21 AND NOT %ML250.5) OR %ML2502.3) AND NOT %ML2500.1 AND NOT %IX1.5.1;
(* Rung L24 *)
%ML250.6 := NOT %ML2502.3 AND NOT %ML2500.0 AND NOT %IX1.5.1 AND NOT %ML261.0 AND %IX1.0.16 AND (%QX1.4.25 OR %QX1.4.26) AND NOT %IX1.5.1;
(* Rung L26 *)
%ML250.4 := ((%IX1.5.7 AND %ML200.0) OR (%ML3010.27 AND %ML100.0) OR %ML250.4) AND NOT %IX1.5.6 AND NOT %ML3010.28 AND NOT %IX1.5.1;
(* Rung L29 *)
%QX1.3.7 := NOT (NOT %ML250.4 AND NOT %ML262.1) AND %ML250.6 AND NOT %IX1.5.1;
(* TO MCC *)
(* Rung L30 *)
%QX1.6.10 := NOT (NOT %ML2000.0 AND NOT %ML2502.3) AND NOT %IX1.5.1;

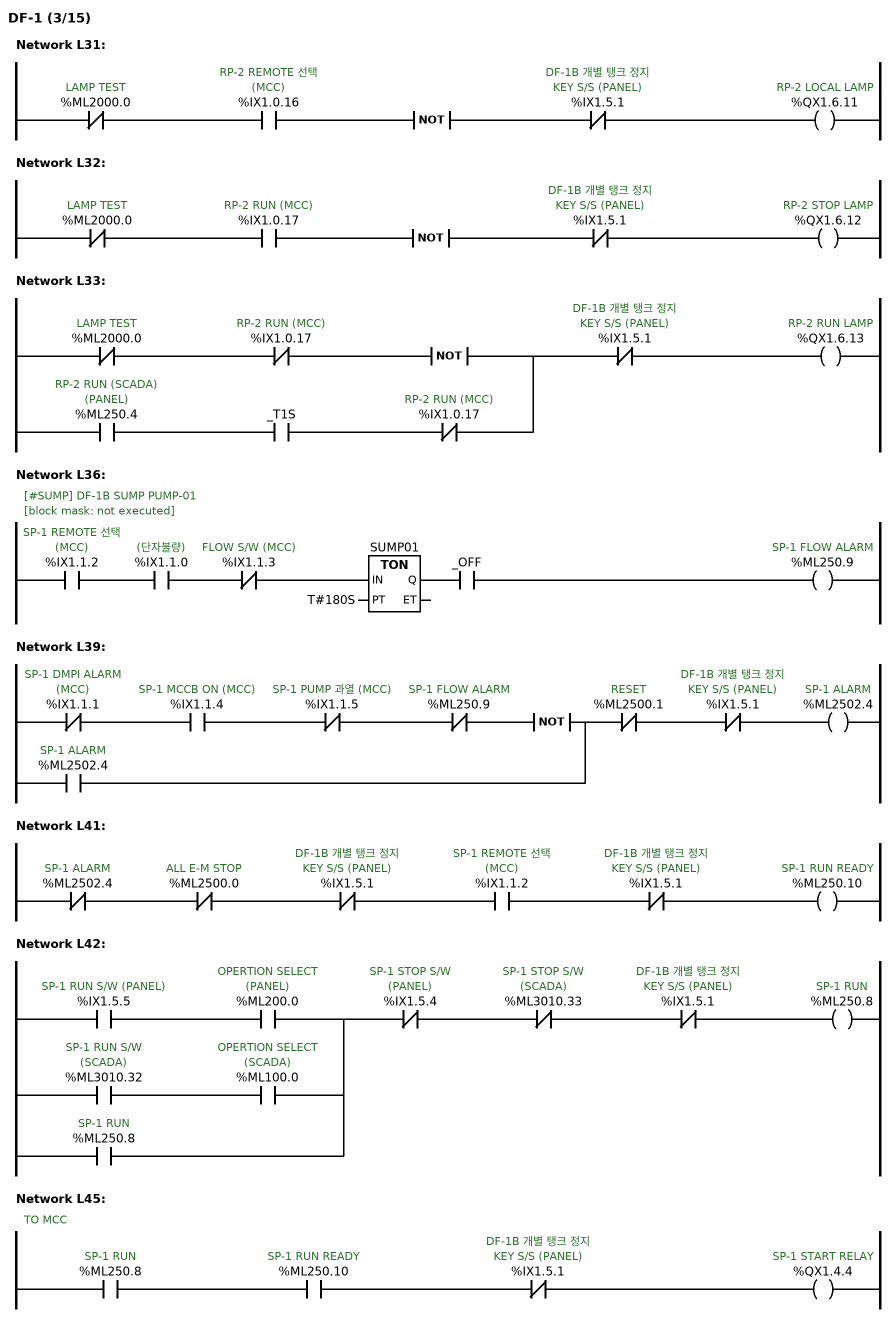
(* Rung L31 *)
%QX1.6.11 := NOT (NOT %ML2000.0 AND %IX1.0.16) AND NOT %IX1.5.1;
(* Rung L32 *)
%QX1.6.12 := NOT (NOT %ML2000.0 AND %IX1.0.17) AND NOT %IX1.5.1;
(* Rung L33 *)
%QX1.6.13 := (NOT (NOT %ML2000.0 AND NOT %IX1.0.17) OR (%ML250.4 AND _T1S AND NOT %IX1.0.17)) AND NOT %IX1.5.1;
(* [#SUMP] DF-1B SUMP PUMP-01 *)
(* Rung L36 is block-masked: not executed *)
// SUMP01(IN := %IX1.1.2 AND %IX1.1.0 AND NOT %IX1.1.3, PT := T#180S);
// %ML250.9 := SUMP01.Q AND _OFF;
(* Rung L39 *)
%ML2502.4 := (NOT (NOT %IX1.1.1 AND %IX1.1.4 AND NOT %IX1.1.5 AND NOT %ML250.9) OR %ML2502.4) AND NOT %ML2500.1 AND NOT %IX1.5.1;
(* Rung L41 *)
%ML250.10 := NOT %ML2502.4 AND NOT %ML2500.0 AND NOT %IX1.5.1 AND %IX1.1.2 AND NOT %IX1.5.1;
(* Rung L42 *)
%ML250.8 := ((%IX1.5.5 AND %ML200.0) OR (%ML3010.32 AND %ML100.0) OR %ML250.8) AND NOT %IX1.5.4 AND NOT %ML3010.33 AND NOT %IX1.5.1;
(* Rung L45 *)
%QX1.4.4 := %ML250.8 AND %ML250.10 AND NOT %IX1.5.1;
(* TO MCC *)

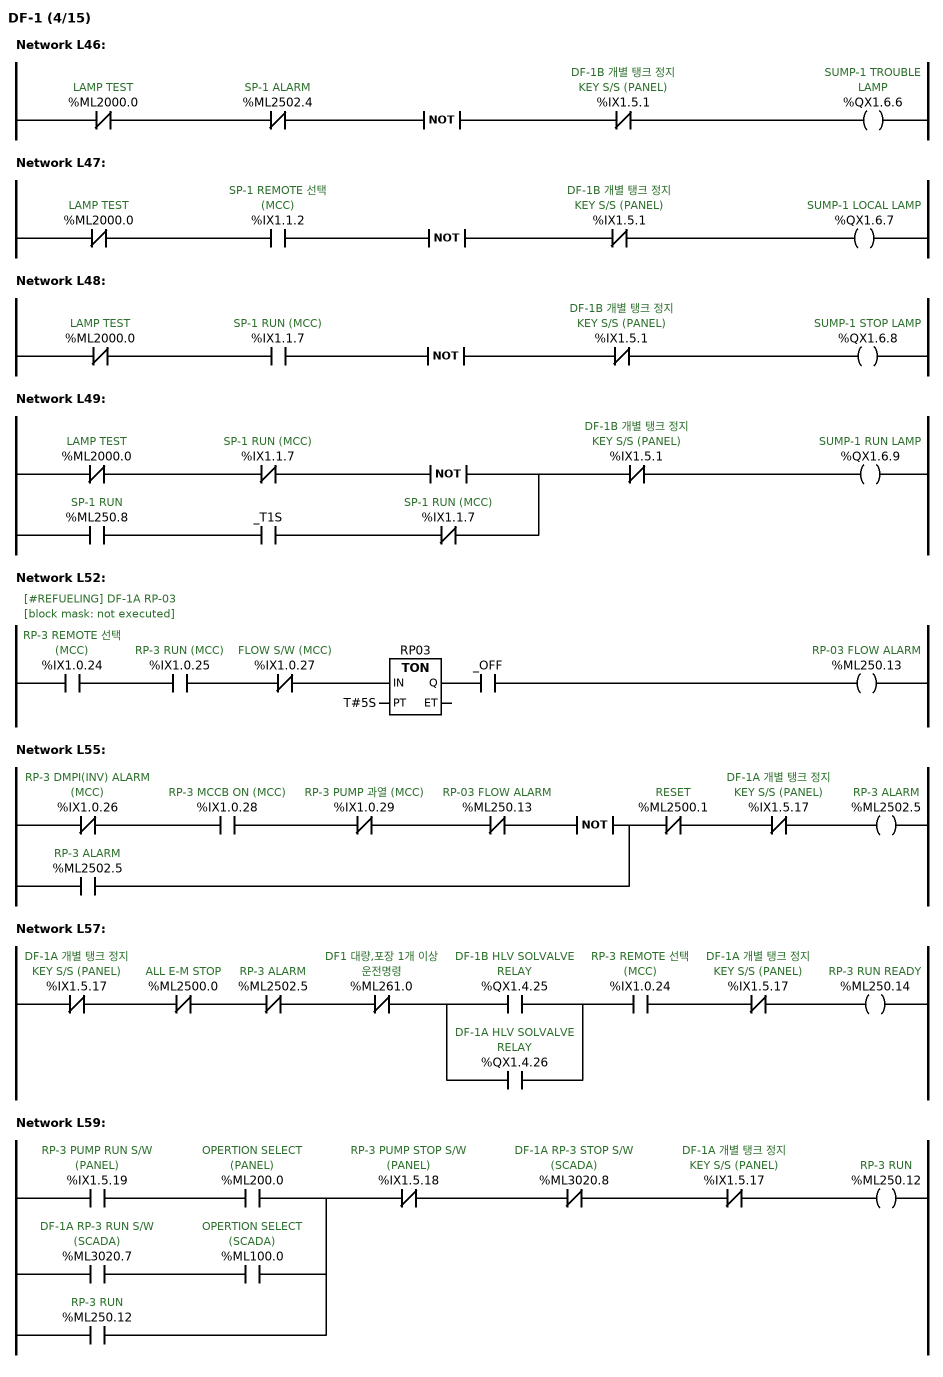
(* Rung L46 *)
%QX1.6.6 := NOT (NOT %ML2000.0 AND NOT %ML2502.4) AND NOT %IX1.5.1;
(* Rung L47 *)
%QX1.6.7 := NOT (NOT %ML2000.0 AND %IX1.1.2) AND NOT %IX1.5.1;
(* Rung L48 *)
%QX1.6.8 := NOT (NOT %ML2000.0 AND %IX1.1.7) AND NOT %IX1.5.1;
(* Rung L49 *)
%QX1.6.9 := (NOT (NOT %ML2000.0 AND NOT %IX1.1.7) OR (%ML250.8 AND _T1S AND NOT %IX1.1.7)) AND NOT %IX1.5.1;
(* [#REFUELING] DF-1A RP-03 *)
(* Rung L52 is block-masked: not executed *)
// RP03(IN := %IX1.0.24 AND %IX1.0.25 AND NOT %IX1.0.27, PT := T#5S);
// %ML250.13 := RP03.Q AND _OFF;
(* Rung L55 *)
%ML2502.5 := (NOT (NOT %IX1.0.26 AND %IX1.0.28 AND NOT %IX1.0.29 AND NOT %ML250.13) OR %ML2502.5) AND NOT %ML2500.1 AND NOT %IX1.5.17;
(* Rung L57 *)
%ML250.14 := NOT %IX1.5.17 AND NOT %ML2500.0 AND NOT %ML2502.5 AND NOT %ML261.0 AND (%QX1.4.25 OR %QX1.4.26) AND %IX1.0.24 AND NOT %IX1.5.17;
(* Rung L59 *)
%ML250.12 := ((%IX1.5.19 AND %ML200.0) OR (%ML3020.7 AND %ML100.0) OR %ML250.12) AND NOT %IX1.5.18 AND NOT %ML3020.8 AND NOT %IX1.5.17;

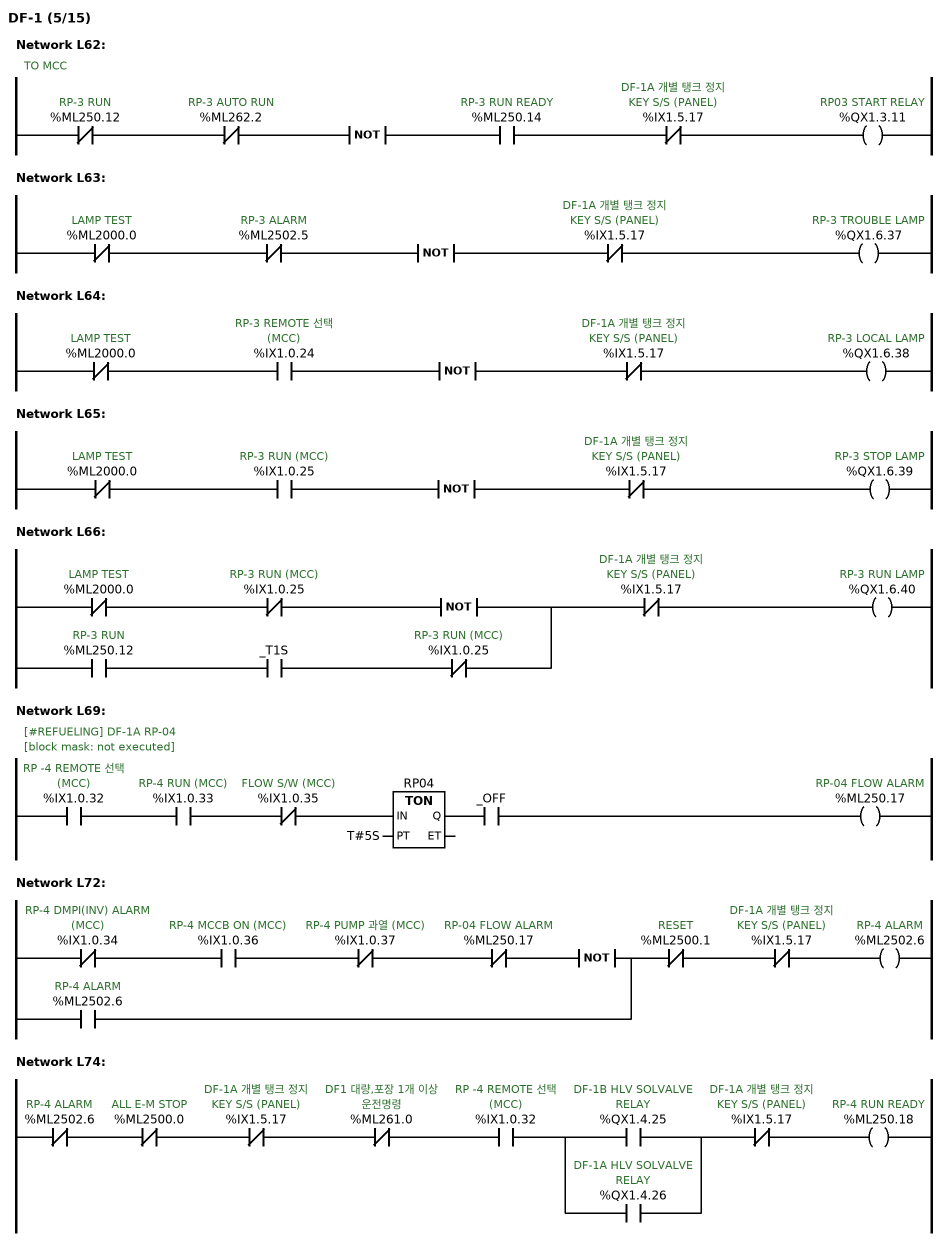
(* Rung L62 *)
%QX1.3.11 := NOT (NOT %ML250.12 AND NOT %ML262.2) AND %ML250.14 AND NOT %IX1.5.17;
(* TO MCC *)
(* Rung L63 *)
%QX1.6.37 := NOT (NOT %ML2000.0 AND NOT %ML2502.5) AND NOT %IX1.5.17;
(* Rung L64 *)
%QX1.6.38 := NOT (NOT %ML2000.0 AND %IX1.0.24) AND NOT %IX1.5.17;
(* Rung L65 *)
%QX1.6.39 := NOT (NOT %ML2000.0 AND %IX1.0.25) AND NOT %IX1.5.17;
(* Rung L66 *)
%QX1.6.40 := (NOT (NOT %ML2000.0 AND NOT %IX1.0.25) OR (%ML250.12 AND _T1S AND NOT %IX1.0.25)) AND NOT %IX1.5.17;
(* [#REFUELING] DF-1A RP-04 *)
(* Rung L69 is block-masked: not executed *)
// RP04(IN := %IX1.0.32 AND %IX1.0.33 AND NOT %IX1.0.35, PT := T#5S);
// %ML250.17 := RP04.Q AND _OFF;
(* Rung L72 *)
%ML2502.6 := (NOT (NOT %IX1.0.34 AND %IX1.0.36 AND NOT %IX1.0.37 AND NOT %ML250.17) OR %ML2502.6) AND NOT %ML2500.1 AND NOT %IX1.5.17;
(* Rung L74 *)
%ML250.18 := NOT %ML2502.6 AND NOT %ML2500.0 AND NOT %IX1.5.17 AND NOT %ML261.0 AND %IX1.0.32 AND (%QX1.4.25 OR %QX1.4.26) AND NOT %IX1.5.17;

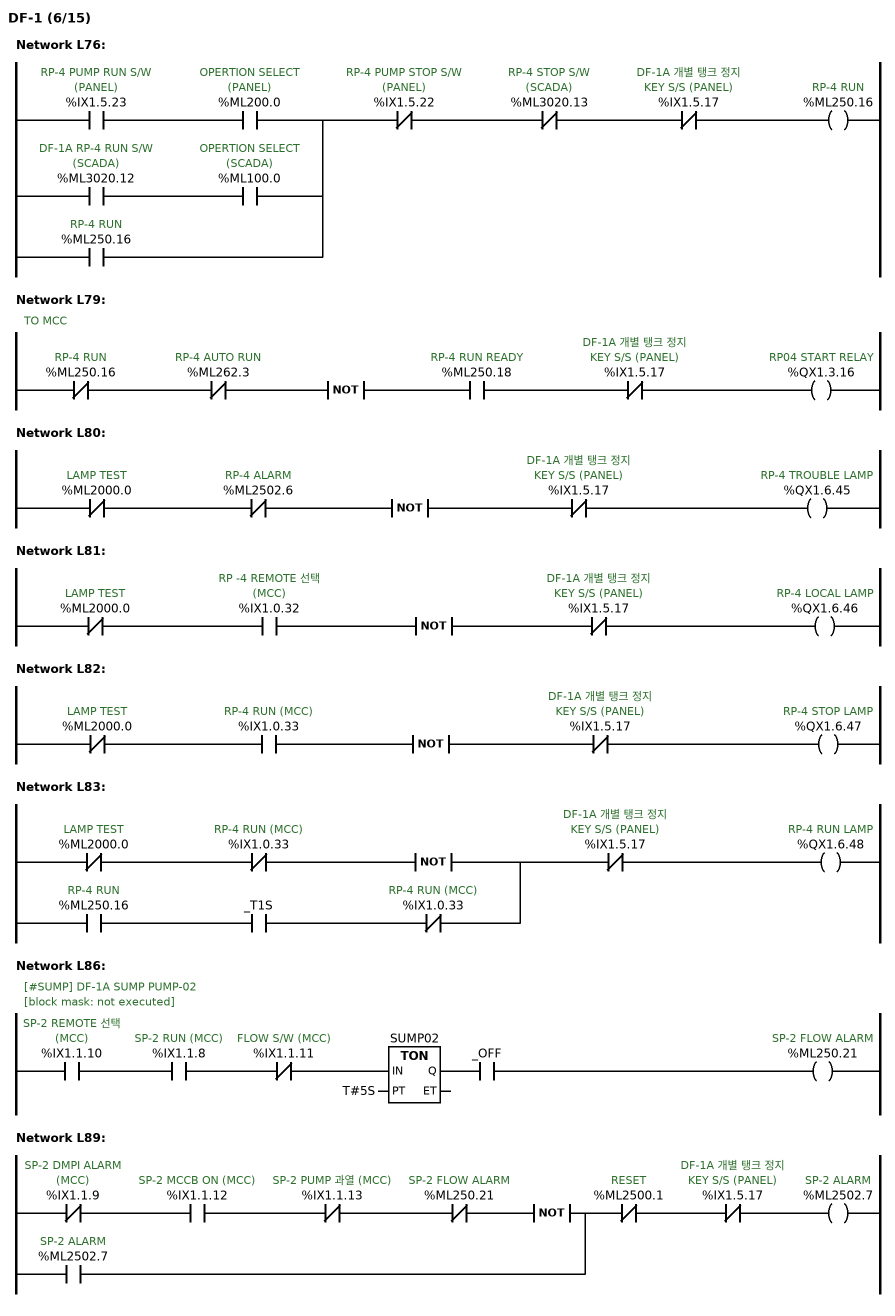
(* Rung L76 *)
%ML250.16 := ((%IX1.5.23 AND %ML200.0) OR (%ML3020.12 AND %ML100.0) OR %ML250.16) AND NOT %IX1.5.22 AND NOT %ML3020.13 AND NOT %IX1.5.17;
(* Rung L79 *)
%QX1.3.16 := NOT (NOT %ML250.16 AND NOT %ML262.3) AND %ML250.18 AND NOT %IX1.5.17;
(* TO MCC *)
(* Rung L80 *)
%QX1.6.45 := NOT (NOT %ML2000.0 AND NOT %ML2502.6) AND NOT %IX1.5.17;
(* Rung L81 *)
%QX1.6.46 := NOT (NOT %ML2000.0 AND %IX1.0.32) AND NOT %IX1.5.17;
(* Rung L82 *)
%QX1.6.47 := NOT (NOT %ML2000.0 AND %IX1.0.33) AND NOT %IX1.5.17;
(* Rung L83 *)
%QX1.6.48 := (NOT (NOT %ML2000.0 AND NOT %IX1.0.33) OR (%ML250.16 AND _T1S AND NOT %IX1.0.33)) AND NOT %IX1.5.17;
(* [#SUMP] DF-1A SUMP PUMP-02 *)
(* Rung L86 is block-masked: not executed *)
// SUMP02(IN := %IX1.1.10 AND %IX1.1.8 AND NOT %IX1.1.11, PT := T#5S);
// %ML250.21 := SUMP02.Q AND _OFF;
(* Rung L89 *)
%ML2502.7 := (NOT (NOT %IX1.1.9 AND %IX1.1.12 AND NOT %IX1.1.13 AND NOT %ML250.21) OR %ML2502.7) AND NOT %ML2500.1 AND NOT %IX1.5.17;

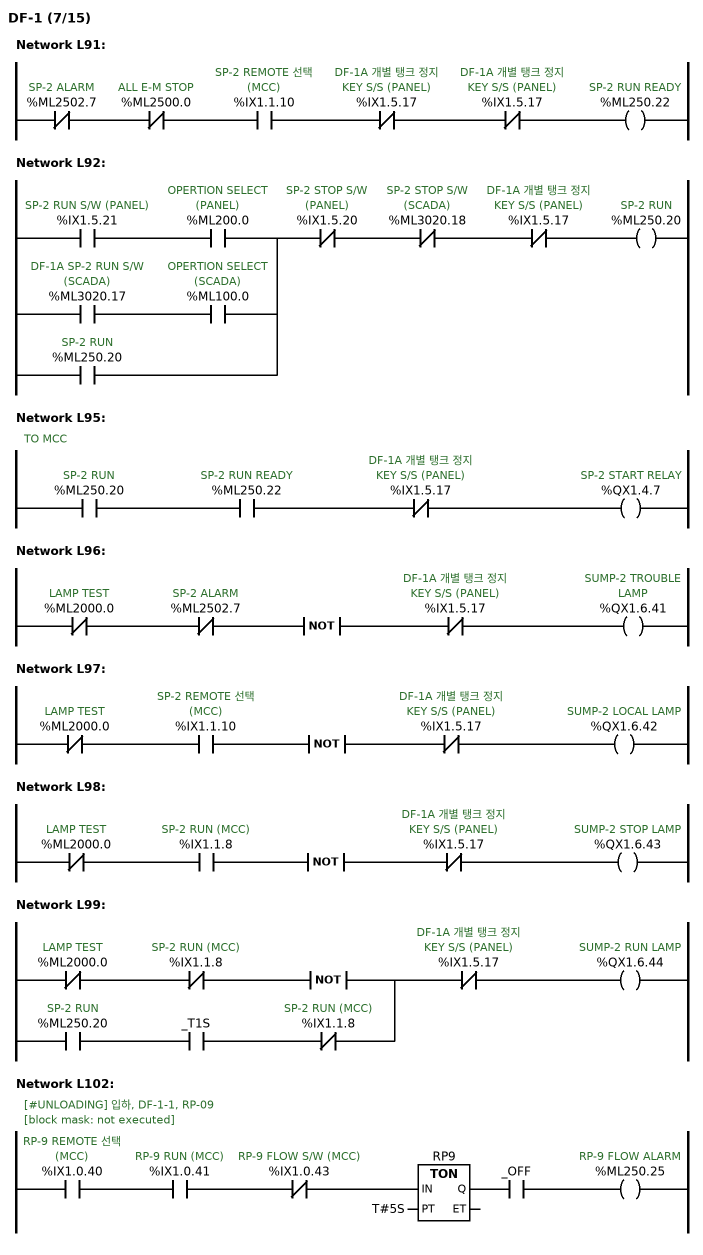
(* Rung L91 *)
%ML250.22 := NOT %ML2502.7 AND NOT %ML2500.0 AND %IX1.1.10 AND NOT %IX1.5.17 AND NOT %IX1.5.17;
(* Rung L92 *)
%ML250.20 := ((%IX1.5.21 AND %ML200.0) OR (%ML3020.17 AND %ML100.0) OR %ML250.20) AND NOT %IX1.5.20 AND NOT %ML3020.18 AND NOT %IX1.5.17;
(* Rung L95 *)
%QX1.4.7 := %ML250.20 AND %ML250.22 AND NOT %IX1.5.17;
(* TO MCC *)
(* Rung L96 *)
%QX1.6.41 := NOT (NOT %ML2000.0 AND NOT %ML2502.7) AND NOT %IX1.5.17;
(* Rung L97 *)
%QX1.6.42 := NOT (NOT %ML2000.0 AND %IX1.1.10) AND NOT %IX1.5.17;
(* Rung L98 *)
%QX1.6.43 := NOT (NOT %ML2000.0 AND %IX1.1.8) AND NOT %IX1.5.17;
(* Rung L99 *)
%QX1.6.44 := (NOT (NOT %ML2000.0 AND NOT %IX1.1.8) OR (%ML250.20 AND _T1S AND NOT %IX1.1.8)) AND NOT %IX1.5.17;
(* [#UNLOADING] 입하, DF-1-1, RP-09 *)
(* Rung L102 is block-masked: not executed *)
// RP9(IN := %IX1.0.40 AND %IX1.0.41 AND NOT %IX1.0.43, PT := T#5S);
// %ML250.25 := RP9.Q AND _OFF;

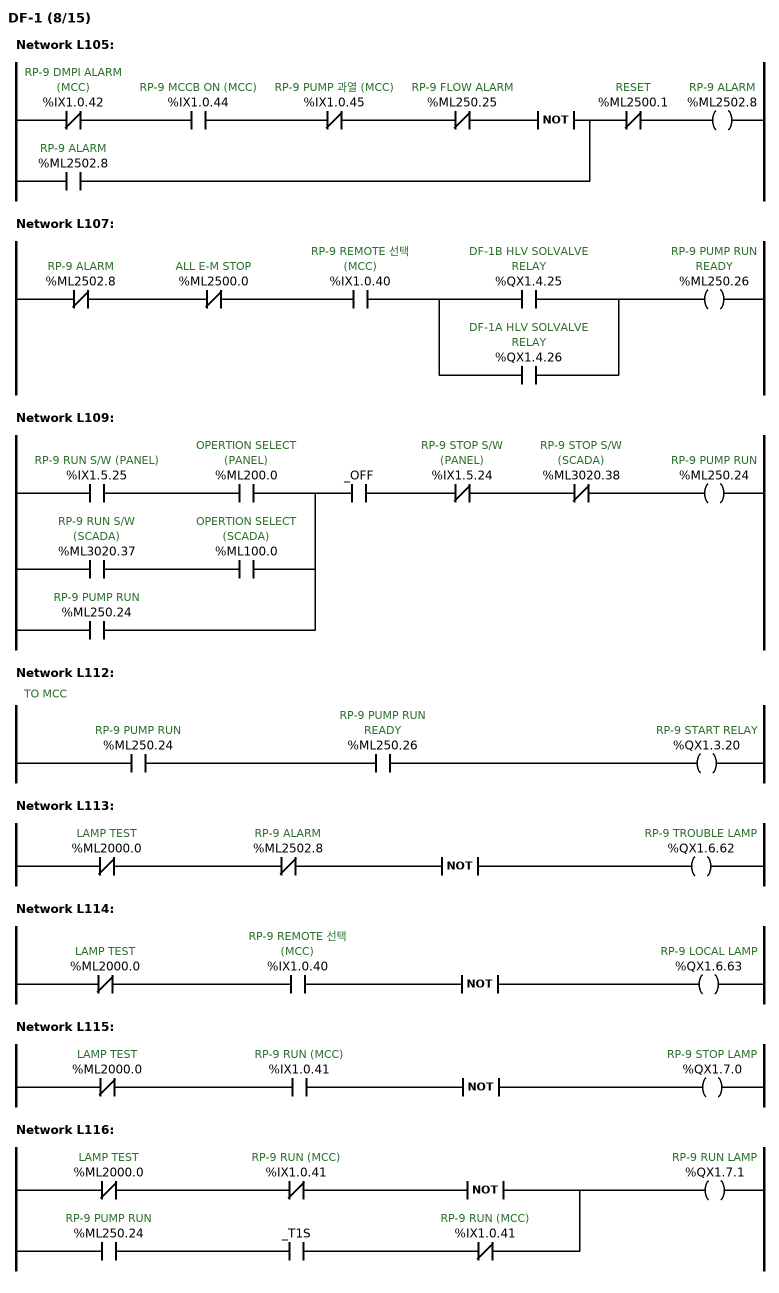
(* Rung L105 *)
%ML2502.8 := (NOT (NOT %IX1.0.42 AND %IX1.0.44 AND NOT %IX1.0.45 AND NOT %ML250.25) OR %ML2502.8) AND NOT %ML2500.1;
(* Rung L107 *)
%ML250.26 := NOT %ML2502.8 AND NOT %ML2500.0 AND %IX1.0.40 AND (%QX1.4.25 OR %QX1.4.26);
(* Rung L109 *)
%ML250.24 := ((%IX1.5.25 AND %ML200.0) OR (%ML3020.37 AND %ML100.0) OR %ML250.24) AND _OFF AND NOT %IX1.5.24 AND NOT %ML3020.38;
(* Rung L112 *)
%QX1.3.20 := %ML250.24 AND %ML250.26;
(* TO MCC *)
(* Rung L113 *)
%QX1.6.62 := NOT (NOT %ML2000.0 AND NOT %ML2502.8);
(* Rung L114 *)
%QX1.6.63 := NOT (NOT %ML2000.0 AND %IX1.0.40);
(* Rung L115 *)
%QX1.7.0 := NOT (NOT %ML2000.0 AND %IX1.0.41);
(* Rung L116 *)
%QX1.7.1 := NOT (NOT %ML2000.0 AND NOT %IX1.0.41) OR (%ML250.24 AND _T1S AND NOT %IX1.0.41);

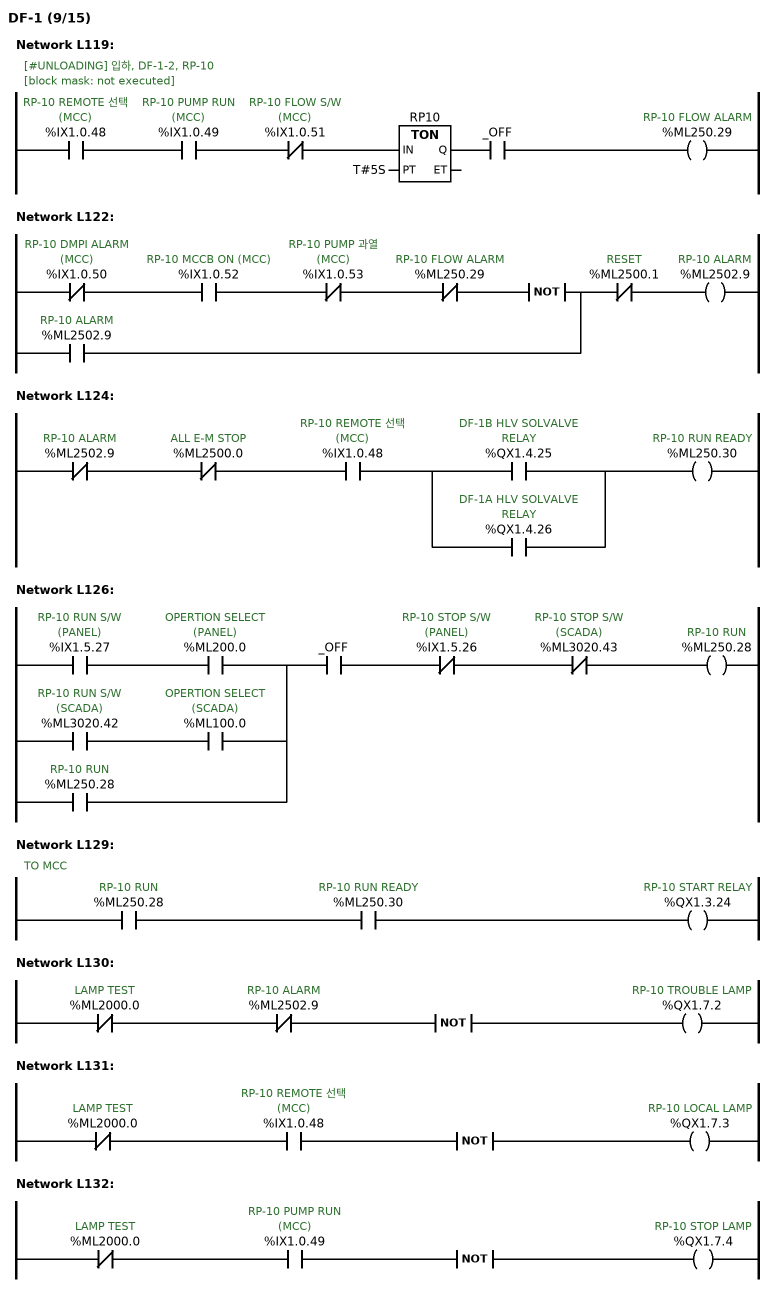
(* [#UNLOADING] 입하, DF-1-2, RP-10 *)
(* Rung L119 is block-masked: not executed *)
// RP10(IN := %IX1.0.48 AND %IX1.0.49 AND NOT %IX1.0.51, PT := T#5S);
// %ML250.29 := RP10.Q AND _OFF;
(* Rung L122 *)
%ML2502.9 := (NOT (NOT %IX1.0.50 AND %IX1.0.52 AND NOT %IX1.0.53 AND NOT %ML250.29) OR %ML2502.9) AND NOT %ML2500.1;
(* Rung L124 *)
%ML250.30 := NOT %ML2502.9 AND NOT %ML2500.0 AND %IX1.0.48 AND (%QX1.4.25 OR %QX1.4.26);
(* Rung L126 *)
%ML250.28 := ((%IX1.5.27 AND %ML200.0) OR (%ML3020.42 AND %ML100.0) OR %ML250.28) AND _OFF AND NOT %IX1.5.26 AND NOT %ML3020.43;
(* Rung L129 *)
%QX1.3.24 := %ML250.28 AND %ML250.30;
(* TO MCC *)
(* Rung L130 *)
%QX1.7.2 := NOT (NOT %ML2000.0 AND NOT %ML2502.9);
(* Rung L131 *)
%QX1.7.3 := NOT (NOT %ML2000.0 AND %IX1.0.48);
(* Rung L132 *)
%QX1.7.4 := NOT (NOT %ML2000.0 AND %IX1.0.49);

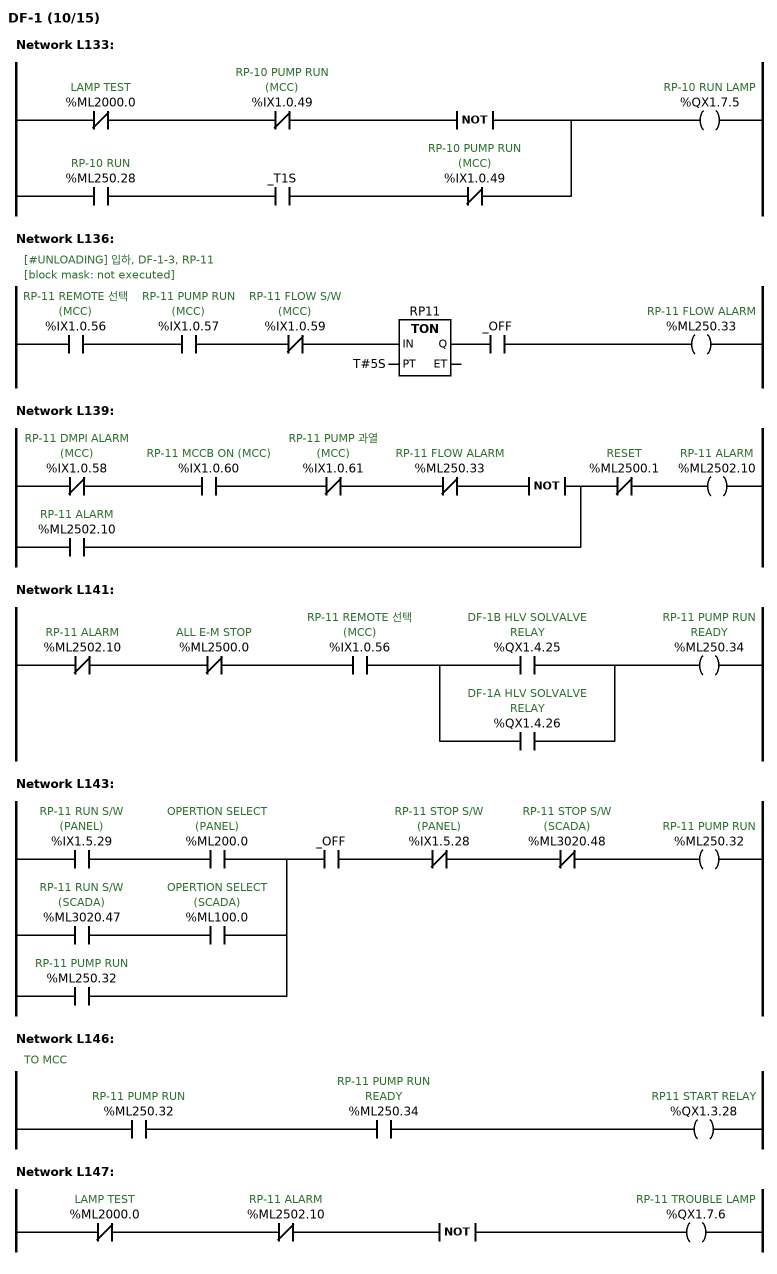
(* Rung L133 *)
%QX1.7.5 := NOT (NOT %ML2000.0 AND NOT %IX1.0.49) OR (%ML250.28 AND _T1S AND NOT %IX1.0.49);
(* [#UNLOADING] 입하, DF-1-3, RP-11 *)
(* Rung L136 is block-masked: not executed *)
// RP11(IN := %IX1.0.56 AND %IX1.0.57 AND NOT %IX1.0.59, PT := T#5S);
// %ML250.33 := RP11.Q AND _OFF;
(* Rung L139 *)
%ML2502.10 := (NOT (NOT %IX1.0.58 AND %IX1.0.60 AND NOT %IX1.0.61 AND NOT %ML250.33) OR %ML2502.10) AND NOT %ML2500.1;
(* Rung L141 *)
%ML250.34 := NOT %ML2502.10 AND NOT %ML2500.0 AND %IX1.0.56 AND (%QX1.4.25 OR %QX1.4.26);
(* Rung L143 *)
%ML250.32 := ((%IX1.5.29 AND %ML200.0) OR (%ML3020.47 AND %ML100.0) OR %ML250.32) AND _OFF AND NOT %IX1.5.28 AND NOT %ML3020.48;
(* Rung L146 *)
%QX1.3.28 := %ML250.32 AND %ML250.34;
(* TO MCC *)
(* Rung L147 *)
%QX1.7.6 := NOT (NOT %ML2000.0 AND NOT %ML2502.10);

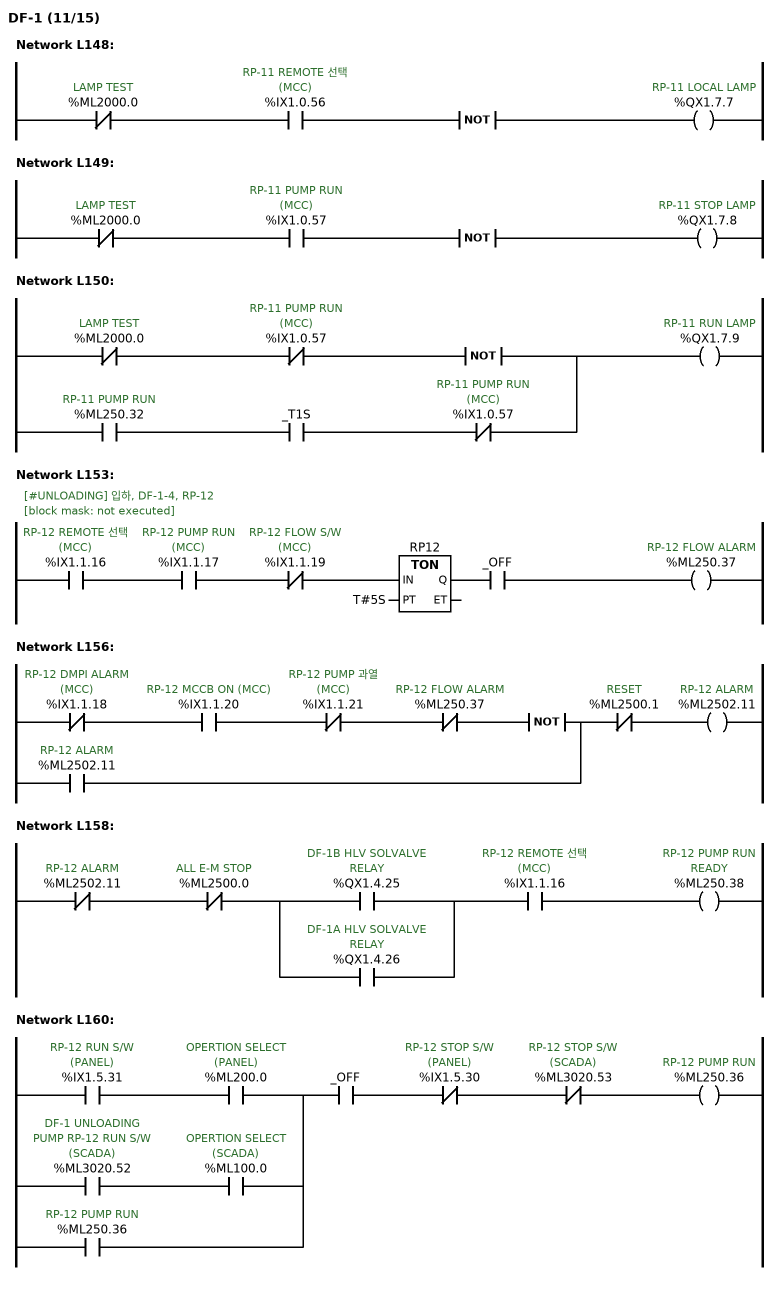
(* Rung L148 *)
%QX1.7.7 := NOT (NOT %ML2000.0 AND %IX1.0.56);
(* Rung L149 *)
%QX1.7.8 := NOT (NOT %ML2000.0 AND %IX1.0.57);
(* Rung L150 *)
%QX1.7.9 := NOT (NOT %ML2000.0 AND NOT %IX1.0.57) OR (%ML250.32 AND _T1S AND NOT %IX1.0.57);
(* [#UNLOADING] 입하, DF-1-4, RP-12 *)
(* Rung L153 is block-masked: not executed *)
// RP12(IN := %IX1.1.16 AND %IX1.1.17 AND NOT %IX1.1.19, PT := T#5S);
// %ML250.37 := RP12.Q AND _OFF;
(* Rung L156 *)
%ML2502.11 := (NOT (NOT %IX1.1.18 AND %IX1.1.20 AND NOT %IX1.1.21 AND NOT %ML250.37) OR %ML2502.11) AND NOT %ML2500.1;
(* Rung L158 *)
%ML250.38 := NOT %ML2502.11 AND NOT %ML2500.0 AND (%QX1.4.25 OR %QX1.4.26) AND %IX1.1.16;
(* Rung L160 *)
%ML250.36 := ((%IX1.5.31 AND %ML200.0) OR (%ML3020.52 AND %ML100.0) OR %ML250.36) AND _OFF AND NOT %IX1.5.30 AND NOT %ML3020.53;

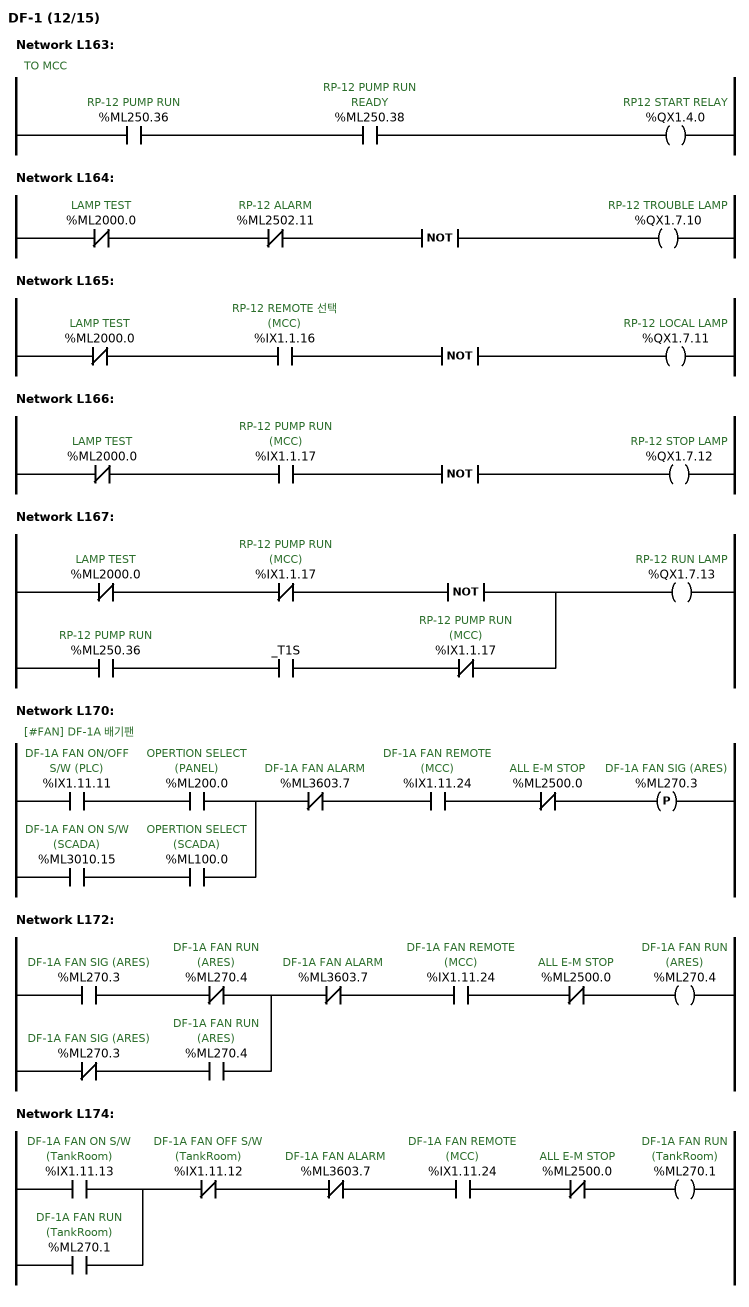
(* Rung L163 *)
%QX1.4.0 := %ML250.36 AND %ML250.38;
(* TO MCC *)
(* Rung L164 *)
%QX1.7.10 := NOT (NOT %ML2000.0 AND NOT %ML2502.11);
(* Rung L165 *)
%QX1.7.11 := NOT (NOT %ML2000.0 AND %IX1.1.16);
(* Rung L166 *)
%QX1.7.12 := NOT (NOT %ML2000.0 AND %IX1.1.17);
(* Rung L167 *)
%QX1.7.13 := NOT (NOT %ML2000.0 AND NOT %IX1.1.17) OR (%ML250.36 AND _T1S AND NOT %IX1.1.17);
(* [#FAN] DF-1A 배기팬 *)
(* Rung L170 *)
_e1(CLK := ((%IX1.11.11 AND %ML200.0) OR (%ML3010.15 AND %ML100.0)) AND NOT %ML3603.7 AND %IX1.11.24 AND NOT %ML2500.0);
%ML270.3 := _e1.Q;
(* Rung L172 *)
%ML270.4 := ((%ML270.3 AND NOT %ML270.4) OR (NOT %ML270.3 AND %ML270.4)) AND NOT %ML3603.7 AND %IX1.11.24 AND NOT %ML2500.0;
(* Rung L174 *)
%ML270.1 := (%IX1.11.13 OR %ML270.1) AND NOT %IX1.11.12 AND NOT %ML3603.7 AND %IX1.11.24 AND NOT %ML2500.0;

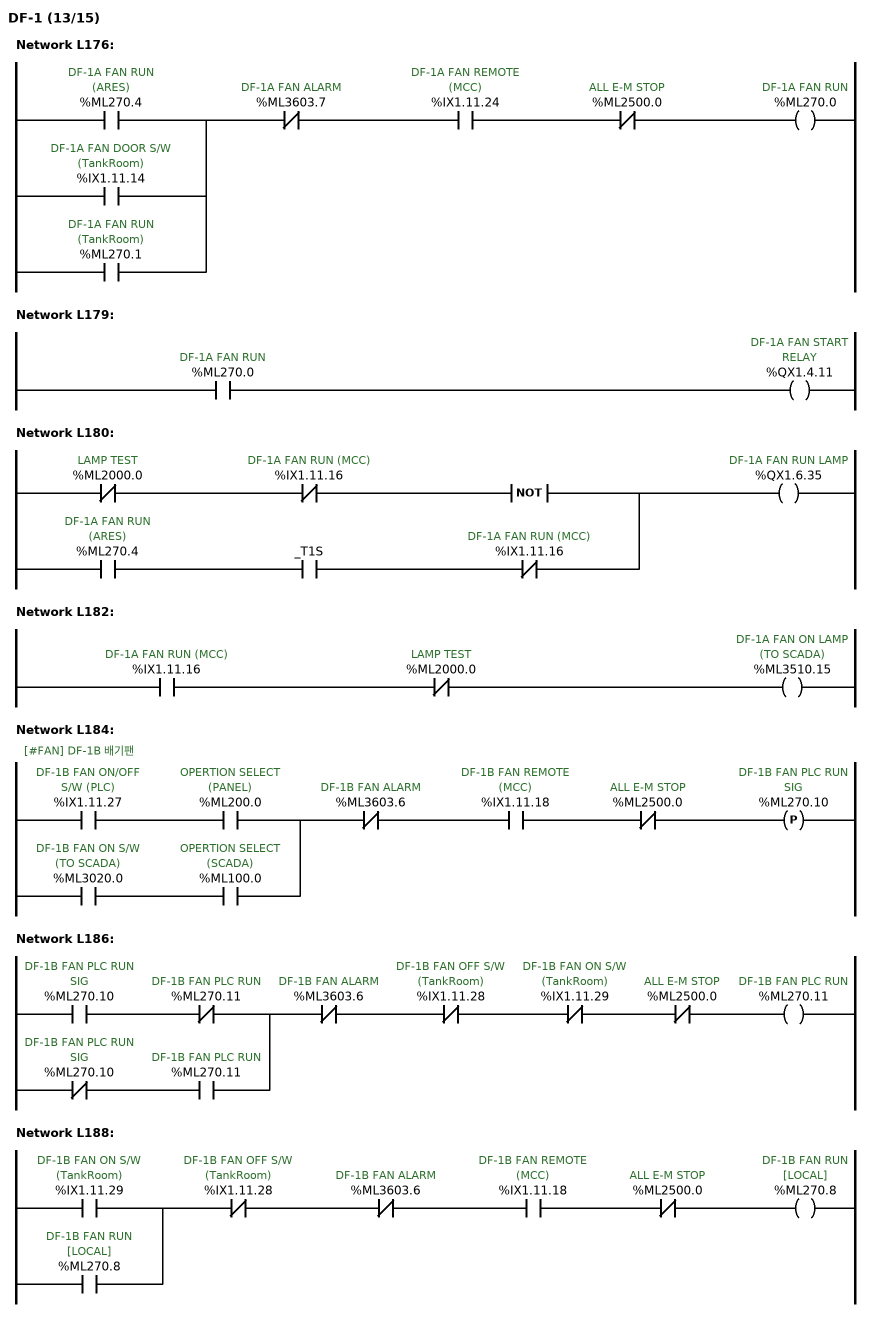
(* Rung L176 *)
%ML270.0 := (%ML270.4 OR %IX1.11.14 OR %ML270.1) AND NOT %ML3603.7 AND %IX1.11.24 AND NOT %ML2500.0;
(* Rung L179 *)
%QX1.4.11 := %ML270.0;
(* Rung L180 *)
%QX1.6.35 := NOT (NOT %ML2000.0 AND NOT %IX1.11.16) OR (%ML270.4 AND _T1S AND NOT %IX1.11.16);
(* Rung L182 *)
%ML3510.15 := %IX1.11.16 AND NOT %ML2000.0;
(* [#FAN] DF-1B 배기팬 *)
(* Rung L184 *)
_e2(CLK := ((%IX1.11.27 AND %ML200.0) OR (%ML3020.0 AND %ML100.0)) AND NOT %ML3603.6 AND %IX1.11.18 AND NOT %ML2500.0);
%ML270.10 := _e2.Q;
(* Rung L186 *)
%ML270.11 := ((%ML270.10 AND NOT %ML270.11) OR (NOT %ML270.10 AND %ML270.11)) AND NOT %ML3603.6 AND NOT %IX1.11.28 AND NOT %IX1.11.29 AND NOT %ML2500.0;
(* Rung L188 *)
%ML270.8 := (%IX1.11.29 OR %ML270.8) AND NOT %IX1.11.28 AND NOT %ML3603.6 AND %IX1.11.18 AND NOT %ML2500.0;

